// TIA Portal V17 export
// export: Created 2025-03-07T09:17:18.0223508Z, ExportSetting WithDefaults, DisplayName Totally Integrated Automation Portal, DisplayVersion V17 Update 8, DisplayName TIA Portal Openness, DisplayVersion V17 Update 8, DisplayName TIA Portal Version Control Interface, DisplayVersion V17, DisplayName SINAMICS Startdrive Advanced, DisplayVersion V17 SP2, DisplayName SINAMICS Startdrive G110M, G120, G120C, G120D, G120P, G115D, DisplayVersion V17 SP2, DisplayName SINAMICS Startdrive G130, G150, S120, S150, SINAMICS MV, S210, DisplayVersion V17 SP2, DisplayName STEP 7 Professional, DisplayVersion V17 Update 8, DisplayName SINUMERIK ONE STEP 7 Toolbox, DisplayVersion V17 Update 12, DisplayName SINUMERIK 840D sl STEP 7 Toolbox, DisplayVersion V17 Update 12, DisplayName STEP 7 Safety, DisplayVersion V17 Update 6, DisplayName WinCC Advanced, DisplayVersion V17 Update 8
FUNCTION "FC357_NCK_M_CH4_UNIT_2_STA_0" : Void   // FC357, LAD
TITLE = Channel 1 data
{ S7_Optimized_Access := 'FALSE' }
AUTHOR : ETXETAR
VERSION : 1.0
// stored: AutoNumber false, IsIECCheckEnabled false, SetENOAutomatically false, UDAEnableTagReadback false
BEGIN

REGION Network 1: ACKNOWLEDGE M400-UNIT 02 FIXTURE 1 CLAMP SEQUENCE (READ-IN DISABLE) / ACKNOWLEDGE M100-CLAMP SEQUENCE FIXTURE 1
   // NOTE: WHEN THERE IS NOT INDEXING TABLE AVAILABLE IN THE MACHINE DELETE 
   // DB2171.DBX5.0 AND DB2171.DBX2.0
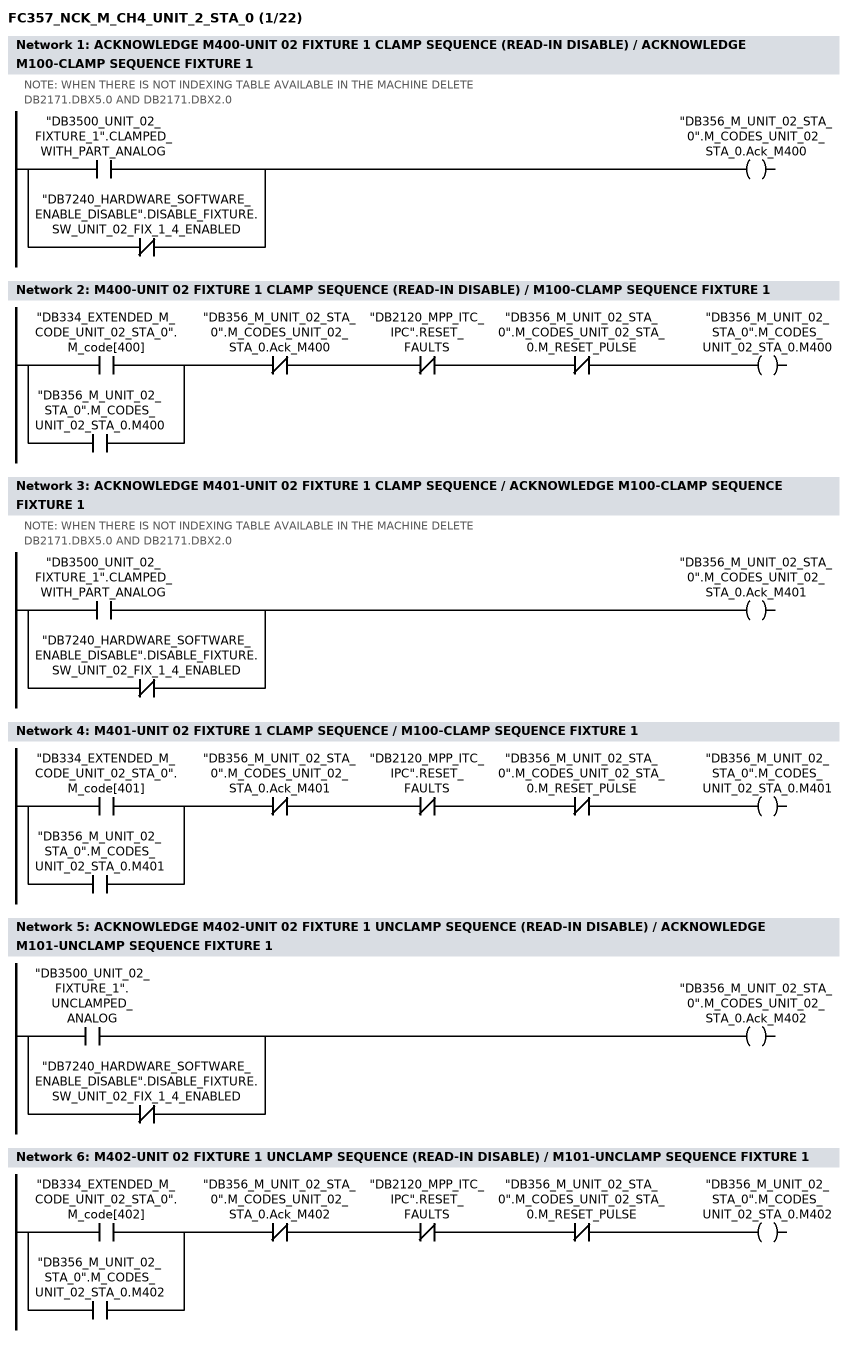
   RUNG wire#powerrail
      Contact( "DB3500_UNIT_02_FIXTURE_1".CLAMPED_WITH_PART_ANALOG )
      wire#w1
      Coil( "DB356_M_UNIT_02_STA_0".M_CODES_UNIT_02_STA_0.Ack_M400 )
   END_RUNG
   RUNG wire#powerrail
      I_Contact( "DB7240_HARDWARE_SOFTWARE_ENABLE_DISABLE".DISABLE_FIXTURE.SW_UNIT_02_FIX_1_4_ENABLED )
   END_RUNG wire#w1
   // the same network as SCL:
   "DB356_M_UNIT_02_STA_0".M_CODES_UNIT_02_STA_0.Ack_M400 := "DB3500_UNIT_02_FIXTURE_1".CLAMPED_WITH_PART_ANALOG OR NOT "DB7240_HARDWARE_SOFTWARE_ENABLE_DISABLE".DISABLE_FIXTURE.SW_UNIT_02_FIX_1_4_ENABLED;
END_REGION

REGION Network 2: M400-UNIT 02 FIXTURE 1 CLAMP SEQUENCE (READ-IN DISABLE) / M100-CLAMP SEQUENCE FIXTURE 1
   RUNG wire#powerrail
      Contact( "DB334_EXTENDED_M_CODE_UNIT_02_STA_0".M_code[400] )
      wire#w1
      I_Contact( "DB356_M_UNIT_02_STA_0".M_CODES_UNIT_02_STA_0.Ack_M400 )
      I_Contact( "DB2120_MPP_ITC_IPC".RESET_FAULTS )
      I_Contact( "DB356_M_UNIT_02_STA_0".M_CODES_UNIT_02_STA_0.M_RESET_PULSE )
      Coil( "DB356_M_UNIT_02_STA_0".M_CODES_UNIT_02_STA_0.M400 )
   END_RUNG
   RUNG wire#powerrail
      Contact( "DB356_M_UNIT_02_STA_0".M_CODES_UNIT_02_STA_0.M400 )
   END_RUNG wire#w1
   // the same network as SCL:
   "DB356_M_UNIT_02_STA_0".M_CODES_UNIT_02_STA_0.M400 := ("DB334_EXTENDED_M_CODE_UNIT_02_STA_0".M_code[400] OR "DB356_M_UNIT_02_STA_0".M_CODES_UNIT_02_STA_0.M400) AND NOT "DB356_M_UNIT_02_STA_0".M_CODES_UNIT_02_STA_0.Ack_M400 AND NOT "DB2120_MPP_ITC_IPC".RESET_FAULTS AND NOT "DB356_M_UNIT_02_STA_0".M_CODES_UNIT_02_STA_0.M_RESET_PULSE;
END_REGION

REGION Network 3: ACKNOWLEDGE M401-UNIT 02 FIXTURE 1 CLAMP SEQUENCE / ACKNOWLEDGE M100-CLAMP SEQUENCE FIXTURE 1
   // NOTE: WHEN THERE IS NOT INDEXING TABLE AVAILABLE IN THE MACHINE DELETE 
   // DB2171.DBX5.0 AND DB2171.DBX2.0
   RUNG wire#powerrail
      Contact( "DB3500_UNIT_02_FIXTURE_1".CLAMPED_WITH_PART_ANALOG )
      wire#w1
      Coil( "DB356_M_UNIT_02_STA_0".M_CODES_UNIT_02_STA_0.Ack_M401 )
   END_RUNG
   RUNG wire#powerrail
      I_Contact( "DB7240_HARDWARE_SOFTWARE_ENABLE_DISABLE".DISABLE_FIXTURE.SW_UNIT_02_FIX_1_4_ENABLED )
   END_RUNG wire#w1
   // the same network as SCL:
   "DB356_M_UNIT_02_STA_0".M_CODES_UNIT_02_STA_0.Ack_M401 := "DB3500_UNIT_02_FIXTURE_1".CLAMPED_WITH_PART_ANALOG OR NOT "DB7240_HARDWARE_SOFTWARE_ENABLE_DISABLE".DISABLE_FIXTURE.SW_UNIT_02_FIX_1_4_ENABLED;
END_REGION

REGION Network 4: M401-UNIT 02 FIXTURE 1 CLAMP SEQUENCE / M100-CLAMP SEQUENCE FIXTURE 1
   RUNG wire#powerrail
      Contact( "DB334_EXTENDED_M_CODE_UNIT_02_STA_0".M_code[401] )
      wire#w1
      I_Contact( "DB356_M_UNIT_02_STA_0".M_CODES_UNIT_02_STA_0.Ack_M401 )
      I_Contact( "DB2120_MPP_ITC_IPC".RESET_FAULTS )
      I_Contact( "DB356_M_UNIT_02_STA_0".M_CODES_UNIT_02_STA_0.M_RESET_PULSE )
      Coil( "DB356_M_UNIT_02_STA_0".M_CODES_UNIT_02_STA_0.M401 )
   END_RUNG
   RUNG wire#powerrail
      Contact( "DB356_M_UNIT_02_STA_0".M_CODES_UNIT_02_STA_0.M401 )
   END_RUNG wire#w1
   // the same network as SCL:
   "DB356_M_UNIT_02_STA_0".M_CODES_UNIT_02_STA_0.M401 := ("DB334_EXTENDED_M_CODE_UNIT_02_STA_0".M_code[401] OR "DB356_M_UNIT_02_STA_0".M_CODES_UNIT_02_STA_0.M401) AND NOT "DB356_M_UNIT_02_STA_0".M_CODES_UNIT_02_STA_0.Ack_M401 AND NOT "DB2120_MPP_ITC_IPC".RESET_FAULTS AND NOT "DB356_M_UNIT_02_STA_0".M_CODES_UNIT_02_STA_0.M_RESET_PULSE;
END_REGION

REGION Network 5: ACKNOWLEDGE M402-UNIT 02 FIXTURE 1 UNCLAMP SEQUENCE (READ-IN DISABLE) / ACKNOWLEDGE M101-UNCLAMP SEQUENCE FIXTURE 1
   RUNG wire#powerrail
      Contact( "DB3500_UNIT_02_FIXTURE_1".UNCLAMPED_ANALOG )
      wire#w1
      Coil( "DB356_M_UNIT_02_STA_0".M_CODES_UNIT_02_STA_0.Ack_M402 )
   END_RUNG
   RUNG wire#powerrail
      I_Contact( "DB7240_HARDWARE_SOFTWARE_ENABLE_DISABLE".DISABLE_FIXTURE.SW_UNIT_02_FIX_1_4_ENABLED )
   END_RUNG wire#w1
   // the same network as SCL:
   "DB356_M_UNIT_02_STA_0".M_CODES_UNIT_02_STA_0.Ack_M402 := "DB3500_UNIT_02_FIXTURE_1".UNCLAMPED_ANALOG OR NOT "DB7240_HARDWARE_SOFTWARE_ENABLE_DISABLE".DISABLE_FIXTURE.SW_UNIT_02_FIX_1_4_ENABLED;
END_REGION

REGION Network 6: M402-UNIT 02 FIXTURE 1 UNCLAMP SEQUENCE (READ-IN DISABLE) / M101-UNCLAMP SEQUENCE FIXTURE 1
   RUNG wire#powerrail
      Contact( "DB334_EXTENDED_M_CODE_UNIT_02_STA_0".M_code[402] )
      wire#w1
      I_Contact( "DB356_M_UNIT_02_STA_0".M_CODES_UNIT_02_STA_0.Ack_M402 )
      I_Contact( "DB2120_MPP_ITC_IPC".RESET_FAULTS )
      I_Contact( "DB356_M_UNIT_02_STA_0".M_CODES_UNIT_02_STA_0.M_RESET_PULSE )
      Coil( "DB356_M_UNIT_02_STA_0".M_CODES_UNIT_02_STA_0.M402 )
   END_RUNG
   RUNG wire#powerrail
      Contact( "DB356_M_UNIT_02_STA_0".M_CODES_UNIT_02_STA_0.M402 )
   END_RUNG wire#w1
   // the same network as SCL:
   "DB356_M_UNIT_02_STA_0".M_CODES_UNIT_02_STA_0.M402 := ("DB334_EXTENDED_M_CODE_UNIT_02_STA_0".M_code[402] OR "DB356_M_UNIT_02_STA_0".M_CODES_UNIT_02_STA_0.M402) AND NOT "DB356_M_UNIT_02_STA_0".M_CODES_UNIT_02_STA_0.Ack_M402 AND NOT "DB2120_MPP_ITC_IPC".RESET_FAULTS AND NOT "DB356_M_UNIT_02_STA_0".M_CODES_UNIT_02_STA_0.M_RESET_PULSE;
END_REGION

REGION Network 7: ACKNOWLEDGE M403-UNIT 02 FIXTURE 1 UNCLAMP SEQUENCE / ACKNOWLEDGE M101-UNCLAMP SEQUENCE FIXTURE 1
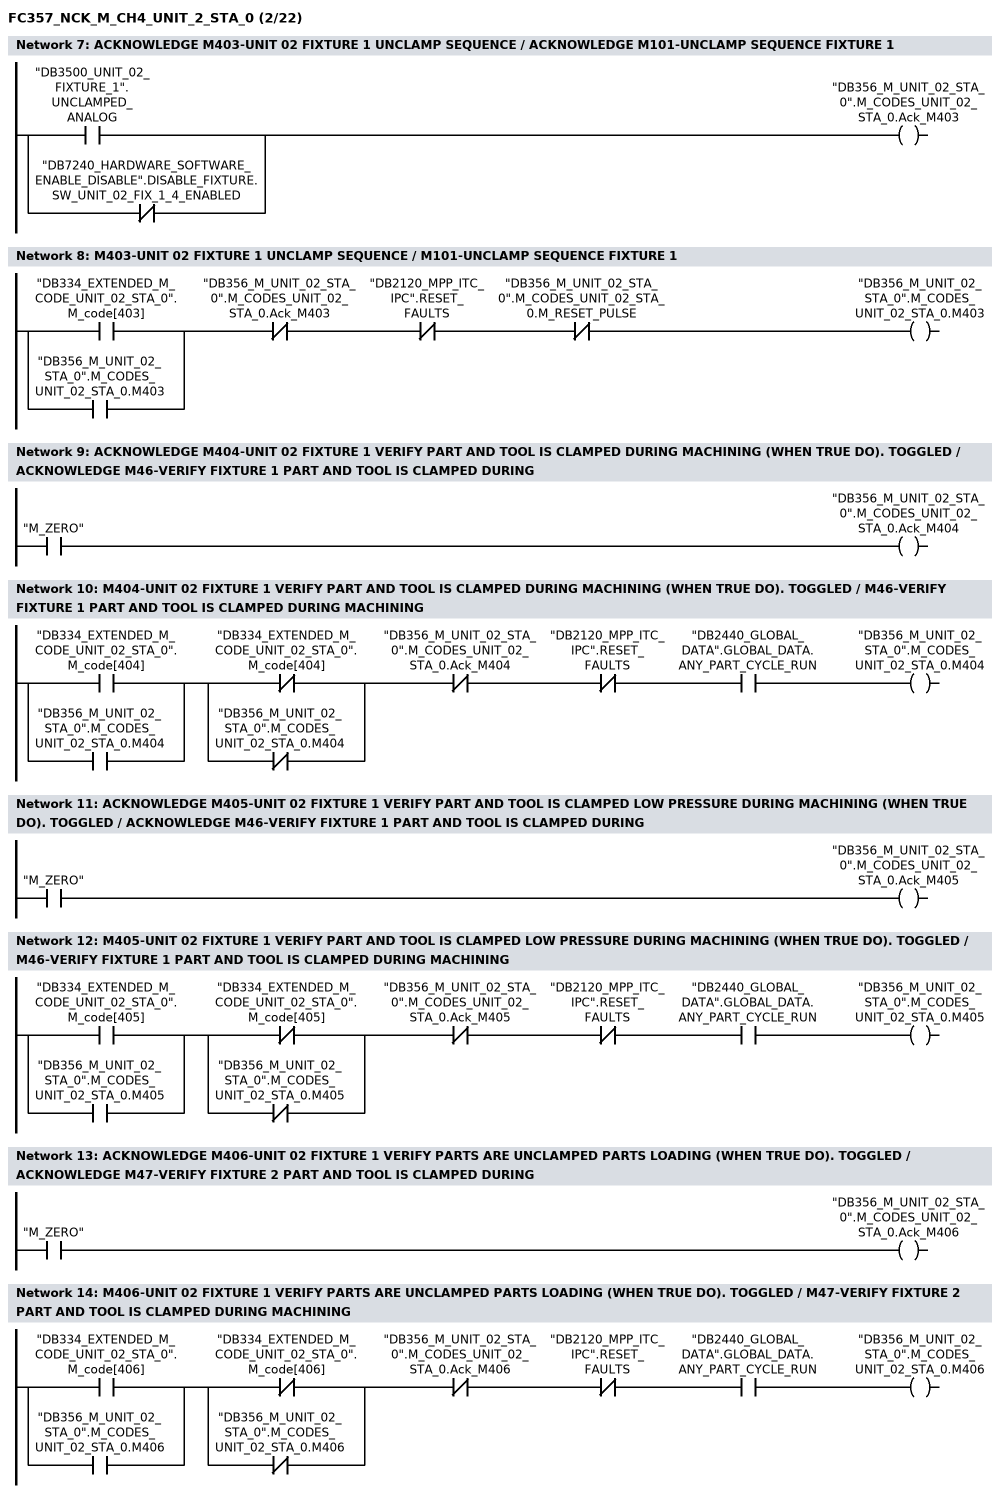
   RUNG wire#powerrail
      Contact( "DB3500_UNIT_02_FIXTURE_1".UNCLAMPED_ANALOG )
      wire#w1
      Coil( "DB356_M_UNIT_02_STA_0".M_CODES_UNIT_02_STA_0.Ack_M403 )
   END_RUNG
   RUNG wire#powerrail
      I_Contact( "DB7240_HARDWARE_SOFTWARE_ENABLE_DISABLE".DISABLE_FIXTURE.SW_UNIT_02_FIX_1_4_ENABLED )
   END_RUNG wire#w1
   // the same network as SCL:
   "DB356_M_UNIT_02_STA_0".M_CODES_UNIT_02_STA_0.Ack_M403 := "DB3500_UNIT_02_FIXTURE_1".UNCLAMPED_ANALOG OR NOT "DB7240_HARDWARE_SOFTWARE_ENABLE_DISABLE".DISABLE_FIXTURE.SW_UNIT_02_FIX_1_4_ENABLED;
END_REGION

REGION Network 8: M403-UNIT 02 FIXTURE 1 UNCLAMP SEQUENCE / M101-UNCLAMP SEQUENCE FIXTURE 1
   RUNG wire#powerrail
      Contact( "DB334_EXTENDED_M_CODE_UNIT_02_STA_0".M_code[403] )
      wire#w1
      I_Contact( "DB356_M_UNIT_02_STA_0".M_CODES_UNIT_02_STA_0.Ack_M403 )
      I_Contact( "DB2120_MPP_ITC_IPC".RESET_FAULTS )
      I_Contact( "DB356_M_UNIT_02_STA_0".M_CODES_UNIT_02_STA_0.M_RESET_PULSE )
      Coil( "DB356_M_UNIT_02_STA_0".M_CODES_UNIT_02_STA_0.M403 )
   END_RUNG
   RUNG wire#powerrail
      Contact( "DB356_M_UNIT_02_STA_0".M_CODES_UNIT_02_STA_0.M403 )
   END_RUNG wire#w1
   // the same network as SCL:
   "DB356_M_UNIT_02_STA_0".M_CODES_UNIT_02_STA_0.M403 := ("DB334_EXTENDED_M_CODE_UNIT_02_STA_0".M_code[403] OR "DB356_M_UNIT_02_STA_0".M_CODES_UNIT_02_STA_0.M403) AND NOT "DB356_M_UNIT_02_STA_0".M_CODES_UNIT_02_STA_0.Ack_M403 AND NOT "DB2120_MPP_ITC_IPC".RESET_FAULTS AND NOT "DB356_M_UNIT_02_STA_0".M_CODES_UNIT_02_STA_0.M_RESET_PULSE;
END_REGION

REGION Network 9: ACKNOWLEDGE M404-UNIT 02 FIXTURE 1 VERIFY PART AND TOOL IS CLAMPED DURING MACHINING (WHEN TRUE DO). TOGGLED / ACKNOWLEDGE M46-VERIFY FIXTURE 1 PART AND TOOL IS CLAMPED DURING
   RUNG wire#powerrail
      Contact( "M_ZERO" )
      Coil( "DB356_M_UNIT_02_STA_0".M_CODES_UNIT_02_STA_0.Ack_M404 )
   END_RUNG
   // the same network as SCL:
   "DB356_M_UNIT_02_STA_0".M_CODES_UNIT_02_STA_0.Ack_M404 := "M_ZERO";
END_REGION

REGION Network 10: M404-UNIT 02 FIXTURE 1 VERIFY PART AND TOOL IS CLAMPED DURING MACHINING (WHEN TRUE DO). TOGGLED / M46-VERIFY FIXTURE 1 PART AND TOOL IS CLAMPED DURING MACHINING
   RUNG wire#powerrail
      Contact( "DB334_EXTENDED_M_CODE_UNIT_02_STA_0".M_code[404] )
      wire#w1
      I_Contact( "DB334_EXTENDED_M_CODE_UNIT_02_STA_0".M_code[404] )
      wire#w2
      I_Contact( "DB356_M_UNIT_02_STA_0".M_CODES_UNIT_02_STA_0.Ack_M404 )
      I_Contact( "DB2120_MPP_ITC_IPC".RESET_FAULTS )
      Contact( "DB2440_GLOBAL_DATA".GLOBAL_DATA.ANY_PART_CYCLE_RUN )
      Coil( "DB356_M_UNIT_02_STA_0".M_CODES_UNIT_02_STA_0.M404 )
   END_RUNG
   RUNG wire#powerrail
      Contact( "DB356_M_UNIT_02_STA_0".M_CODES_UNIT_02_STA_0.M404 )
   END_RUNG wire#w1
   RUNG wire#w1
      I_Contact( "DB356_M_UNIT_02_STA_0".M_CODES_UNIT_02_STA_0.M404 )
   END_RUNG wire#w2
   // the same network as SCL:
   "DB356_M_UNIT_02_STA_0".M_CODES_UNIT_02_STA_0.M404 := ("DB334_EXTENDED_M_CODE_UNIT_02_STA_0".M_code[404] OR "DB356_M_UNIT_02_STA_0".M_CODES_UNIT_02_STA_0.M404) AND (NOT "DB334_EXTENDED_M_CODE_UNIT_02_STA_0".M_code[404] OR NOT "DB356_M_UNIT_02_STA_0".M_CODES_UNIT_02_STA_0.M404) AND NOT "DB356_M_UNIT_02_STA_0".M_CODES_UNIT_02_STA_0.Ack_M404 AND NOT "DB2120_MPP_ITC_IPC".RESET_FAULTS AND "DB2440_GLOBAL_DATA".GLOBAL_DATA.ANY_PART_CYCLE_RUN;
END_REGION

REGION Network 11: ACKNOWLEDGE M405-UNIT 02 FIXTURE 1 VERIFY PART AND TOOL IS CLAMPED LOW PRESSURE DURING MACHINING (WHEN TRUE DO). TOGGLED / ACKNOWLEDGE M46-VERIFY FIXTURE 1 PART AND TOOL IS CLAMPED DURING
   RUNG wire#powerrail
      Contact( "M_ZERO" )
      Coil( "DB356_M_UNIT_02_STA_0".M_CODES_UNIT_02_STA_0.Ack_M405 )
   END_RUNG
   // the same network as SCL:
   "DB356_M_UNIT_02_STA_0".M_CODES_UNIT_02_STA_0.Ack_M405 := "M_ZERO";
END_REGION

REGION Network 12: M405-UNIT 02 FIXTURE 1 VERIFY PART AND TOOL IS CLAMPED LOW PRESSURE DURING MACHINING (WHEN TRUE DO). TOGGLED / M46-VERIFY FIXTURE 1 PART AND TOOL IS CLAMPED DURING MACHINING
   RUNG wire#powerrail
      Contact( "DB334_EXTENDED_M_CODE_UNIT_02_STA_0".M_code[405] )
      wire#w1
      I_Contact( "DB334_EXTENDED_M_CODE_UNIT_02_STA_0".M_code[405] )
      wire#w2
      I_Contact( "DB356_M_UNIT_02_STA_0".M_CODES_UNIT_02_STA_0.Ack_M405 )
      I_Contact( "DB2120_MPP_ITC_IPC".RESET_FAULTS )
      Contact( "DB2440_GLOBAL_DATA".GLOBAL_DATA.ANY_PART_CYCLE_RUN )
      Coil( "DB356_M_UNIT_02_STA_0".M_CODES_UNIT_02_STA_0.M405 )
   END_RUNG
   RUNG wire#powerrail
      Contact( "DB356_M_UNIT_02_STA_0".M_CODES_UNIT_02_STA_0.M405 )
   END_RUNG wire#w1
   RUNG wire#w1
      I_Contact( "DB356_M_UNIT_02_STA_0".M_CODES_UNIT_02_STA_0.M405 )
   END_RUNG wire#w2
   // the same network as SCL:
   "DB356_M_UNIT_02_STA_0".M_CODES_UNIT_02_STA_0.M405 := ("DB334_EXTENDED_M_CODE_UNIT_02_STA_0".M_code[405] OR "DB356_M_UNIT_02_STA_0".M_CODES_UNIT_02_STA_0.M405) AND (NOT "DB334_EXTENDED_M_CODE_UNIT_02_STA_0".M_code[405] OR NOT "DB356_M_UNIT_02_STA_0".M_CODES_UNIT_02_STA_0.M405) AND NOT "DB356_M_UNIT_02_STA_0".M_CODES_UNIT_02_STA_0.Ack_M405 AND NOT "DB2120_MPP_ITC_IPC".RESET_FAULTS AND "DB2440_GLOBAL_DATA".GLOBAL_DATA.ANY_PART_CYCLE_RUN;
END_REGION

REGION Network 13: ACKNOWLEDGE M406-UNIT 02 FIXTURE 1 VERIFY PARTS ARE UNCLAMPED PARTS LOADING (WHEN TRUE DO). TOGGLED / ACKNOWLEDGE M47-VERIFY FIXTURE 2 PART AND TOOL IS CLAMPED DURING
   RUNG wire#powerrail
      Contact( "M_ZERO" )
      Coil( "DB356_M_UNIT_02_STA_0".M_CODES_UNIT_02_STA_0.Ack_M406 )
   END_RUNG
   // the same network as SCL:
   "DB356_M_UNIT_02_STA_0".M_CODES_UNIT_02_STA_0.Ack_M406 := "M_ZERO";
END_REGION

REGION Network 14: M406-UNIT 02 FIXTURE 1 VERIFY PARTS ARE UNCLAMPED PARTS LOADING (WHEN TRUE DO). TOGGLED / M47-VERIFY FIXTURE 2 PART AND TOOL IS CLAMPED DURING MACHINING
   RUNG wire#powerrail
      Contact( "DB334_EXTENDED_M_CODE_UNIT_02_STA_0".M_code[406] )
      wire#w1
      I_Contact( "DB334_EXTENDED_M_CODE_UNIT_02_STA_0".M_code[406] )
      wire#w2
      I_Contact( "DB356_M_UNIT_02_STA_0".M_CODES_UNIT_02_STA_0.Ack_M406 )
      I_Contact( "DB2120_MPP_ITC_IPC".RESET_FAULTS )
      Contact( "DB2440_GLOBAL_DATA".GLOBAL_DATA.ANY_PART_CYCLE_RUN )
      Coil( "DB356_M_UNIT_02_STA_0".M_CODES_UNIT_02_STA_0.M406 )
   END_RUNG
   RUNG wire#powerrail
      Contact( "DB356_M_UNIT_02_STA_0".M_CODES_UNIT_02_STA_0.M406 )
   END_RUNG wire#w1
   RUNG wire#w1
      I_Contact( "DB356_M_UNIT_02_STA_0".M_CODES_UNIT_02_STA_0.M406 )
   END_RUNG wire#w2
   // the same network as SCL:
   "DB356_M_UNIT_02_STA_0".M_CODES_UNIT_02_STA_0.M406 := ("DB334_EXTENDED_M_CODE_UNIT_02_STA_0".M_code[406] OR "DB356_M_UNIT_02_STA_0".M_CODES_UNIT_02_STA_0.M406) AND (NOT "DB334_EXTENDED_M_CODE_UNIT_02_STA_0".M_code[406] OR NOT "DB356_M_UNIT_02_STA_0".M_CODES_UNIT_02_STA_0.M406) AND NOT "DB356_M_UNIT_02_STA_0".M_CODES_UNIT_02_STA_0.Ack_M406 AND NOT "DB2120_MPP_ITC_IPC".RESET_FAULTS AND "DB2440_GLOBAL_DATA".GLOBAL_DATA.ANY_PART_CYCLE_RUN;
END_REGION

REGION Network 15: ACKNOWLEDGE M407-UNIT 02 FIXTURE 1 VERIFY FIXTURE REMAINS CLAMPED
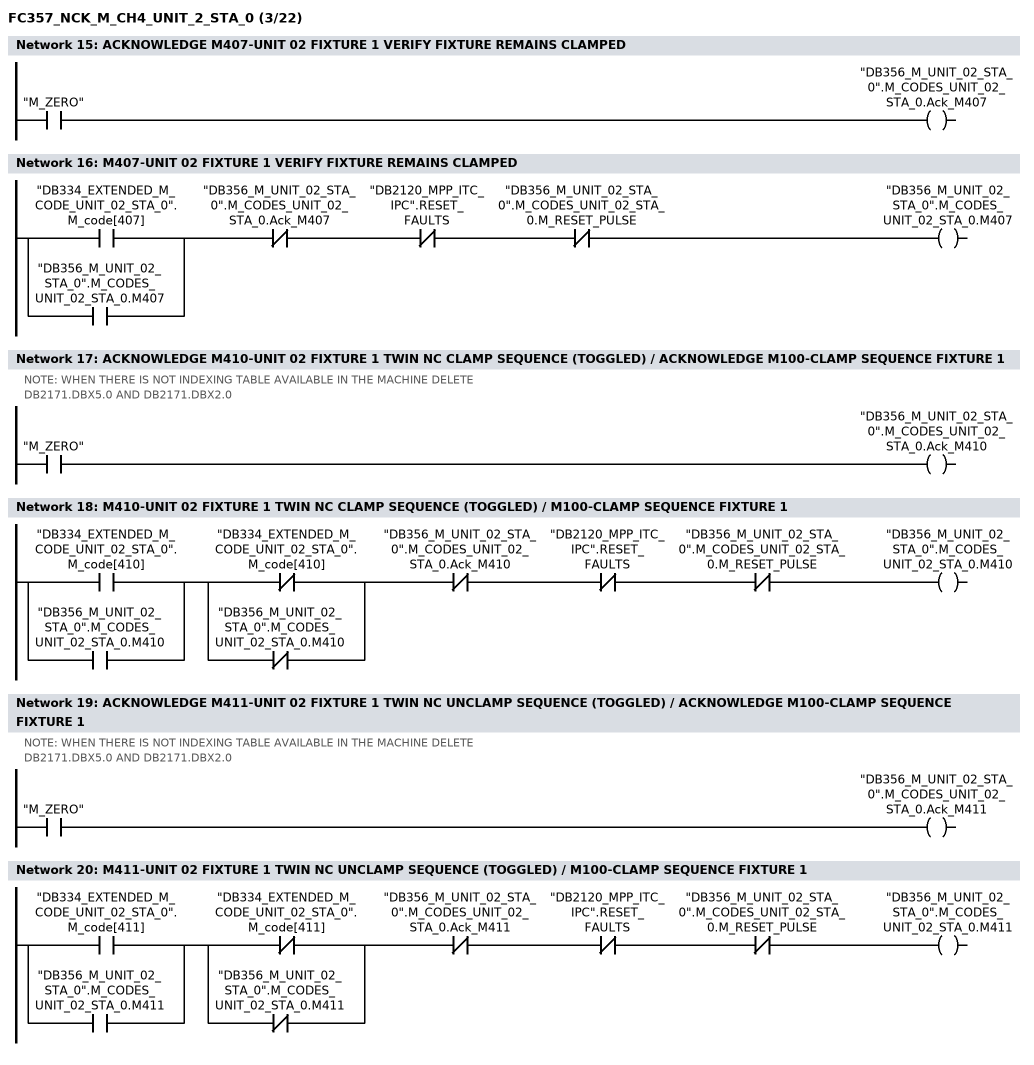
   RUNG wire#powerrail
      Contact( "M_ZERO" )
      Coil( "DB356_M_UNIT_02_STA_0".M_CODES_UNIT_02_STA_0.Ack_M407 )
   END_RUNG
   // the same network as SCL:
   "DB356_M_UNIT_02_STA_0".M_CODES_UNIT_02_STA_0.Ack_M407 := "M_ZERO";
END_REGION

REGION Network 16: M407-UNIT 02 FIXTURE 1 VERIFY FIXTURE REMAINS CLAMPED
   RUNG wire#powerrail
      Contact( "DB334_EXTENDED_M_CODE_UNIT_02_STA_0".M_code[407] )
      wire#w1
      I_Contact( "DB356_M_UNIT_02_STA_0".M_CODES_UNIT_02_STA_0.Ack_M407 )
      I_Contact( "DB2120_MPP_ITC_IPC".RESET_FAULTS )
      I_Contact( "DB356_M_UNIT_02_STA_0".M_CODES_UNIT_02_STA_0.M_RESET_PULSE )
      Coil( "DB356_M_UNIT_02_STA_0".M_CODES_UNIT_02_STA_0.M407 )
   END_RUNG
   RUNG wire#powerrail
      Contact( "DB356_M_UNIT_02_STA_0".M_CODES_UNIT_02_STA_0.M407 )
   END_RUNG wire#w1
   // the same network as SCL:
   "DB356_M_UNIT_02_STA_0".M_CODES_UNIT_02_STA_0.M407 := ("DB334_EXTENDED_M_CODE_UNIT_02_STA_0".M_code[407] OR "DB356_M_UNIT_02_STA_0".M_CODES_UNIT_02_STA_0.M407) AND NOT "DB356_M_UNIT_02_STA_0".M_CODES_UNIT_02_STA_0.Ack_M407 AND NOT "DB2120_MPP_ITC_IPC".RESET_FAULTS AND NOT "DB356_M_UNIT_02_STA_0".M_CODES_UNIT_02_STA_0.M_RESET_PULSE;
END_REGION

REGION Network 17: ACKNOWLEDGE M410-UNIT 02 FIXTURE 1 TWIN NC CLAMP SEQUENCE (TOGGLED) / ACKNOWLEDGE M100-CLAMP SEQUENCE FIXTURE 1
   // NOTE: WHEN THERE IS NOT INDEXING TABLE AVAILABLE IN THE MACHINE DELETE 
   // DB2171.DBX5.0 AND DB2171.DBX2.0
   RUNG wire#powerrail
      Contact( "M_ZERO" )
      Coil( "DB356_M_UNIT_02_STA_0".M_CODES_UNIT_02_STA_0.Ack_M410 )
   END_RUNG
   // the same network as SCL:
   "DB356_M_UNIT_02_STA_0".M_CODES_UNIT_02_STA_0.Ack_M410 := "M_ZERO";
END_REGION

REGION Network 18: M410-UNIT 02 FIXTURE 1 TWIN NC CLAMP SEQUENCE (TOGGLED) / M100-CLAMP SEQUENCE FIXTURE 1
   RUNG wire#powerrail
      Contact( "DB334_EXTENDED_M_CODE_UNIT_02_STA_0".M_code[410] )
      wire#w1
      I_Contact( "DB334_EXTENDED_M_CODE_UNIT_02_STA_0".M_code[410] )
      wire#w2
      I_Contact( "DB356_M_UNIT_02_STA_0".M_CODES_UNIT_02_STA_0.Ack_M410 )
      I_Contact( "DB2120_MPP_ITC_IPC".RESET_FAULTS )
      I_Contact( "DB356_M_UNIT_02_STA_0".M_CODES_UNIT_02_STA_0.M_RESET_PULSE )
      Coil( "DB356_M_UNIT_02_STA_0".M_CODES_UNIT_02_STA_0.M410 )
   END_RUNG
   RUNG wire#powerrail
      Contact( "DB356_M_UNIT_02_STA_0".M_CODES_UNIT_02_STA_0.M410 )
   END_RUNG wire#w1
   RUNG wire#w1
      I_Contact( "DB356_M_UNIT_02_STA_0".M_CODES_UNIT_02_STA_0.M410 )
   END_RUNG wire#w2
   // the same network as SCL:
   "DB356_M_UNIT_02_STA_0".M_CODES_UNIT_02_STA_0.M410 := ("DB334_EXTENDED_M_CODE_UNIT_02_STA_0".M_code[410] OR "DB356_M_UNIT_02_STA_0".M_CODES_UNIT_02_STA_0.M410) AND (NOT "DB334_EXTENDED_M_CODE_UNIT_02_STA_0".M_code[410] OR NOT "DB356_M_UNIT_02_STA_0".M_CODES_UNIT_02_STA_0.M410) AND NOT "DB356_M_UNIT_02_STA_0".M_CODES_UNIT_02_STA_0.Ack_M410 AND NOT "DB2120_MPP_ITC_IPC".RESET_FAULTS AND NOT "DB356_M_UNIT_02_STA_0".M_CODES_UNIT_02_STA_0.M_RESET_PULSE;
END_REGION

REGION Network 19: ACKNOWLEDGE M411-UNIT 02 FIXTURE 1 TWIN NC UNCLAMP SEQUENCE (TOGGLED) / ACKNOWLEDGE M100-CLAMP SEQUENCE FIXTURE 1
   // NOTE: WHEN THERE IS NOT INDEXING TABLE AVAILABLE IN THE MACHINE DELETE 
   // DB2171.DBX5.0 AND DB2171.DBX2.0
   RUNG wire#powerrail
      Contact( "M_ZERO" )
      Coil( "DB356_M_UNIT_02_STA_0".M_CODES_UNIT_02_STA_0.Ack_M411 )
   END_RUNG
   // the same network as SCL:
   "DB356_M_UNIT_02_STA_0".M_CODES_UNIT_02_STA_0.Ack_M411 := "M_ZERO";
END_REGION

REGION Network 20: M411-UNIT 02 FIXTURE 1 TWIN NC UNCLAMP SEQUENCE (TOGGLED) / M100-CLAMP SEQUENCE FIXTURE 1
   RUNG wire#powerrail
      Contact( "DB334_EXTENDED_M_CODE_UNIT_02_STA_0".M_code[411] )
      wire#w1
      I_Contact( "DB334_EXTENDED_M_CODE_UNIT_02_STA_0".M_code[411] )
      wire#w2
      I_Contact( "DB356_M_UNIT_02_STA_0".M_CODES_UNIT_02_STA_0.Ack_M411 )
      I_Contact( "DB2120_MPP_ITC_IPC".RESET_FAULTS )
      I_Contact( "DB356_M_UNIT_02_STA_0".M_CODES_UNIT_02_STA_0.M_RESET_PULSE )
      Coil( "DB356_M_UNIT_02_STA_0".M_CODES_UNIT_02_STA_0.M411 )
   END_RUNG
   RUNG wire#powerrail
      Contact( "DB356_M_UNIT_02_STA_0".M_CODES_UNIT_02_STA_0.M411 )
   END_RUNG wire#w1
   RUNG wire#w1
      I_Contact( "DB356_M_UNIT_02_STA_0".M_CODES_UNIT_02_STA_0.M411 )
   END_RUNG wire#w2
   // the same network as SCL:
   "DB356_M_UNIT_02_STA_0".M_CODES_UNIT_02_STA_0.M411 := ("DB334_EXTENDED_M_CODE_UNIT_02_STA_0".M_code[411] OR "DB356_M_UNIT_02_STA_0".M_CODES_UNIT_02_STA_0.M411) AND (NOT "DB334_EXTENDED_M_CODE_UNIT_02_STA_0".M_code[411] OR NOT "DB356_M_UNIT_02_STA_0".M_CODES_UNIT_02_STA_0.M411) AND NOT "DB356_M_UNIT_02_STA_0".M_CODES_UNIT_02_STA_0.Ack_M411 AND NOT "DB2120_MPP_ITC_IPC".RESET_FAULTS AND NOT "DB356_M_UNIT_02_STA_0".M_CODES_UNIT_02_STA_0.M_RESET_PULSE;
END_REGION

REGION Network 21: ACKNOWLEDGE M420- UNIT 02 FIXTURE 1 GRIPPER CLOSE (READ-IN DISABLE)
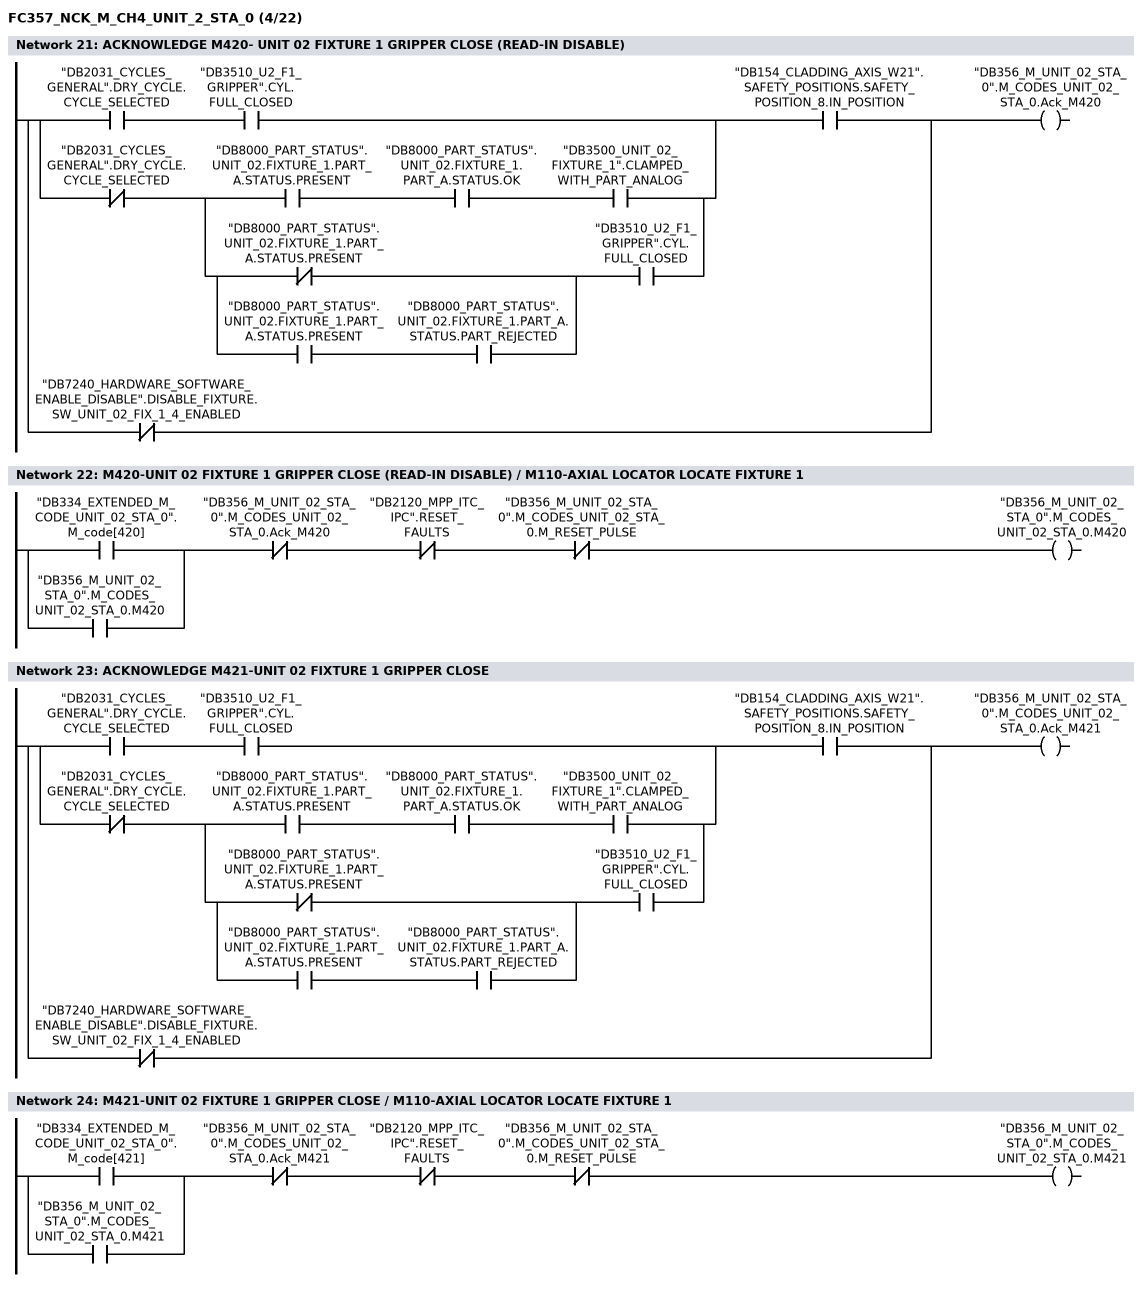
   RUNG wire#powerrail
      Contact( "DB2031_CYCLES_GENERAL".DRY_CYCLE.CYCLE_SELECTED )
      Contact( "DB3510_U2_F1_GRIPPER".CYL.FULL_CLOSED )
      wire#w1
      Contact( "DB154_CLADDING_AXIS_W21".SAFETY_POSITIONS.SAFETY_POSITION_8.IN_POSITION )
      wire#w4
      Coil( "DB356_M_UNIT_02_STA_0".M_CODES_UNIT_02_STA_0.Ack_M420 )
   END_RUNG
   RUNG wire#powerrail
      I_Contact( "DB2031_CYCLES_GENERAL".DRY_CYCLE.CYCLE_SELECTED )
      wire#w2
      Contact( "DB8000_PART_STATUS".UNIT_02.FIXTURE_1.PART_A.STATUS.PRESENT )
      Contact( "DB8000_PART_STATUS".UNIT_02.FIXTURE_1.PART_A.STATUS.OK )
      Contact( "DB3500_UNIT_02_FIXTURE_1".CLAMPED_WITH_PART_ANALOG )
   END_RUNG wire#w1
   RUNG wire#w2
      I_Contact( "DB8000_PART_STATUS".UNIT_02.FIXTURE_1.PART_A.STATUS.PRESENT )
      wire#w3
      Contact( "DB3510_U2_F1_GRIPPER".CYL.FULL_CLOSED )
   END_RUNG wire#w1
   RUNG wire#w2
      Contact( "DB8000_PART_STATUS".UNIT_02.FIXTURE_1.PART_A.STATUS.PRESENT )
      Contact( "DB8000_PART_STATUS".UNIT_02.FIXTURE_1.PART_A.STATUS.PART_REJECTED )
   END_RUNG wire#w3
   RUNG wire#powerrail
      I_Contact( "DB7240_HARDWARE_SOFTWARE_ENABLE_DISABLE".DISABLE_FIXTURE.SW_UNIT_02_FIX_1_4_ENABLED )
   END_RUNG wire#w4
   // the same network as SCL:
   "DB356_M_UNIT_02_STA_0".M_CODES_UNIT_02_STA_0.Ack_M420 := ((("DB2031_CYCLES_GENERAL".DRY_CYCLE.CYCLE_SELECTED AND "DB3510_U2_F1_GRIPPER".CYL.FULL_CLOSED) OR (NOT "DB2031_CYCLES_GENERAL".DRY_CYCLE.CYCLE_SELECTED AND (("DB8000_PART_STATUS".UNIT_02.FIXTURE_1.PART_A.STATUS.PRESENT AND "DB8000_PART_STATUS".UNIT_02.FIXTURE_1.PART_A.STATUS.OK AND "DB3500_UNIT_02_FIXTURE_1".CLAMPED_WITH_PART_ANALOG) OR ((NOT "DB8000_PART_STATUS".UNIT_02.FIXTURE_1.PART_A.STATUS.PRESENT OR ("DB8000_PART_STATUS".UNIT_02.FIXTURE_1.PART_A.STATUS.PRESENT AND "DB8000_PART_STATUS".UNIT_02.FIXTURE_1.PART_A.STATUS.PART_REJECTED)) AND "DB3510_U2_F1_GRIPPER".CYL.FULL_CLOSED)))) AND "DB154_CLADDING_AXIS_W21".SAFETY_POSITIONS.SAFETY_POSITION_8.IN_POSITION) OR NOT "DB7240_HARDWARE_SOFTWARE_ENABLE_DISABLE".DISABLE_FIXTURE.SW_UNIT_02_FIX_1_4_ENABLED;
END_REGION

REGION Network 22: M420-UNIT 02 FIXTURE 1 GRIPPER CLOSE (READ-IN DISABLE) / M110-AXIAL LOCATOR LOCATE FIXTURE 1
   RUNG wire#powerrail
      Contact( "DB334_EXTENDED_M_CODE_UNIT_02_STA_0".M_code[420] )
      wire#w1
      I_Contact( "DB356_M_UNIT_02_STA_0".M_CODES_UNIT_02_STA_0.Ack_M420 )
      I_Contact( "DB2120_MPP_ITC_IPC".RESET_FAULTS )
      I_Contact( "DB356_M_UNIT_02_STA_0".M_CODES_UNIT_02_STA_0.M_RESET_PULSE )
      Coil( "DB356_M_UNIT_02_STA_0".M_CODES_UNIT_02_STA_0.M420 )
   END_RUNG
   RUNG wire#powerrail
      Contact( "DB356_M_UNIT_02_STA_0".M_CODES_UNIT_02_STA_0.M420 )
   END_RUNG wire#w1
   // the same network as SCL:
   "DB356_M_UNIT_02_STA_0".M_CODES_UNIT_02_STA_0.M420 := ("DB334_EXTENDED_M_CODE_UNIT_02_STA_0".M_code[420] OR "DB356_M_UNIT_02_STA_0".M_CODES_UNIT_02_STA_0.M420) AND NOT "DB356_M_UNIT_02_STA_0".M_CODES_UNIT_02_STA_0.Ack_M420 AND NOT "DB2120_MPP_ITC_IPC".RESET_FAULTS AND NOT "DB356_M_UNIT_02_STA_0".M_CODES_UNIT_02_STA_0.M_RESET_PULSE;
END_REGION

REGION Network 23: ACKNOWLEDGE M421-UNIT 02 FIXTURE 1 GRIPPER CLOSE
   RUNG wire#powerrail
      Contact( "DB2031_CYCLES_GENERAL".DRY_CYCLE.CYCLE_SELECTED )
      Contact( "DB3510_U2_F1_GRIPPER".CYL.FULL_CLOSED )
      wire#w1
      Contact( "DB154_CLADDING_AXIS_W21".SAFETY_POSITIONS.SAFETY_POSITION_8.IN_POSITION )
      wire#w4
      Coil( "DB356_M_UNIT_02_STA_0".M_CODES_UNIT_02_STA_0.Ack_M421 )
   END_RUNG
   RUNG wire#powerrail
      I_Contact( "DB2031_CYCLES_GENERAL".DRY_CYCLE.CYCLE_SELECTED )
      wire#w2
      Contact( "DB8000_PART_STATUS".UNIT_02.FIXTURE_1.PART_A.STATUS.PRESENT )
      Contact( "DB8000_PART_STATUS".UNIT_02.FIXTURE_1.PART_A.STATUS.OK )
      Contact( "DB3500_UNIT_02_FIXTURE_1".CLAMPED_WITH_PART_ANALOG )
   END_RUNG wire#w1
   RUNG wire#w2
      I_Contact( "DB8000_PART_STATUS".UNIT_02.FIXTURE_1.PART_A.STATUS.PRESENT )
      wire#w3
      Contact( "DB3510_U2_F1_GRIPPER".CYL.FULL_CLOSED )
   END_RUNG wire#w1
   RUNG wire#w2
      Contact( "DB8000_PART_STATUS".UNIT_02.FIXTURE_1.PART_A.STATUS.PRESENT )
      Contact( "DB8000_PART_STATUS".UNIT_02.FIXTURE_1.PART_A.STATUS.PART_REJECTED )
   END_RUNG wire#w3
   RUNG wire#powerrail
      I_Contact( "DB7240_HARDWARE_SOFTWARE_ENABLE_DISABLE".DISABLE_FIXTURE.SW_UNIT_02_FIX_1_4_ENABLED )
   END_RUNG wire#w4
   // the same network as SCL:
   "DB356_M_UNIT_02_STA_0".M_CODES_UNIT_02_STA_0.Ack_M421 := ((("DB2031_CYCLES_GENERAL".DRY_CYCLE.CYCLE_SELECTED AND "DB3510_U2_F1_GRIPPER".CYL.FULL_CLOSED) OR (NOT "DB2031_CYCLES_GENERAL".DRY_CYCLE.CYCLE_SELECTED AND (("DB8000_PART_STATUS".UNIT_02.FIXTURE_1.PART_A.STATUS.PRESENT AND "DB8000_PART_STATUS".UNIT_02.FIXTURE_1.PART_A.STATUS.OK AND "DB3500_UNIT_02_FIXTURE_1".CLAMPED_WITH_PART_ANALOG) OR ((NOT "DB8000_PART_STATUS".UNIT_02.FIXTURE_1.PART_A.STATUS.PRESENT OR ("DB8000_PART_STATUS".UNIT_02.FIXTURE_1.PART_A.STATUS.PRESENT AND "DB8000_PART_STATUS".UNIT_02.FIXTURE_1.PART_A.STATUS.PART_REJECTED)) AND "DB3510_U2_F1_GRIPPER".CYL.FULL_CLOSED)))) AND "DB154_CLADDING_AXIS_W21".SAFETY_POSITIONS.SAFETY_POSITION_8.IN_POSITION) OR NOT "DB7240_HARDWARE_SOFTWARE_ENABLE_DISABLE".DISABLE_FIXTURE.SW_UNIT_02_FIX_1_4_ENABLED;
END_REGION

REGION Network 24: M421-UNIT 02 FIXTURE 1 GRIPPER CLOSE / M110-AXIAL LOCATOR LOCATE FIXTURE 1
   RUNG wire#powerrail
      Contact( "DB334_EXTENDED_M_CODE_UNIT_02_STA_0".M_code[421] )
      wire#w1
      I_Contact( "DB356_M_UNIT_02_STA_0".M_CODES_UNIT_02_STA_0.Ack_M421 )
      I_Contact( "DB2120_MPP_ITC_IPC".RESET_FAULTS )
      I_Contact( "DB356_M_UNIT_02_STA_0".M_CODES_UNIT_02_STA_0.M_RESET_PULSE )
      Coil( "DB356_M_UNIT_02_STA_0".M_CODES_UNIT_02_STA_0.M421 )
   END_RUNG
   RUNG wire#powerrail
      Contact( "DB356_M_UNIT_02_STA_0".M_CODES_UNIT_02_STA_0.M421 )
   END_RUNG wire#w1
   // the same network as SCL:
   "DB356_M_UNIT_02_STA_0".M_CODES_UNIT_02_STA_0.M421 := ("DB334_EXTENDED_M_CODE_UNIT_02_STA_0".M_code[421] OR "DB356_M_UNIT_02_STA_0".M_CODES_UNIT_02_STA_0.M421) AND NOT "DB356_M_UNIT_02_STA_0".M_CODES_UNIT_02_STA_0.Ack_M421 AND NOT "DB2120_MPP_ITC_IPC".RESET_FAULTS AND NOT "DB356_M_UNIT_02_STA_0".M_CODES_UNIT_02_STA_0.M_RESET_PULSE;
END_REGION

REGION Network 25: ACKNOWLEDGE M422-UNIT 02 FIXTURE 1 GRIPPER OPEN (READ-IN DISABLE) / ACKNOWLEDGE M111-AXIAL LOCATOR RETURN FIXTURE 1
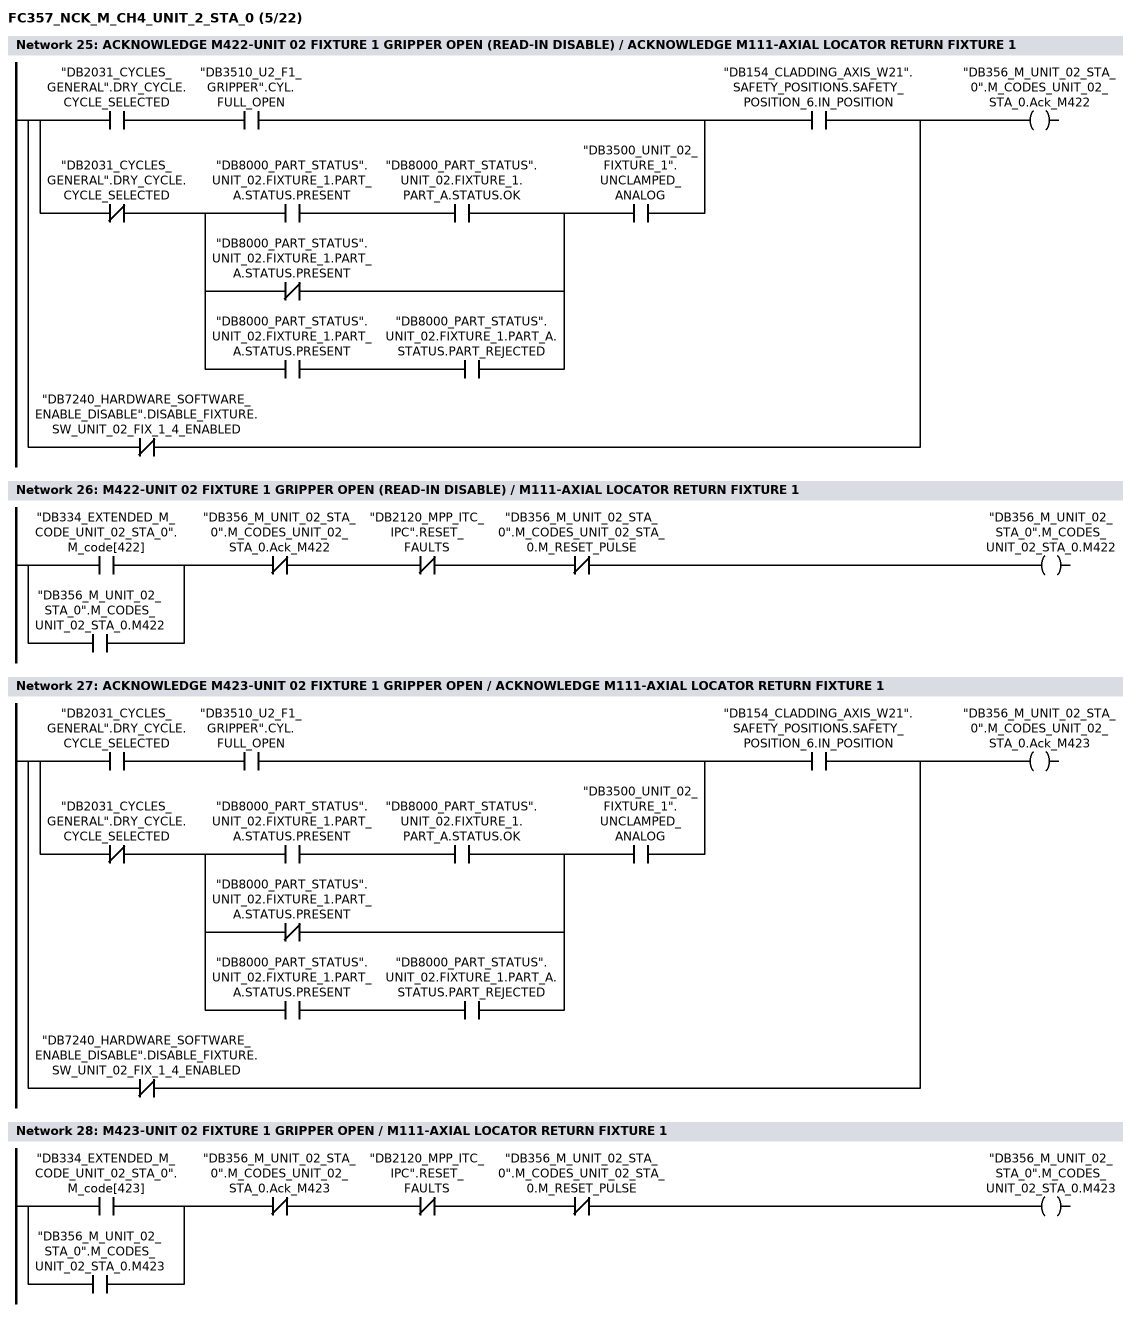
   RUNG wire#powerrail
      Contact( "DB2031_CYCLES_GENERAL".DRY_CYCLE.CYCLE_SELECTED )
      Contact( "DB3510_U2_F1_GRIPPER".CYL.FULL_OPEN )
      wire#w1
      Contact( "DB154_CLADDING_AXIS_W21".SAFETY_POSITIONS.SAFETY_POSITION_6.IN_POSITION )
      wire#w4
      Coil( "DB356_M_UNIT_02_STA_0".M_CODES_UNIT_02_STA_0.Ack_M422 )
   END_RUNG
   RUNG wire#powerrail
      I_Contact( "DB2031_CYCLES_GENERAL".DRY_CYCLE.CYCLE_SELECTED )
      wire#w2
      Contact( "DB8000_PART_STATUS".UNIT_02.FIXTURE_1.PART_A.STATUS.PRESENT )
      Contact( "DB8000_PART_STATUS".UNIT_02.FIXTURE_1.PART_A.STATUS.OK )
      wire#w3
      Contact( "DB3500_UNIT_02_FIXTURE_1".UNCLAMPED_ANALOG )
   END_RUNG wire#w1
   RUNG wire#w2
      I_Contact( "DB8000_PART_STATUS".UNIT_02.FIXTURE_1.PART_A.STATUS.PRESENT )
   END_RUNG wire#w3
   RUNG wire#w2
      Contact( "DB8000_PART_STATUS".UNIT_02.FIXTURE_1.PART_A.STATUS.PRESENT )
      Contact( "DB8000_PART_STATUS".UNIT_02.FIXTURE_1.PART_A.STATUS.PART_REJECTED )
   END_RUNG wire#w3
   RUNG wire#powerrail
      I_Contact( "DB7240_HARDWARE_SOFTWARE_ENABLE_DISABLE".DISABLE_FIXTURE.SW_UNIT_02_FIX_1_4_ENABLED )
   END_RUNG wire#w4
   // the same network as SCL:
   "DB356_M_UNIT_02_STA_0".M_CODES_UNIT_02_STA_0.Ack_M422 := ((("DB2031_CYCLES_GENERAL".DRY_CYCLE.CYCLE_SELECTED AND "DB3510_U2_F1_GRIPPER".CYL.FULL_OPEN) OR (NOT "DB2031_CYCLES_GENERAL".DRY_CYCLE.CYCLE_SELECTED AND (("DB8000_PART_STATUS".UNIT_02.FIXTURE_1.PART_A.STATUS.PRESENT AND "DB8000_PART_STATUS".UNIT_02.FIXTURE_1.PART_A.STATUS.OK) OR NOT "DB8000_PART_STATUS".UNIT_02.FIXTURE_1.PART_A.STATUS.PRESENT OR ("DB8000_PART_STATUS".UNIT_02.FIXTURE_1.PART_A.STATUS.PRESENT AND "DB8000_PART_STATUS".UNIT_02.FIXTURE_1.PART_A.STATUS.PART_REJECTED)) AND "DB3500_UNIT_02_FIXTURE_1".UNCLAMPED_ANALOG)) AND "DB154_CLADDING_AXIS_W21".SAFETY_POSITIONS.SAFETY_POSITION_6.IN_POSITION) OR NOT "DB7240_HARDWARE_SOFTWARE_ENABLE_DISABLE".DISABLE_FIXTURE.SW_UNIT_02_FIX_1_4_ENABLED;
END_REGION

REGION Network 26: M422-UNIT 02 FIXTURE 1 GRIPPER OPEN (READ-IN DISABLE) / M111-AXIAL LOCATOR RETURN FIXTURE 1
   RUNG wire#powerrail
      Contact( "DB334_EXTENDED_M_CODE_UNIT_02_STA_0".M_code[422] )
      wire#w1
      I_Contact( "DB356_M_UNIT_02_STA_0".M_CODES_UNIT_02_STA_0.Ack_M422 )
      I_Contact( "DB2120_MPP_ITC_IPC".RESET_FAULTS )
      I_Contact( "DB356_M_UNIT_02_STA_0".M_CODES_UNIT_02_STA_0.M_RESET_PULSE )
      Coil( "DB356_M_UNIT_02_STA_0".M_CODES_UNIT_02_STA_0.M422 )
   END_RUNG
   RUNG wire#powerrail
      Contact( "DB356_M_UNIT_02_STA_0".M_CODES_UNIT_02_STA_0.M422 )
   END_RUNG wire#w1
   // the same network as SCL:
   "DB356_M_UNIT_02_STA_0".M_CODES_UNIT_02_STA_0.M422 := ("DB334_EXTENDED_M_CODE_UNIT_02_STA_0".M_code[422] OR "DB356_M_UNIT_02_STA_0".M_CODES_UNIT_02_STA_0.M422) AND NOT "DB356_M_UNIT_02_STA_0".M_CODES_UNIT_02_STA_0.Ack_M422 AND NOT "DB2120_MPP_ITC_IPC".RESET_FAULTS AND NOT "DB356_M_UNIT_02_STA_0".M_CODES_UNIT_02_STA_0.M_RESET_PULSE;
END_REGION

REGION Network 27: ACKNOWLEDGE M423-UNIT 02 FIXTURE 1 GRIPPER OPEN / ACKNOWLEDGE M111-AXIAL LOCATOR RETURN FIXTURE 1
   RUNG wire#powerrail
      Contact( "DB2031_CYCLES_GENERAL".DRY_CYCLE.CYCLE_SELECTED )
      Contact( "DB3510_U2_F1_GRIPPER".CYL.FULL_OPEN )
      wire#w1
      Contact( "DB154_CLADDING_AXIS_W21".SAFETY_POSITIONS.SAFETY_POSITION_6.IN_POSITION )
      wire#w4
      Coil( "DB356_M_UNIT_02_STA_0".M_CODES_UNIT_02_STA_0.Ack_M423 )
   END_RUNG
   RUNG wire#powerrail
      I_Contact( "DB2031_CYCLES_GENERAL".DRY_CYCLE.CYCLE_SELECTED )
      wire#w2
      Contact( "DB8000_PART_STATUS".UNIT_02.FIXTURE_1.PART_A.STATUS.PRESENT )
      Contact( "DB8000_PART_STATUS".UNIT_02.FIXTURE_1.PART_A.STATUS.OK )
      wire#w3
      Contact( "DB3500_UNIT_02_FIXTURE_1".UNCLAMPED_ANALOG )
   END_RUNG wire#w1
   RUNG wire#w2
      I_Contact( "DB8000_PART_STATUS".UNIT_02.FIXTURE_1.PART_A.STATUS.PRESENT )
   END_RUNG wire#w3
   RUNG wire#w2
      Contact( "DB8000_PART_STATUS".UNIT_02.FIXTURE_1.PART_A.STATUS.PRESENT )
      Contact( "DB8000_PART_STATUS".UNIT_02.FIXTURE_1.PART_A.STATUS.PART_REJECTED )
   END_RUNG wire#w3
   RUNG wire#powerrail
      I_Contact( "DB7240_HARDWARE_SOFTWARE_ENABLE_DISABLE".DISABLE_FIXTURE.SW_UNIT_02_FIX_1_4_ENABLED )
   END_RUNG wire#w4
   // the same network as SCL:
   "DB356_M_UNIT_02_STA_0".M_CODES_UNIT_02_STA_0.Ack_M423 := ((("DB2031_CYCLES_GENERAL".DRY_CYCLE.CYCLE_SELECTED AND "DB3510_U2_F1_GRIPPER".CYL.FULL_OPEN) OR (NOT "DB2031_CYCLES_GENERAL".DRY_CYCLE.CYCLE_SELECTED AND (("DB8000_PART_STATUS".UNIT_02.FIXTURE_1.PART_A.STATUS.PRESENT AND "DB8000_PART_STATUS".UNIT_02.FIXTURE_1.PART_A.STATUS.OK) OR NOT "DB8000_PART_STATUS".UNIT_02.FIXTURE_1.PART_A.STATUS.PRESENT OR ("DB8000_PART_STATUS".UNIT_02.FIXTURE_1.PART_A.STATUS.PRESENT AND "DB8000_PART_STATUS".UNIT_02.FIXTURE_1.PART_A.STATUS.PART_REJECTED)) AND "DB3500_UNIT_02_FIXTURE_1".UNCLAMPED_ANALOG)) AND "DB154_CLADDING_AXIS_W21".SAFETY_POSITIONS.SAFETY_POSITION_6.IN_POSITION) OR NOT "DB7240_HARDWARE_SOFTWARE_ENABLE_DISABLE".DISABLE_FIXTURE.SW_UNIT_02_FIX_1_4_ENABLED;
END_REGION

REGION Network 28: M423-UNIT 02 FIXTURE 1 GRIPPER OPEN / M111-AXIAL LOCATOR RETURN FIXTURE 1
   RUNG wire#powerrail
      Contact( "DB334_EXTENDED_M_CODE_UNIT_02_STA_0".M_code[423] )
      wire#w1
      I_Contact( "DB356_M_UNIT_02_STA_0".M_CODES_UNIT_02_STA_0.Ack_M423 )
      I_Contact( "DB2120_MPP_ITC_IPC".RESET_FAULTS )
      I_Contact( "DB356_M_UNIT_02_STA_0".M_CODES_UNIT_02_STA_0.M_RESET_PULSE )
      Coil( "DB356_M_UNIT_02_STA_0".M_CODES_UNIT_02_STA_0.M423 )
   END_RUNG
   RUNG wire#powerrail
      Contact( "DB356_M_UNIT_02_STA_0".M_CODES_UNIT_02_STA_0.M423 )
   END_RUNG wire#w1
   // the same network as SCL:
   "DB356_M_UNIT_02_STA_0".M_CODES_UNIT_02_STA_0.M423 := ("DB334_EXTENDED_M_CODE_UNIT_02_STA_0".M_code[423] OR "DB356_M_UNIT_02_STA_0".M_CODES_UNIT_02_STA_0.M423) AND NOT "DB356_M_UNIT_02_STA_0".M_CODES_UNIT_02_STA_0.Ack_M423 AND NOT "DB2120_MPP_ITC_IPC".RESET_FAULTS AND NOT "DB356_M_UNIT_02_STA_0".M_CODES_UNIT_02_STA_0.M_RESET_PULSE;
END_REGION

REGION Network 29: ACKNOWLEDGE M424-UNIT 02 FIXTURE 1 GRIPPER RELEASE PRESSURE (READ-IN DISABLE) / ACKNOWLEDGE M112-AXIAL LOCATOR RELAX FIXTURE 1
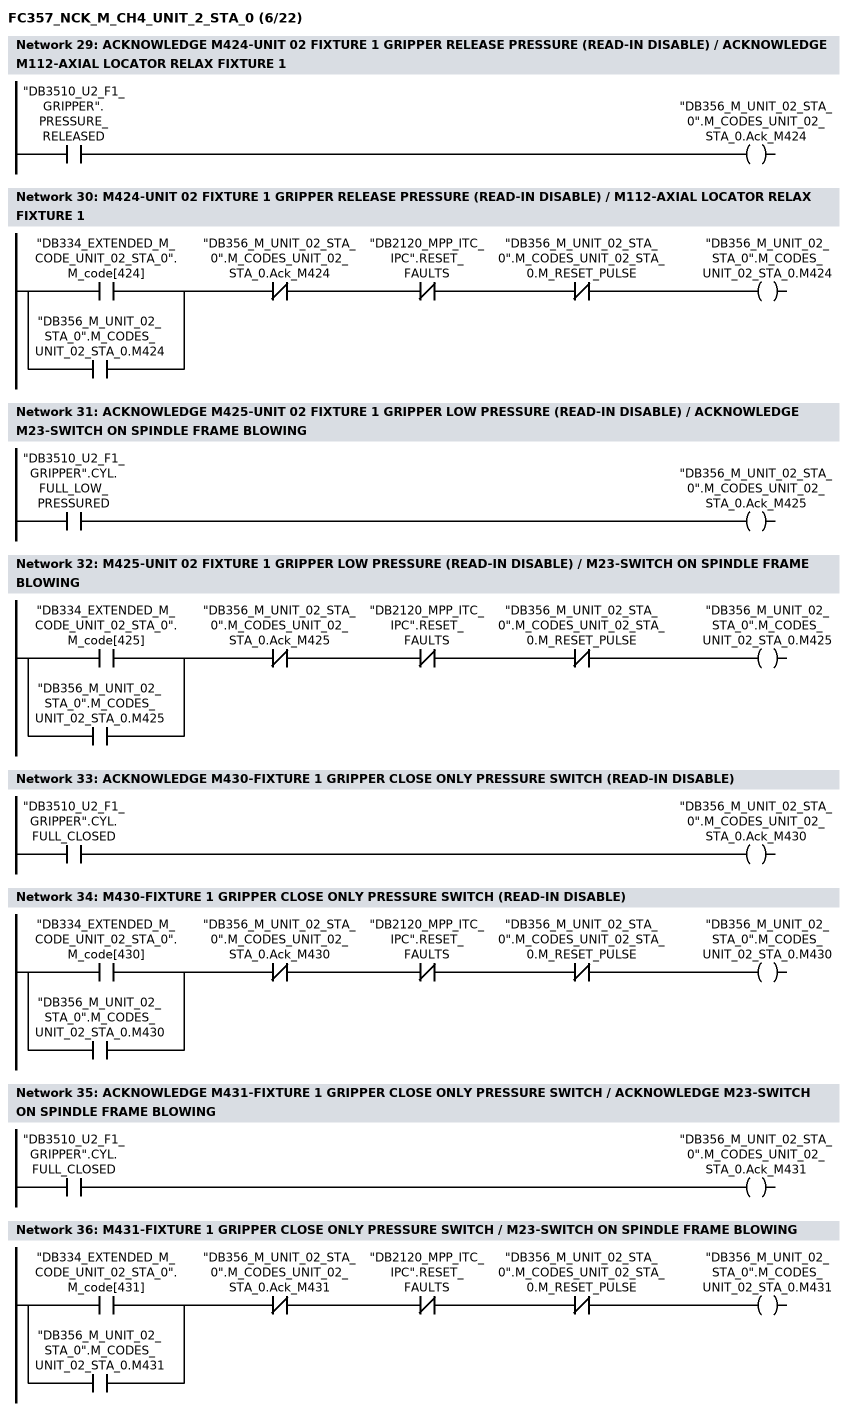
   RUNG wire#powerrail
      Contact( "DB3510_U2_F1_GRIPPER".PRESSURE_RELEASED )
      Coil( "DB356_M_UNIT_02_STA_0".M_CODES_UNIT_02_STA_0.Ack_M424 )
   END_RUNG
   // the same network as SCL:
   "DB356_M_UNIT_02_STA_0".M_CODES_UNIT_02_STA_0.Ack_M424 := "DB3510_U2_F1_GRIPPER".PRESSURE_RELEASED;
END_REGION

REGION Network 30: M424-UNIT 02 FIXTURE 1 GRIPPER RELEASE PRESSURE (READ-IN DISABLE) / M112-AXIAL LOCATOR RELAX FIXTURE 1
   RUNG wire#powerrail
      Contact( "DB334_EXTENDED_M_CODE_UNIT_02_STA_0".M_code[424] )
      wire#w1
      I_Contact( "DB356_M_UNIT_02_STA_0".M_CODES_UNIT_02_STA_0.Ack_M424 )
      I_Contact( "DB2120_MPP_ITC_IPC".RESET_FAULTS )
      I_Contact( "DB356_M_UNIT_02_STA_0".M_CODES_UNIT_02_STA_0.M_RESET_PULSE )
      Coil( "DB356_M_UNIT_02_STA_0".M_CODES_UNIT_02_STA_0.M424 )
   END_RUNG
   RUNG wire#powerrail
      Contact( "DB356_M_UNIT_02_STA_0".M_CODES_UNIT_02_STA_0.M424 )
   END_RUNG wire#w1
   // the same network as SCL:
   "DB356_M_UNIT_02_STA_0".M_CODES_UNIT_02_STA_0.M424 := ("DB334_EXTENDED_M_CODE_UNIT_02_STA_0".M_code[424] OR "DB356_M_UNIT_02_STA_0".M_CODES_UNIT_02_STA_0.M424) AND NOT "DB356_M_UNIT_02_STA_0".M_CODES_UNIT_02_STA_0.Ack_M424 AND NOT "DB2120_MPP_ITC_IPC".RESET_FAULTS AND NOT "DB356_M_UNIT_02_STA_0".M_CODES_UNIT_02_STA_0.M_RESET_PULSE;
END_REGION

REGION Network 31: ACKNOWLEDGE M425-UNIT 02 FIXTURE 1 GRIPPER LOW PRESSURE (READ-IN DISABLE) / ACKNOWLEDGE M23-SWITCH ON SPINDLE FRAME BLOWING
   RUNG wire#powerrail
      Contact( "DB3510_U2_F1_GRIPPER".CYL.FULL_LOW_PRESSURED )
      Coil( "DB356_M_UNIT_02_STA_0".M_CODES_UNIT_02_STA_0.Ack_M425 )
   END_RUNG
   // the same network as SCL:
   "DB356_M_UNIT_02_STA_0".M_CODES_UNIT_02_STA_0.Ack_M425 := "DB3510_U2_F1_GRIPPER".CYL.FULL_LOW_PRESSURED;
END_REGION

REGION Network 32: M425-UNIT 02 FIXTURE 1 GRIPPER LOW PRESSURE (READ-IN DISABLE) / M23-SWITCH ON SPINDLE FRAME BLOWING
   RUNG wire#powerrail
      Contact( "DB334_EXTENDED_M_CODE_UNIT_02_STA_0".M_code[425] )
      wire#w1
      I_Contact( "DB356_M_UNIT_02_STA_0".M_CODES_UNIT_02_STA_0.Ack_M425 )
      I_Contact( "DB2120_MPP_ITC_IPC".RESET_FAULTS )
      I_Contact( "DB356_M_UNIT_02_STA_0".M_CODES_UNIT_02_STA_0.M_RESET_PULSE )
      Coil( "DB356_M_UNIT_02_STA_0".M_CODES_UNIT_02_STA_0.M425 )
   END_RUNG
   RUNG wire#powerrail
      Contact( "DB356_M_UNIT_02_STA_0".M_CODES_UNIT_02_STA_0.M425 )
   END_RUNG wire#w1
   // the same network as SCL:
   "DB356_M_UNIT_02_STA_0".M_CODES_UNIT_02_STA_0.M425 := ("DB334_EXTENDED_M_CODE_UNIT_02_STA_0".M_code[425] OR "DB356_M_UNIT_02_STA_0".M_CODES_UNIT_02_STA_0.M425) AND NOT "DB356_M_UNIT_02_STA_0".M_CODES_UNIT_02_STA_0.Ack_M425 AND NOT "DB2120_MPP_ITC_IPC".RESET_FAULTS AND NOT "DB356_M_UNIT_02_STA_0".M_CODES_UNIT_02_STA_0.M_RESET_PULSE;
END_REGION

REGION Network 33: ACKNOWLEDGE M430-FIXTURE 1 GRIPPER CLOSE ONLY PRESSURE SWITCH (READ-IN DISABLE)
   RUNG wire#powerrail
      Contact( "DB3510_U2_F1_GRIPPER".CYL.FULL_CLOSED )
      Coil( "DB356_M_UNIT_02_STA_0".M_CODES_UNIT_02_STA_0.Ack_M430 )
   END_RUNG
   // the same network as SCL:
   "DB356_M_UNIT_02_STA_0".M_CODES_UNIT_02_STA_0.Ack_M430 := "DB3510_U2_F1_GRIPPER".CYL.FULL_CLOSED;
END_REGION

REGION Network 34: M430-FIXTURE 1 GRIPPER CLOSE ONLY PRESSURE SWITCH (READ-IN DISABLE)
   RUNG wire#powerrail
      Contact( "DB334_EXTENDED_M_CODE_UNIT_02_STA_0".M_code[430] )
      wire#w1
      I_Contact( "DB356_M_UNIT_02_STA_0".M_CODES_UNIT_02_STA_0.Ack_M430 )
      I_Contact( "DB2120_MPP_ITC_IPC".RESET_FAULTS )
      I_Contact( "DB356_M_UNIT_02_STA_0".M_CODES_UNIT_02_STA_0.M_RESET_PULSE )
      Coil( "DB356_M_UNIT_02_STA_0".M_CODES_UNIT_02_STA_0.M430 )
   END_RUNG
   RUNG wire#powerrail
      Contact( "DB356_M_UNIT_02_STA_0".M_CODES_UNIT_02_STA_0.M430 )
   END_RUNG wire#w1
   // the same network as SCL:
   "DB356_M_UNIT_02_STA_0".M_CODES_UNIT_02_STA_0.M430 := ("DB334_EXTENDED_M_CODE_UNIT_02_STA_0".M_code[430] OR "DB356_M_UNIT_02_STA_0".M_CODES_UNIT_02_STA_0.M430) AND NOT "DB356_M_UNIT_02_STA_0".M_CODES_UNIT_02_STA_0.Ack_M430 AND NOT "DB2120_MPP_ITC_IPC".RESET_FAULTS AND NOT "DB356_M_UNIT_02_STA_0".M_CODES_UNIT_02_STA_0.M_RESET_PULSE;
END_REGION

REGION Network 35: ACKNOWLEDGE M431-FIXTURE 1 GRIPPER CLOSE ONLY PRESSURE SWITCH / ACKNOWLEDGE M23-SWITCH ON SPINDLE FRAME BLOWING
   RUNG wire#powerrail
      Contact( "DB3510_U2_F1_GRIPPER".CYL.FULL_CLOSED )
      Coil( "DB356_M_UNIT_02_STA_0".M_CODES_UNIT_02_STA_0.Ack_M431 )
   END_RUNG
   // the same network as SCL:
   "DB356_M_UNIT_02_STA_0".M_CODES_UNIT_02_STA_0.Ack_M431 := "DB3510_U2_F1_GRIPPER".CYL.FULL_CLOSED;
END_REGION

REGION Network 36: M431-FIXTURE 1 GRIPPER CLOSE ONLY PRESSURE SWITCH / M23-SWITCH ON SPINDLE FRAME BLOWING
   RUNG wire#powerrail
      Contact( "DB334_EXTENDED_M_CODE_UNIT_02_STA_0".M_code[431] )
      wire#w1
      I_Contact( "DB356_M_UNIT_02_STA_0".M_CODES_UNIT_02_STA_0.Ack_M431 )
      I_Contact( "DB2120_MPP_ITC_IPC".RESET_FAULTS )
      I_Contact( "DB356_M_UNIT_02_STA_0".M_CODES_UNIT_02_STA_0.M_RESET_PULSE )
      Coil( "DB356_M_UNIT_02_STA_0".M_CODES_UNIT_02_STA_0.M431 )
   END_RUNG
   RUNG wire#powerrail
      Contact( "DB356_M_UNIT_02_STA_0".M_CODES_UNIT_02_STA_0.M431 )
   END_RUNG wire#w1
   // the same network as SCL:
   "DB356_M_UNIT_02_STA_0".M_CODES_UNIT_02_STA_0.M431 := ("DB334_EXTENDED_M_CODE_UNIT_02_STA_0".M_code[431] OR "DB356_M_UNIT_02_STA_0".M_CODES_UNIT_02_STA_0.M431) AND NOT "DB356_M_UNIT_02_STA_0".M_CODES_UNIT_02_STA_0.Ack_M431 AND NOT "DB2120_MPP_ITC_IPC".RESET_FAULTS AND NOT "DB356_M_UNIT_02_STA_0".M_CODES_UNIT_02_STA_0.M_RESET_PULSE;
END_REGION

REGION Network 37: ACKNOWLEDGE M432-FIXTURE 1 GRIPPER OPEN ONLY PRESSURE SWITCH (READ-IN DISABLE) / ACKNOWLEDGE M111-AXIAL LOCATOR RETURN FIXTURE 1
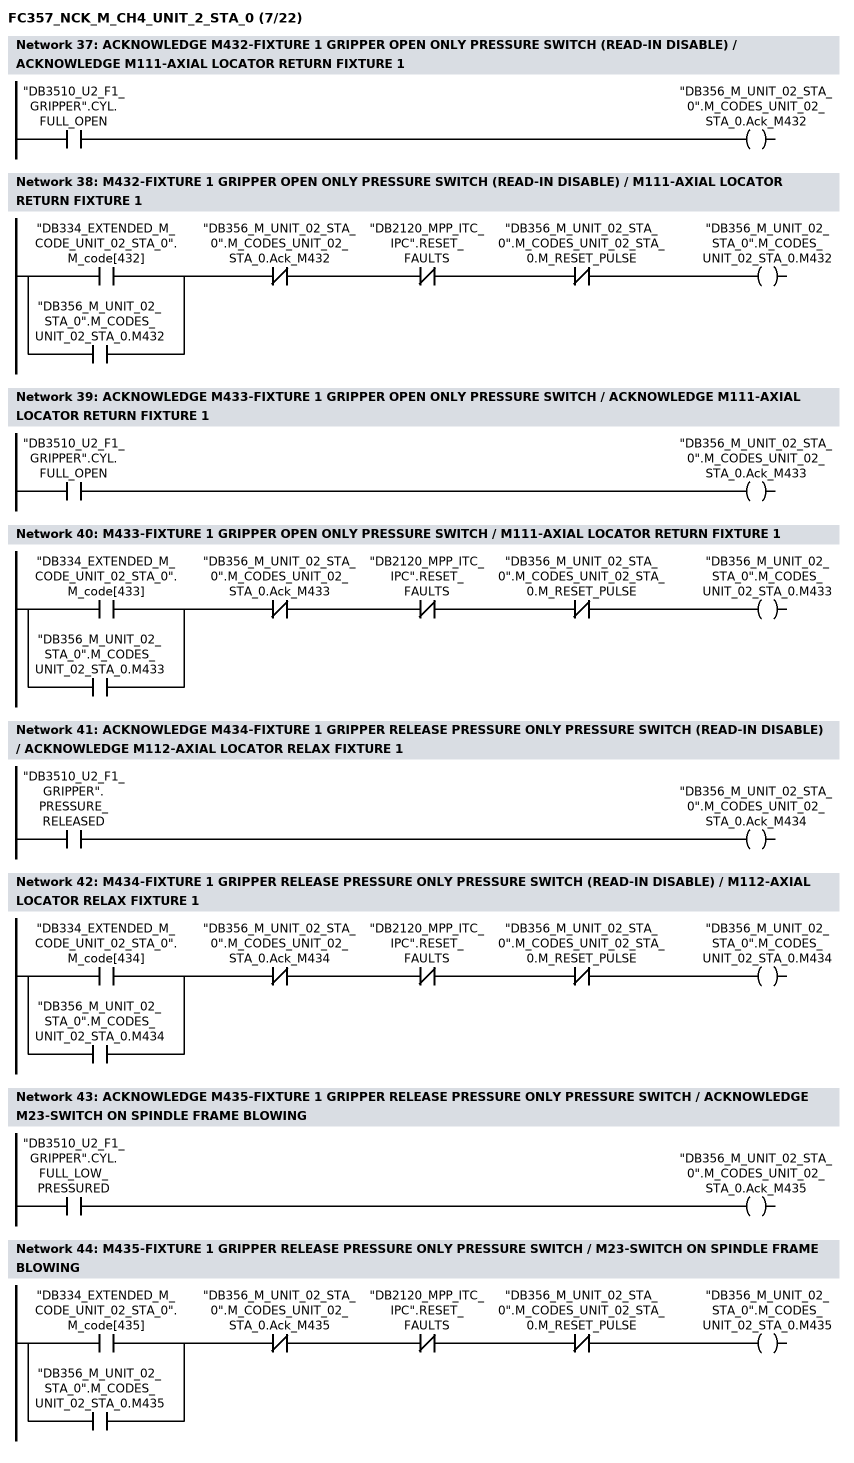
   RUNG wire#powerrail
      Contact( "DB3510_U2_F1_GRIPPER".CYL.FULL_OPEN )
      Coil( "DB356_M_UNIT_02_STA_0".M_CODES_UNIT_02_STA_0.Ack_M432 )
   END_RUNG
   // the same network as SCL:
   "DB356_M_UNIT_02_STA_0".M_CODES_UNIT_02_STA_0.Ack_M432 := "DB3510_U2_F1_GRIPPER".CYL.FULL_OPEN;
END_REGION

REGION Network 38: M432-FIXTURE 1 GRIPPER OPEN ONLY PRESSURE SWITCH (READ-IN DISABLE) / M111-AXIAL LOCATOR RETURN FIXTURE 1
   RUNG wire#powerrail
      Contact( "DB334_EXTENDED_M_CODE_UNIT_02_STA_0".M_code[432] )
      wire#w1
      I_Contact( "DB356_M_UNIT_02_STA_0".M_CODES_UNIT_02_STA_0.Ack_M432 )
      I_Contact( "DB2120_MPP_ITC_IPC".RESET_FAULTS )
      I_Contact( "DB356_M_UNIT_02_STA_0".M_CODES_UNIT_02_STA_0.M_RESET_PULSE )
      Coil( "DB356_M_UNIT_02_STA_0".M_CODES_UNIT_02_STA_0.M432 )
   END_RUNG
   RUNG wire#powerrail
      Contact( "DB356_M_UNIT_02_STA_0".M_CODES_UNIT_02_STA_0.M432 )
   END_RUNG wire#w1
   // the same network as SCL:
   "DB356_M_UNIT_02_STA_0".M_CODES_UNIT_02_STA_0.M432 := ("DB334_EXTENDED_M_CODE_UNIT_02_STA_0".M_code[432] OR "DB356_M_UNIT_02_STA_0".M_CODES_UNIT_02_STA_0.M432) AND NOT "DB356_M_UNIT_02_STA_0".M_CODES_UNIT_02_STA_0.Ack_M432 AND NOT "DB2120_MPP_ITC_IPC".RESET_FAULTS AND NOT "DB356_M_UNIT_02_STA_0".M_CODES_UNIT_02_STA_0.M_RESET_PULSE;
END_REGION

REGION Network 39: ACKNOWLEDGE M433-FIXTURE 1 GRIPPER OPEN ONLY PRESSURE SWITCH / ACKNOWLEDGE M111-AXIAL LOCATOR RETURN FIXTURE 1
   RUNG wire#powerrail
      Contact( "DB3510_U2_F1_GRIPPER".CYL.FULL_OPEN )
      Coil( "DB356_M_UNIT_02_STA_0".M_CODES_UNIT_02_STA_0.Ack_M433 )
   END_RUNG
   // the same network as SCL:
   "DB356_M_UNIT_02_STA_0".M_CODES_UNIT_02_STA_0.Ack_M433 := "DB3510_U2_F1_GRIPPER".CYL.FULL_OPEN;
END_REGION

REGION Network 40: M433-FIXTURE 1 GRIPPER OPEN ONLY PRESSURE SWITCH / M111-AXIAL LOCATOR RETURN FIXTURE 1
   RUNG wire#powerrail
      Contact( "DB334_EXTENDED_M_CODE_UNIT_02_STA_0".M_code[433] )
      wire#w1
      I_Contact( "DB356_M_UNIT_02_STA_0".M_CODES_UNIT_02_STA_0.Ack_M433 )
      I_Contact( "DB2120_MPP_ITC_IPC".RESET_FAULTS )
      I_Contact( "DB356_M_UNIT_02_STA_0".M_CODES_UNIT_02_STA_0.M_RESET_PULSE )
      Coil( "DB356_M_UNIT_02_STA_0".M_CODES_UNIT_02_STA_0.M433 )
   END_RUNG
   RUNG wire#powerrail
      Contact( "DB356_M_UNIT_02_STA_0".M_CODES_UNIT_02_STA_0.M433 )
   END_RUNG wire#w1
   // the same network as SCL:
   "DB356_M_UNIT_02_STA_0".M_CODES_UNIT_02_STA_0.M433 := ("DB334_EXTENDED_M_CODE_UNIT_02_STA_0".M_code[433] OR "DB356_M_UNIT_02_STA_0".M_CODES_UNIT_02_STA_0.M433) AND NOT "DB356_M_UNIT_02_STA_0".M_CODES_UNIT_02_STA_0.Ack_M433 AND NOT "DB2120_MPP_ITC_IPC".RESET_FAULTS AND NOT "DB356_M_UNIT_02_STA_0".M_CODES_UNIT_02_STA_0.M_RESET_PULSE;
END_REGION

REGION Network 41: ACKNOWLEDGE M434-FIXTURE 1 GRIPPER RELEASE PRESSURE ONLY PRESSURE SWITCH (READ-IN DISABLE) / ACKNOWLEDGE M112-AXIAL LOCATOR RELAX FIXTURE 1
   RUNG wire#powerrail
      Contact( "DB3510_U2_F1_GRIPPER".PRESSURE_RELEASED )
      Coil( "DB356_M_UNIT_02_STA_0".M_CODES_UNIT_02_STA_0.Ack_M434 )
   END_RUNG
   // the same network as SCL:
   "DB356_M_UNIT_02_STA_0".M_CODES_UNIT_02_STA_0.Ack_M434 := "DB3510_U2_F1_GRIPPER".PRESSURE_RELEASED;
END_REGION

REGION Network 42: M434-FIXTURE 1 GRIPPER RELEASE PRESSURE ONLY PRESSURE SWITCH (READ-IN DISABLE) / M112-AXIAL LOCATOR RELAX FIXTURE 1
   RUNG wire#powerrail
      Contact( "DB334_EXTENDED_M_CODE_UNIT_02_STA_0".M_code[434] )
      wire#w1
      I_Contact( "DB356_M_UNIT_02_STA_0".M_CODES_UNIT_02_STA_0.Ack_M434 )
      I_Contact( "DB2120_MPP_ITC_IPC".RESET_FAULTS )
      I_Contact( "DB356_M_UNIT_02_STA_0".M_CODES_UNIT_02_STA_0.M_RESET_PULSE )
      Coil( "DB356_M_UNIT_02_STA_0".M_CODES_UNIT_02_STA_0.M434 )
   END_RUNG
   RUNG wire#powerrail
      Contact( "DB356_M_UNIT_02_STA_0".M_CODES_UNIT_02_STA_0.M434 )
   END_RUNG wire#w1
   // the same network as SCL:
   "DB356_M_UNIT_02_STA_0".M_CODES_UNIT_02_STA_0.M434 := ("DB334_EXTENDED_M_CODE_UNIT_02_STA_0".M_code[434] OR "DB356_M_UNIT_02_STA_0".M_CODES_UNIT_02_STA_0.M434) AND NOT "DB356_M_UNIT_02_STA_0".M_CODES_UNIT_02_STA_0.Ack_M434 AND NOT "DB2120_MPP_ITC_IPC".RESET_FAULTS AND NOT "DB356_M_UNIT_02_STA_0".M_CODES_UNIT_02_STA_0.M_RESET_PULSE;
END_REGION

REGION Network 43: ACKNOWLEDGE M435-FIXTURE 1 GRIPPER RELEASE PRESSURE ONLY PRESSURE SWITCH / ACKNOWLEDGE M23-SWITCH ON SPINDLE FRAME BLOWING
   RUNG wire#powerrail
      Contact( "DB3510_U2_F1_GRIPPER".CYL.FULL_LOW_PRESSURED )
      Coil( "DB356_M_UNIT_02_STA_0".M_CODES_UNIT_02_STA_0.Ack_M435 )
   END_RUNG
   // the same network as SCL:
   "DB356_M_UNIT_02_STA_0".M_CODES_UNIT_02_STA_0.Ack_M435 := "DB3510_U2_F1_GRIPPER".CYL.FULL_LOW_PRESSURED;
END_REGION

REGION Network 44: M435-FIXTURE 1 GRIPPER RELEASE PRESSURE ONLY PRESSURE SWITCH / M23-SWITCH ON SPINDLE FRAME BLOWING
   RUNG wire#powerrail
      Contact( "DB334_EXTENDED_M_CODE_UNIT_02_STA_0".M_code[435] )
      wire#w1
      I_Contact( "DB356_M_UNIT_02_STA_0".M_CODES_UNIT_02_STA_0.Ack_M435 )
      I_Contact( "DB2120_MPP_ITC_IPC".RESET_FAULTS )
      I_Contact( "DB356_M_UNIT_02_STA_0".M_CODES_UNIT_02_STA_0.M_RESET_PULSE )
      Coil( "DB356_M_UNIT_02_STA_0".M_CODES_UNIT_02_STA_0.M435 )
   END_RUNG
   RUNG wire#powerrail
      Contact( "DB356_M_UNIT_02_STA_0".M_CODES_UNIT_02_STA_0.M435 )
   END_RUNG wire#w1
   // the same network as SCL:
   "DB356_M_UNIT_02_STA_0".M_CODES_UNIT_02_STA_0.M435 := ("DB334_EXTENDED_M_CODE_UNIT_02_STA_0".M_code[435] OR "DB356_M_UNIT_02_STA_0".M_CODES_UNIT_02_STA_0.M435) AND NOT "DB356_M_UNIT_02_STA_0".M_CODES_UNIT_02_STA_0.Ack_M435 AND NOT "DB2120_MPP_ITC_IPC".RESET_FAULTS AND NOT "DB356_M_UNIT_02_STA_0".M_CODES_UNIT_02_STA_0.M_RESET_PULSE;
END_REGION

REGION Network 45: ACKNOWLEDGE M500-UNIT 02 FIXTURE 2 CLAMP SEQUENCE (READ-IN DISABLE) / ACKNOWLEDGE M100-CLAMP SEQUENCE FIXTURE 1
   // NOTE: WHEN THERE IS NOT INDEXING TABLE AVAILABLE IN THE MACHINE DELETE 
   // DB2171.DBX5.0 AND DB2171.DBX2.0
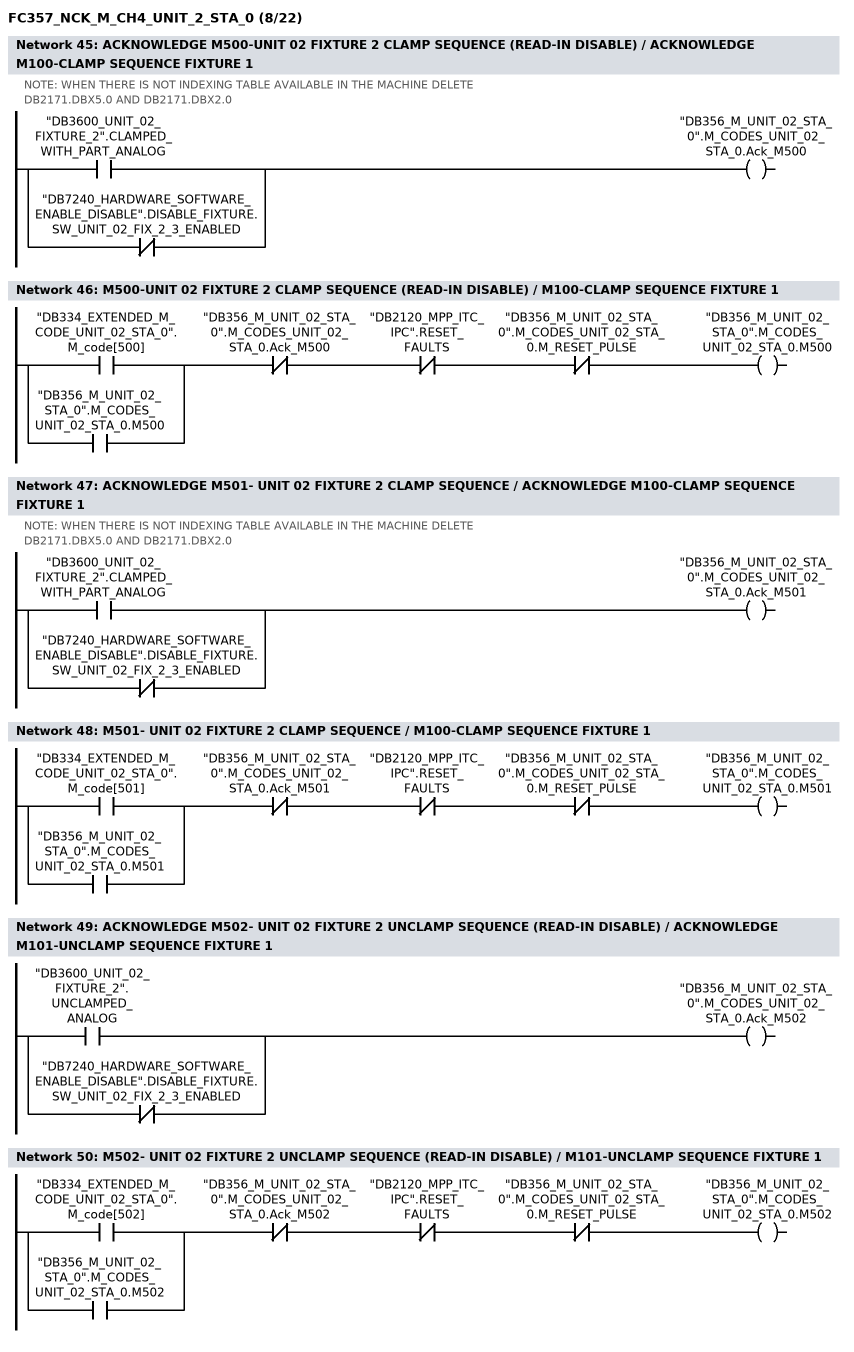
   RUNG wire#powerrail
      Contact( "DB3600_UNIT_02_FIXTURE_2".CLAMPED_WITH_PART_ANALOG )
      wire#w1
      Coil( "DB356_M_UNIT_02_STA_0".M_CODES_UNIT_02_STA_0.Ack_M500 )
   END_RUNG
   RUNG wire#powerrail
      I_Contact( "DB7240_HARDWARE_SOFTWARE_ENABLE_DISABLE".DISABLE_FIXTURE.SW_UNIT_02_FIX_2_3_ENABLED )
   END_RUNG wire#w1
   // the same network as SCL:
   "DB356_M_UNIT_02_STA_0".M_CODES_UNIT_02_STA_0.Ack_M500 := "DB3600_UNIT_02_FIXTURE_2".CLAMPED_WITH_PART_ANALOG OR NOT "DB7240_HARDWARE_SOFTWARE_ENABLE_DISABLE".DISABLE_FIXTURE.SW_UNIT_02_FIX_2_3_ENABLED;
END_REGION

REGION Network 46: M500-UNIT 02 FIXTURE 2 CLAMP SEQUENCE (READ-IN DISABLE) / M100-CLAMP SEQUENCE FIXTURE 1
   RUNG wire#powerrail
      Contact( "DB334_EXTENDED_M_CODE_UNIT_02_STA_0".M_code[500] )
      wire#w1
      I_Contact( "DB356_M_UNIT_02_STA_0".M_CODES_UNIT_02_STA_0.Ack_M500 )
      I_Contact( "DB2120_MPP_ITC_IPC".RESET_FAULTS )
      I_Contact( "DB356_M_UNIT_02_STA_0".M_CODES_UNIT_02_STA_0.M_RESET_PULSE )
      Coil( "DB356_M_UNIT_02_STA_0".M_CODES_UNIT_02_STA_0.M500 )
   END_RUNG
   RUNG wire#powerrail
      Contact( "DB356_M_UNIT_02_STA_0".M_CODES_UNIT_02_STA_0.M500 )
   END_RUNG wire#w1
   // the same network as SCL:
   "DB356_M_UNIT_02_STA_0".M_CODES_UNIT_02_STA_0.M500 := ("DB334_EXTENDED_M_CODE_UNIT_02_STA_0".M_code[500] OR "DB356_M_UNIT_02_STA_0".M_CODES_UNIT_02_STA_0.M500) AND NOT "DB356_M_UNIT_02_STA_0".M_CODES_UNIT_02_STA_0.Ack_M500 AND NOT "DB2120_MPP_ITC_IPC".RESET_FAULTS AND NOT "DB356_M_UNIT_02_STA_0".M_CODES_UNIT_02_STA_0.M_RESET_PULSE;
END_REGION

REGION Network 47: ACKNOWLEDGE M501- UNIT 02 FIXTURE 2 CLAMP SEQUENCE / ACKNOWLEDGE M100-CLAMP SEQUENCE FIXTURE 1
   // NOTE: WHEN THERE IS NOT INDEXING TABLE AVAILABLE IN THE MACHINE DELETE 
   // DB2171.DBX5.0 AND DB2171.DBX2.0
   RUNG wire#powerrail
      Contact( "DB3600_UNIT_02_FIXTURE_2".CLAMPED_WITH_PART_ANALOG )
      wire#w1
      Coil( "DB356_M_UNIT_02_STA_0".M_CODES_UNIT_02_STA_0.Ack_M501 )
   END_RUNG
   RUNG wire#powerrail
      I_Contact( "DB7240_HARDWARE_SOFTWARE_ENABLE_DISABLE".DISABLE_FIXTURE.SW_UNIT_02_FIX_2_3_ENABLED )
   END_RUNG wire#w1
   // the same network as SCL:
   "DB356_M_UNIT_02_STA_0".M_CODES_UNIT_02_STA_0.Ack_M501 := "DB3600_UNIT_02_FIXTURE_2".CLAMPED_WITH_PART_ANALOG OR NOT "DB7240_HARDWARE_SOFTWARE_ENABLE_DISABLE".DISABLE_FIXTURE.SW_UNIT_02_FIX_2_3_ENABLED;
END_REGION

REGION Network 48: M501- UNIT 02 FIXTURE 2 CLAMP SEQUENCE / M100-CLAMP SEQUENCE FIXTURE 1
   RUNG wire#powerrail
      Contact( "DB334_EXTENDED_M_CODE_UNIT_02_STA_0".M_code[501] )
      wire#w1
      I_Contact( "DB356_M_UNIT_02_STA_0".M_CODES_UNIT_02_STA_0.Ack_M501 )
      I_Contact( "DB2120_MPP_ITC_IPC".RESET_FAULTS )
      I_Contact( "DB356_M_UNIT_02_STA_0".M_CODES_UNIT_02_STA_0.M_RESET_PULSE )
      Coil( "DB356_M_UNIT_02_STA_0".M_CODES_UNIT_02_STA_0.M501 )
   END_RUNG
   RUNG wire#powerrail
      Contact( "DB356_M_UNIT_02_STA_0".M_CODES_UNIT_02_STA_0.M501 )
   END_RUNG wire#w1
   // the same network as SCL:
   "DB356_M_UNIT_02_STA_0".M_CODES_UNIT_02_STA_0.M501 := ("DB334_EXTENDED_M_CODE_UNIT_02_STA_0".M_code[501] OR "DB356_M_UNIT_02_STA_0".M_CODES_UNIT_02_STA_0.M501) AND NOT "DB356_M_UNIT_02_STA_0".M_CODES_UNIT_02_STA_0.Ack_M501 AND NOT "DB2120_MPP_ITC_IPC".RESET_FAULTS AND NOT "DB356_M_UNIT_02_STA_0".M_CODES_UNIT_02_STA_0.M_RESET_PULSE;
END_REGION

REGION Network 49: ACKNOWLEDGE M502- UNIT 02 FIXTURE 2 UNCLAMP SEQUENCE (READ-IN DISABLE) / ACKNOWLEDGE M101-UNCLAMP SEQUENCE FIXTURE 1
   RUNG wire#powerrail
      Contact( "DB3600_UNIT_02_FIXTURE_2".UNCLAMPED_ANALOG )
      wire#w1
      Coil( "DB356_M_UNIT_02_STA_0".M_CODES_UNIT_02_STA_0.Ack_M502 )
   END_RUNG
   RUNG wire#powerrail
      I_Contact( "DB7240_HARDWARE_SOFTWARE_ENABLE_DISABLE".DISABLE_FIXTURE.SW_UNIT_02_FIX_2_3_ENABLED )
   END_RUNG wire#w1
   // the same network as SCL:
   "DB356_M_UNIT_02_STA_0".M_CODES_UNIT_02_STA_0.Ack_M502 := "DB3600_UNIT_02_FIXTURE_2".UNCLAMPED_ANALOG OR NOT "DB7240_HARDWARE_SOFTWARE_ENABLE_DISABLE".DISABLE_FIXTURE.SW_UNIT_02_FIX_2_3_ENABLED;
END_REGION

REGION Network 50: M502- UNIT 02 FIXTURE 2 UNCLAMP SEQUENCE (READ-IN DISABLE) / M101-UNCLAMP SEQUENCE FIXTURE 1
   RUNG wire#powerrail
      Contact( "DB334_EXTENDED_M_CODE_UNIT_02_STA_0".M_code[502] )
      wire#w1
      I_Contact( "DB356_M_UNIT_02_STA_0".M_CODES_UNIT_02_STA_0.Ack_M502 )
      I_Contact( "DB2120_MPP_ITC_IPC".RESET_FAULTS )
      I_Contact( "DB356_M_UNIT_02_STA_0".M_CODES_UNIT_02_STA_0.M_RESET_PULSE )
      Coil( "DB356_M_UNIT_02_STA_0".M_CODES_UNIT_02_STA_0.M502 )
   END_RUNG
   RUNG wire#powerrail
      Contact( "DB356_M_UNIT_02_STA_0".M_CODES_UNIT_02_STA_0.M502 )
   END_RUNG wire#w1
   // the same network as SCL:
   "DB356_M_UNIT_02_STA_0".M_CODES_UNIT_02_STA_0.M502 := ("DB334_EXTENDED_M_CODE_UNIT_02_STA_0".M_code[502] OR "DB356_M_UNIT_02_STA_0".M_CODES_UNIT_02_STA_0.M502) AND NOT "DB356_M_UNIT_02_STA_0".M_CODES_UNIT_02_STA_0.Ack_M502 AND NOT "DB2120_MPP_ITC_IPC".RESET_FAULTS AND NOT "DB356_M_UNIT_02_STA_0".M_CODES_UNIT_02_STA_0.M_RESET_PULSE;
END_REGION

REGION Network 51: ACKNOWLEDGE M503- UNIT 02 FIXTURE 2 UNCLAMP SEQUENCE / ACKNOWLEDGE M101-UNCLAMP SEQUENCE FIXTURE 1
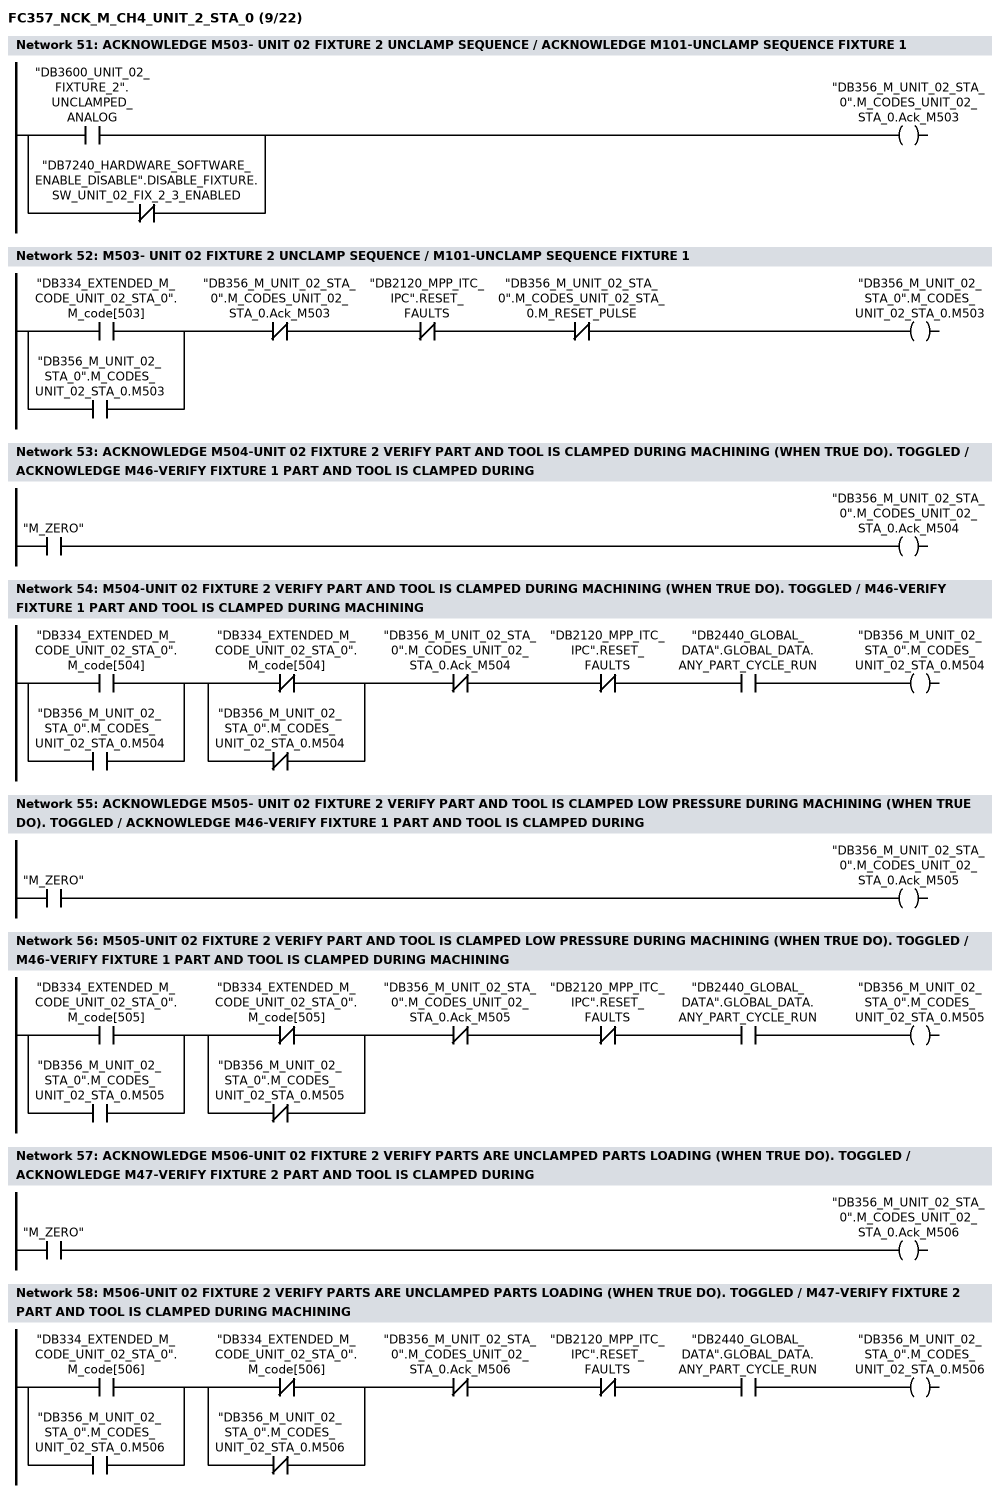
   RUNG wire#powerrail
      Contact( "DB3600_UNIT_02_FIXTURE_2".UNCLAMPED_ANALOG )
      wire#w1
      Coil( "DB356_M_UNIT_02_STA_0".M_CODES_UNIT_02_STA_0.Ack_M503 )
   END_RUNG
   RUNG wire#powerrail
      I_Contact( "DB7240_HARDWARE_SOFTWARE_ENABLE_DISABLE".DISABLE_FIXTURE.SW_UNIT_02_FIX_2_3_ENABLED )
   END_RUNG wire#w1
   // the same network as SCL:
   "DB356_M_UNIT_02_STA_0".M_CODES_UNIT_02_STA_0.Ack_M503 := "DB3600_UNIT_02_FIXTURE_2".UNCLAMPED_ANALOG OR NOT "DB7240_HARDWARE_SOFTWARE_ENABLE_DISABLE".DISABLE_FIXTURE.SW_UNIT_02_FIX_2_3_ENABLED;
END_REGION

REGION Network 52: M503- UNIT 02 FIXTURE 2 UNCLAMP SEQUENCE / M101-UNCLAMP SEQUENCE FIXTURE 1
   RUNG wire#powerrail
      Contact( "DB334_EXTENDED_M_CODE_UNIT_02_STA_0".M_code[503] )
      wire#w1
      I_Contact( "DB356_M_UNIT_02_STA_0".M_CODES_UNIT_02_STA_0.Ack_M503 )
      I_Contact( "DB2120_MPP_ITC_IPC".RESET_FAULTS )
      I_Contact( "DB356_M_UNIT_02_STA_0".M_CODES_UNIT_02_STA_0.M_RESET_PULSE )
      Coil( "DB356_M_UNIT_02_STA_0".M_CODES_UNIT_02_STA_0.M503 )
   END_RUNG
   RUNG wire#powerrail
      Contact( "DB356_M_UNIT_02_STA_0".M_CODES_UNIT_02_STA_0.M503 )
   END_RUNG wire#w1
   // the same network as SCL:
   "DB356_M_UNIT_02_STA_0".M_CODES_UNIT_02_STA_0.M503 := ("DB334_EXTENDED_M_CODE_UNIT_02_STA_0".M_code[503] OR "DB356_M_UNIT_02_STA_0".M_CODES_UNIT_02_STA_0.M503) AND NOT "DB356_M_UNIT_02_STA_0".M_CODES_UNIT_02_STA_0.Ack_M503 AND NOT "DB2120_MPP_ITC_IPC".RESET_FAULTS AND NOT "DB356_M_UNIT_02_STA_0".M_CODES_UNIT_02_STA_0.M_RESET_PULSE;
END_REGION

REGION Network 53: ACKNOWLEDGE M504-UNIT 02 FIXTURE 2 VERIFY PART AND TOOL IS CLAMPED DURING MACHINING (WHEN TRUE DO). TOGGLED / ACKNOWLEDGE M46-VERIFY FIXTURE 1 PART AND TOOL IS CLAMPED DURING
   RUNG wire#powerrail
      Contact( "M_ZERO" )
      Coil( "DB356_M_UNIT_02_STA_0".M_CODES_UNIT_02_STA_0.Ack_M504 )
   END_RUNG
   // the same network as SCL:
   "DB356_M_UNIT_02_STA_0".M_CODES_UNIT_02_STA_0.Ack_M504 := "M_ZERO";
END_REGION

REGION Network 54: M504-UNIT 02 FIXTURE 2 VERIFY PART AND TOOL IS CLAMPED DURING MACHINING (WHEN TRUE DO). TOGGLED / M46-VERIFY FIXTURE 1 PART AND TOOL IS CLAMPED DURING MACHINING
   RUNG wire#powerrail
      Contact( "DB334_EXTENDED_M_CODE_UNIT_02_STA_0".M_code[504] )
      wire#w1
      I_Contact( "DB334_EXTENDED_M_CODE_UNIT_02_STA_0".M_code[504] )
      wire#w2
      I_Contact( "DB356_M_UNIT_02_STA_0".M_CODES_UNIT_02_STA_0.Ack_M504 )
      I_Contact( "DB2120_MPP_ITC_IPC".RESET_FAULTS )
      Contact( "DB2440_GLOBAL_DATA".GLOBAL_DATA.ANY_PART_CYCLE_RUN )
      Coil( "DB356_M_UNIT_02_STA_0".M_CODES_UNIT_02_STA_0.M504 )
   END_RUNG
   RUNG wire#powerrail
      Contact( "DB356_M_UNIT_02_STA_0".M_CODES_UNIT_02_STA_0.M504 )
   END_RUNG wire#w1
   RUNG wire#w1
      I_Contact( "DB356_M_UNIT_02_STA_0".M_CODES_UNIT_02_STA_0.M504 )
   END_RUNG wire#w2
   // the same network as SCL:
   "DB356_M_UNIT_02_STA_0".M_CODES_UNIT_02_STA_0.M504 := ("DB334_EXTENDED_M_CODE_UNIT_02_STA_0".M_code[504] OR "DB356_M_UNIT_02_STA_0".M_CODES_UNIT_02_STA_0.M504) AND (NOT "DB334_EXTENDED_M_CODE_UNIT_02_STA_0".M_code[504] OR NOT "DB356_M_UNIT_02_STA_0".M_CODES_UNIT_02_STA_0.M504) AND NOT "DB356_M_UNIT_02_STA_0".M_CODES_UNIT_02_STA_0.Ack_M504 AND NOT "DB2120_MPP_ITC_IPC".RESET_FAULTS AND "DB2440_GLOBAL_DATA".GLOBAL_DATA.ANY_PART_CYCLE_RUN;
END_REGION

REGION Network 55: ACKNOWLEDGE M505- UNIT 02 FIXTURE 2 VERIFY PART AND TOOL IS CLAMPED LOW PRESSURE DURING MACHINING (WHEN TRUE DO). TOGGLED / ACKNOWLEDGE M46-VERIFY FIXTURE 1 PART AND TOOL IS CLAMPED DURING
   RUNG wire#powerrail
      Contact( "M_ZERO" )
      Coil( "DB356_M_UNIT_02_STA_0".M_CODES_UNIT_02_STA_0.Ack_M505 )
   END_RUNG
   // the same network as SCL:
   "DB356_M_UNIT_02_STA_0".M_CODES_UNIT_02_STA_0.Ack_M505 := "M_ZERO";
END_REGION

REGION Network 56: M505-UNIT 02 FIXTURE 2 VERIFY PART AND TOOL IS CLAMPED LOW PRESSURE DURING MACHINING (WHEN TRUE DO). TOGGLED / M46-VERIFY FIXTURE 1 PART AND TOOL IS CLAMPED DURING MACHINING
   RUNG wire#powerrail
      Contact( "DB334_EXTENDED_M_CODE_UNIT_02_STA_0".M_code[505] )
      wire#w1
      I_Contact( "DB334_EXTENDED_M_CODE_UNIT_02_STA_0".M_code[505] )
      wire#w2
      I_Contact( "DB356_M_UNIT_02_STA_0".M_CODES_UNIT_02_STA_0.Ack_M505 )
      I_Contact( "DB2120_MPP_ITC_IPC".RESET_FAULTS )
      Contact( "DB2440_GLOBAL_DATA".GLOBAL_DATA.ANY_PART_CYCLE_RUN )
      Coil( "DB356_M_UNIT_02_STA_0".M_CODES_UNIT_02_STA_0.M505 )
   END_RUNG
   RUNG wire#powerrail
      Contact( "DB356_M_UNIT_02_STA_0".M_CODES_UNIT_02_STA_0.M505 )
   END_RUNG wire#w1
   RUNG wire#w1
      I_Contact( "DB356_M_UNIT_02_STA_0".M_CODES_UNIT_02_STA_0.M505 )
   END_RUNG wire#w2
   // the same network as SCL:
   "DB356_M_UNIT_02_STA_0".M_CODES_UNIT_02_STA_0.M505 := ("DB334_EXTENDED_M_CODE_UNIT_02_STA_0".M_code[505] OR "DB356_M_UNIT_02_STA_0".M_CODES_UNIT_02_STA_0.M505) AND (NOT "DB334_EXTENDED_M_CODE_UNIT_02_STA_0".M_code[505] OR NOT "DB356_M_UNIT_02_STA_0".M_CODES_UNIT_02_STA_0.M505) AND NOT "DB356_M_UNIT_02_STA_0".M_CODES_UNIT_02_STA_0.Ack_M505 AND NOT "DB2120_MPP_ITC_IPC".RESET_FAULTS AND "DB2440_GLOBAL_DATA".GLOBAL_DATA.ANY_PART_CYCLE_RUN;
END_REGION

REGION Network 57: ACKNOWLEDGE M506-UNIT 02 FIXTURE 2 VERIFY PARTS ARE UNCLAMPED PARTS LOADING (WHEN TRUE DO). TOGGLED / ACKNOWLEDGE M47-VERIFY FIXTURE 2 PART AND TOOL IS CLAMPED DURING
   RUNG wire#powerrail
      Contact( "M_ZERO" )
      Coil( "DB356_M_UNIT_02_STA_0".M_CODES_UNIT_02_STA_0.Ack_M506 )
   END_RUNG
   // the same network as SCL:
   "DB356_M_UNIT_02_STA_0".M_CODES_UNIT_02_STA_0.Ack_M506 := "M_ZERO";
END_REGION

REGION Network 58: M506-UNIT 02 FIXTURE 2 VERIFY PARTS ARE UNCLAMPED PARTS LOADING (WHEN TRUE DO). TOGGLED / M47-VERIFY FIXTURE 2 PART AND TOOL IS CLAMPED DURING MACHINING
   RUNG wire#powerrail
      Contact( "DB334_EXTENDED_M_CODE_UNIT_02_STA_0".M_code[506] )
      wire#w1
      I_Contact( "DB334_EXTENDED_M_CODE_UNIT_02_STA_0".M_code[506] )
      wire#w2
      I_Contact( "DB356_M_UNIT_02_STA_0".M_CODES_UNIT_02_STA_0.Ack_M506 )
      I_Contact( "DB2120_MPP_ITC_IPC".RESET_FAULTS )
      Contact( "DB2440_GLOBAL_DATA".GLOBAL_DATA.ANY_PART_CYCLE_RUN )
      Coil( "DB356_M_UNIT_02_STA_0".M_CODES_UNIT_02_STA_0.M506 )
   END_RUNG
   RUNG wire#powerrail
      Contact( "DB356_M_UNIT_02_STA_0".M_CODES_UNIT_02_STA_0.M506 )
   END_RUNG wire#w1
   RUNG wire#w1
      I_Contact( "DB356_M_UNIT_02_STA_0".M_CODES_UNIT_02_STA_0.M506 )
   END_RUNG wire#w2
   // the same network as SCL:
   "DB356_M_UNIT_02_STA_0".M_CODES_UNIT_02_STA_0.M506 := ("DB334_EXTENDED_M_CODE_UNIT_02_STA_0".M_code[506] OR "DB356_M_UNIT_02_STA_0".M_CODES_UNIT_02_STA_0.M506) AND (NOT "DB334_EXTENDED_M_CODE_UNIT_02_STA_0".M_code[506] OR NOT "DB356_M_UNIT_02_STA_0".M_CODES_UNIT_02_STA_0.M506) AND NOT "DB356_M_UNIT_02_STA_0".M_CODES_UNIT_02_STA_0.Ack_M506 AND NOT "DB2120_MPP_ITC_IPC".RESET_FAULTS AND "DB2440_GLOBAL_DATA".GLOBAL_DATA.ANY_PART_CYCLE_RUN;
END_REGION

REGION Network 59: ACKNOWLEDGE M507-UNIT 02 FIXTURE 2 VERIFY FIXTURE REMAINS CLAMPED
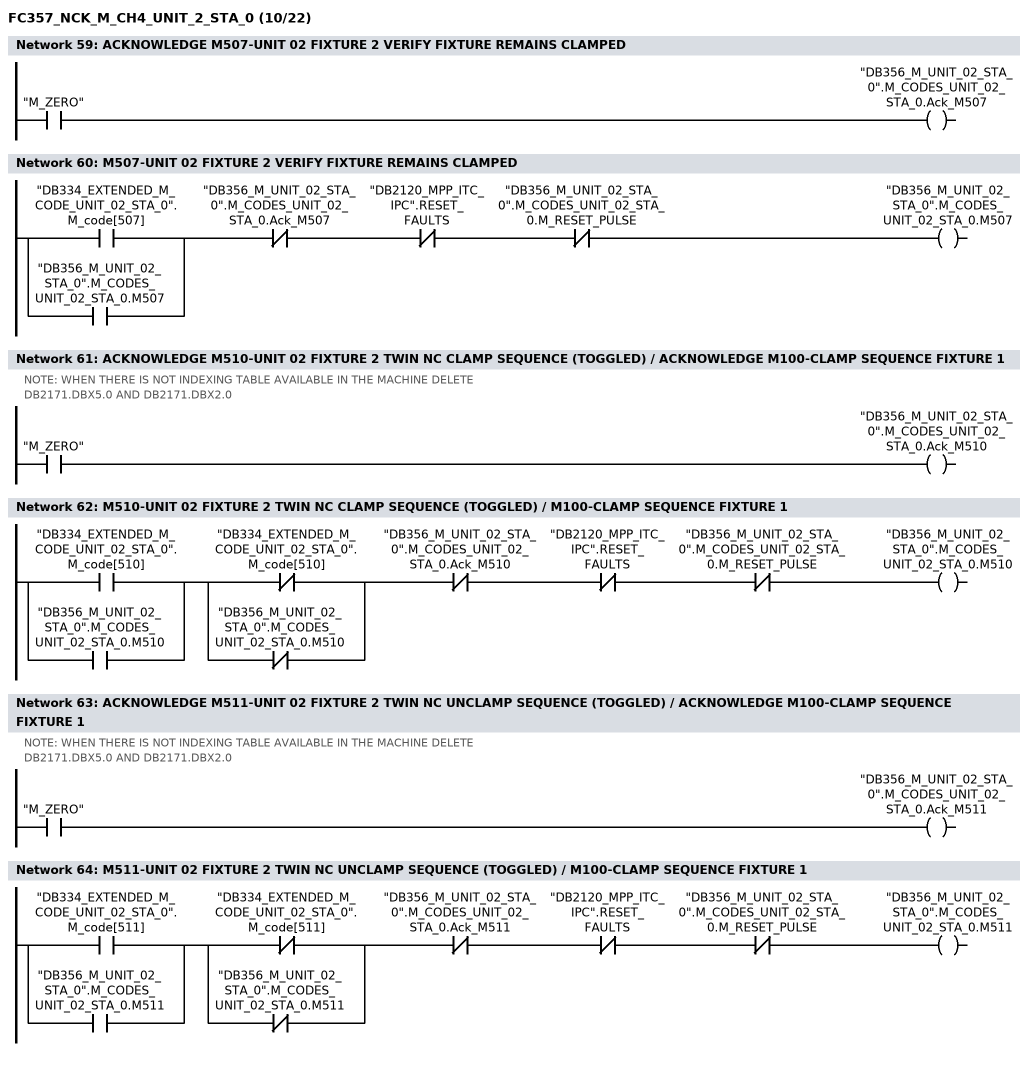
   RUNG wire#powerrail
      Contact( "M_ZERO" )
      Coil( "DB356_M_UNIT_02_STA_0".M_CODES_UNIT_02_STA_0.Ack_M507 )
   END_RUNG
   // the same network as SCL:
   "DB356_M_UNIT_02_STA_0".M_CODES_UNIT_02_STA_0.Ack_M507 := "M_ZERO";
END_REGION

REGION Network 60: M507-UNIT 02 FIXTURE 2 VERIFY FIXTURE REMAINS CLAMPED
   RUNG wire#powerrail
      Contact( "DB334_EXTENDED_M_CODE_UNIT_02_STA_0".M_code[507] )
      wire#w1
      I_Contact( "DB356_M_UNIT_02_STA_0".M_CODES_UNIT_02_STA_0.Ack_M507 )
      I_Contact( "DB2120_MPP_ITC_IPC".RESET_FAULTS )
      I_Contact( "DB356_M_UNIT_02_STA_0".M_CODES_UNIT_02_STA_0.M_RESET_PULSE )
      Coil( "DB356_M_UNIT_02_STA_0".M_CODES_UNIT_02_STA_0.M507 )
   END_RUNG
   RUNG wire#powerrail
      Contact( "DB356_M_UNIT_02_STA_0".M_CODES_UNIT_02_STA_0.M507 )
   END_RUNG wire#w1
   // the same network as SCL:
   "DB356_M_UNIT_02_STA_0".M_CODES_UNIT_02_STA_0.M507 := ("DB334_EXTENDED_M_CODE_UNIT_02_STA_0".M_code[507] OR "DB356_M_UNIT_02_STA_0".M_CODES_UNIT_02_STA_0.M507) AND NOT "DB356_M_UNIT_02_STA_0".M_CODES_UNIT_02_STA_0.Ack_M507 AND NOT "DB2120_MPP_ITC_IPC".RESET_FAULTS AND NOT "DB356_M_UNIT_02_STA_0".M_CODES_UNIT_02_STA_0.M_RESET_PULSE;
END_REGION

REGION Network 61: ACKNOWLEDGE M510-UNIT 02 FIXTURE 2 TWIN NC CLAMP SEQUENCE (TOGGLED) / ACKNOWLEDGE M100-CLAMP SEQUENCE FIXTURE 1
   // NOTE: WHEN THERE IS NOT INDEXING TABLE AVAILABLE IN THE MACHINE DELETE 
   // DB2171.DBX5.0 AND DB2171.DBX2.0
   RUNG wire#powerrail
      Contact( "M_ZERO" )
      Coil( "DB356_M_UNIT_02_STA_0".M_CODES_UNIT_02_STA_0.Ack_M510 )
   END_RUNG
   // the same network as SCL:
   "DB356_M_UNIT_02_STA_0".M_CODES_UNIT_02_STA_0.Ack_M510 := "M_ZERO";
END_REGION

REGION Network 62: M510-UNIT 02 FIXTURE 2 TWIN NC CLAMP SEQUENCE (TOGGLED) / M100-CLAMP SEQUENCE FIXTURE 1
   RUNG wire#powerrail
      Contact( "DB334_EXTENDED_M_CODE_UNIT_02_STA_0".M_code[510] )
      wire#w1
      I_Contact( "DB334_EXTENDED_M_CODE_UNIT_02_STA_0".M_code[510] )
      wire#w2
      I_Contact( "DB356_M_UNIT_02_STA_0".M_CODES_UNIT_02_STA_0.Ack_M510 )
      I_Contact( "DB2120_MPP_ITC_IPC".RESET_FAULTS )
      I_Contact( "DB356_M_UNIT_02_STA_0".M_CODES_UNIT_02_STA_0.M_RESET_PULSE )
      Coil( "DB356_M_UNIT_02_STA_0".M_CODES_UNIT_02_STA_0.M510 )
   END_RUNG
   RUNG wire#powerrail
      Contact( "DB356_M_UNIT_02_STA_0".M_CODES_UNIT_02_STA_0.M510 )
   END_RUNG wire#w1
   RUNG wire#w1
      I_Contact( "DB356_M_UNIT_02_STA_0".M_CODES_UNIT_02_STA_0.M510 )
   END_RUNG wire#w2
   // the same network as SCL:
   "DB356_M_UNIT_02_STA_0".M_CODES_UNIT_02_STA_0.M510 := ("DB334_EXTENDED_M_CODE_UNIT_02_STA_0".M_code[510] OR "DB356_M_UNIT_02_STA_0".M_CODES_UNIT_02_STA_0.M510) AND (NOT "DB334_EXTENDED_M_CODE_UNIT_02_STA_0".M_code[510] OR NOT "DB356_M_UNIT_02_STA_0".M_CODES_UNIT_02_STA_0.M510) AND NOT "DB356_M_UNIT_02_STA_0".M_CODES_UNIT_02_STA_0.Ack_M510 AND NOT "DB2120_MPP_ITC_IPC".RESET_FAULTS AND NOT "DB356_M_UNIT_02_STA_0".M_CODES_UNIT_02_STA_0.M_RESET_PULSE;
END_REGION

REGION Network 63: ACKNOWLEDGE M511-UNIT 02 FIXTURE 2 TWIN NC UNCLAMP SEQUENCE (TOGGLED) / ACKNOWLEDGE M100-CLAMP SEQUENCE FIXTURE 1
   // NOTE: WHEN THERE IS NOT INDEXING TABLE AVAILABLE IN THE MACHINE DELETE 
   // DB2171.DBX5.0 AND DB2171.DBX2.0
   RUNG wire#powerrail
      Contact( "M_ZERO" )
      Coil( "DB356_M_UNIT_02_STA_0".M_CODES_UNIT_02_STA_0.Ack_M511 )
   END_RUNG
   // the same network as SCL:
   "DB356_M_UNIT_02_STA_0".M_CODES_UNIT_02_STA_0.Ack_M511 := "M_ZERO";
END_REGION

REGION Network 64: M511-UNIT 02 FIXTURE 2 TWIN NC UNCLAMP SEQUENCE (TOGGLED) / M100-CLAMP SEQUENCE FIXTURE 1
   RUNG wire#powerrail
      Contact( "DB334_EXTENDED_M_CODE_UNIT_02_STA_0".M_code[511] )
      wire#w1
      I_Contact( "DB334_EXTENDED_M_CODE_UNIT_02_STA_0".M_code[511] )
      wire#w2
      I_Contact( "DB356_M_UNIT_02_STA_0".M_CODES_UNIT_02_STA_0.Ack_M511 )
      I_Contact( "DB2120_MPP_ITC_IPC".RESET_FAULTS )
      I_Contact( "DB356_M_UNIT_02_STA_0".M_CODES_UNIT_02_STA_0.M_RESET_PULSE )
      Coil( "DB356_M_UNIT_02_STA_0".M_CODES_UNIT_02_STA_0.M511 )
   END_RUNG
   RUNG wire#powerrail
      Contact( "DB356_M_UNIT_02_STA_0".M_CODES_UNIT_02_STA_0.M511 )
   END_RUNG wire#w1
   RUNG wire#w1
      I_Contact( "DB356_M_UNIT_02_STA_0".M_CODES_UNIT_02_STA_0.M511 )
   END_RUNG wire#w2
   // the same network as SCL:
   "DB356_M_UNIT_02_STA_0".M_CODES_UNIT_02_STA_0.M511 := ("DB334_EXTENDED_M_CODE_UNIT_02_STA_0".M_code[511] OR "DB356_M_UNIT_02_STA_0".M_CODES_UNIT_02_STA_0.M511) AND (NOT "DB334_EXTENDED_M_CODE_UNIT_02_STA_0".M_code[511] OR NOT "DB356_M_UNIT_02_STA_0".M_CODES_UNIT_02_STA_0.M511) AND NOT "DB356_M_UNIT_02_STA_0".M_CODES_UNIT_02_STA_0.Ack_M511 AND NOT "DB2120_MPP_ITC_IPC".RESET_FAULTS AND NOT "DB356_M_UNIT_02_STA_0".M_CODES_UNIT_02_STA_0.M_RESET_PULSE;
END_REGION

REGION Network 65: ACKNOWLEDGE M520- UNIT 02 FIXTURE 2 GRIPPER CLOSE (READ-IN DISABLE)
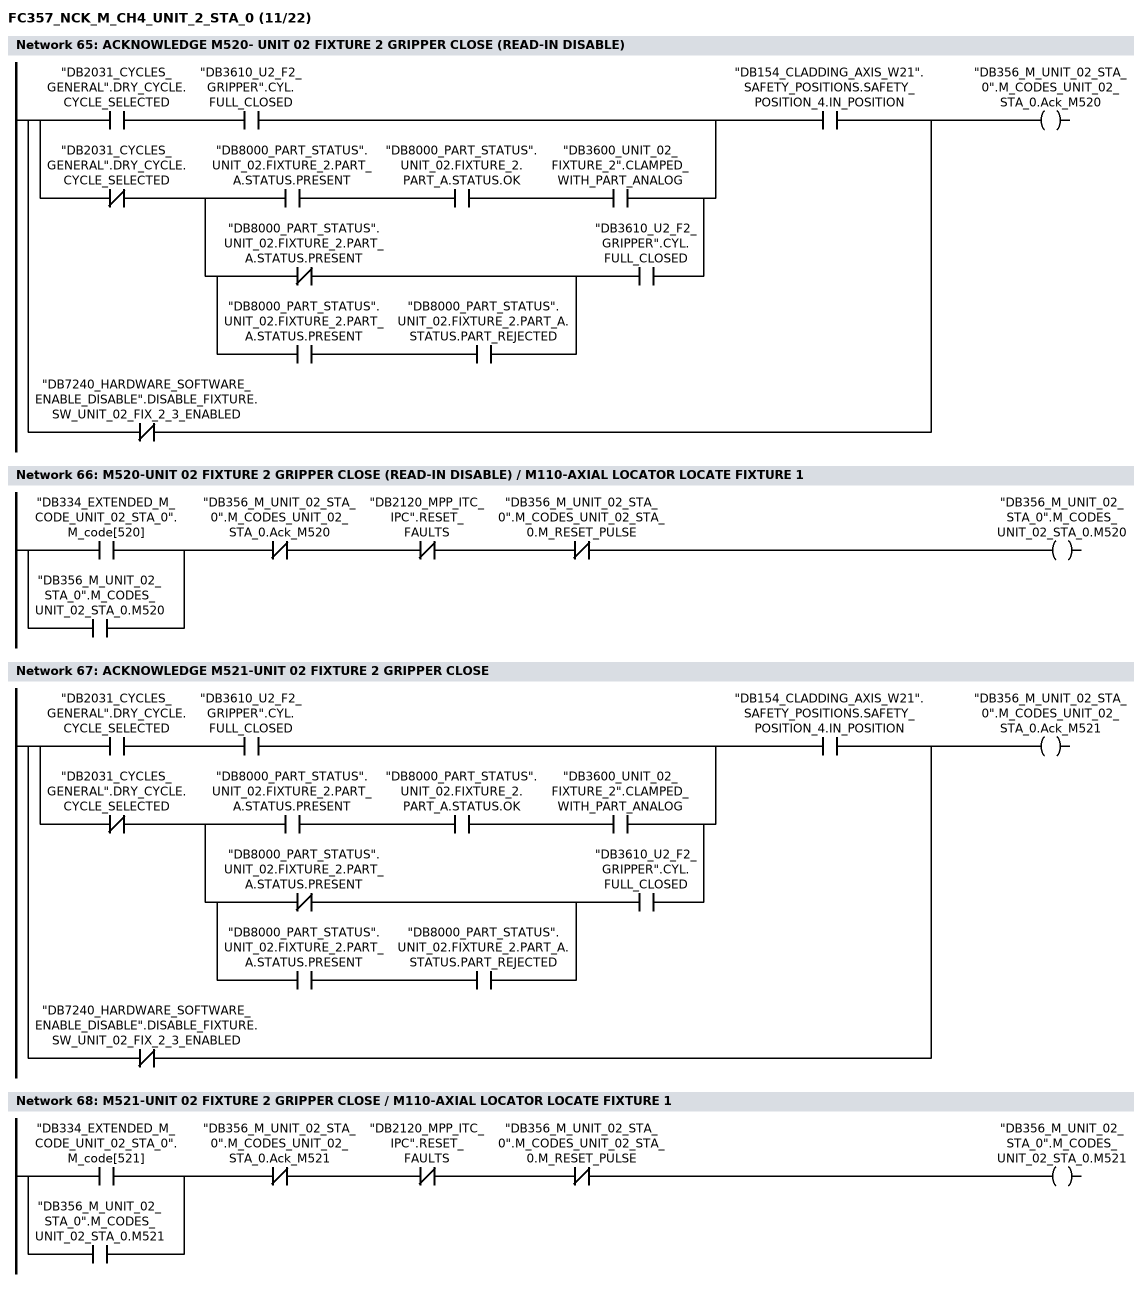
   RUNG wire#powerrail
      Contact( "DB2031_CYCLES_GENERAL".DRY_CYCLE.CYCLE_SELECTED )
      Contact( "DB3610_U2_F2_GRIPPER".CYL.FULL_CLOSED )
      wire#w1
      Contact( "DB154_CLADDING_AXIS_W21".SAFETY_POSITIONS.SAFETY_POSITION_4.IN_POSITION )
      wire#w4
      Coil( "DB356_M_UNIT_02_STA_0".M_CODES_UNIT_02_STA_0.Ack_M520 )
   END_RUNG
   RUNG wire#powerrail
      I_Contact( "DB2031_CYCLES_GENERAL".DRY_CYCLE.CYCLE_SELECTED )
      wire#w2
      Contact( "DB8000_PART_STATUS".UNIT_02.FIXTURE_2.PART_A.STATUS.PRESENT )
      Contact( "DB8000_PART_STATUS".UNIT_02.FIXTURE_2.PART_A.STATUS.OK )
      Contact( "DB3600_UNIT_02_FIXTURE_2".CLAMPED_WITH_PART_ANALOG )
   END_RUNG wire#w1
   RUNG wire#w2
      I_Contact( "DB8000_PART_STATUS".UNIT_02.FIXTURE_2.PART_A.STATUS.PRESENT )
      wire#w3
      Contact( "DB3610_U2_F2_GRIPPER".CYL.FULL_CLOSED )
   END_RUNG wire#w1
   RUNG wire#w2
      Contact( "DB8000_PART_STATUS".UNIT_02.FIXTURE_2.PART_A.STATUS.PRESENT )
      Contact( "DB8000_PART_STATUS".UNIT_02.FIXTURE_2.PART_A.STATUS.PART_REJECTED )
   END_RUNG wire#w3
   RUNG wire#powerrail
      I_Contact( "DB7240_HARDWARE_SOFTWARE_ENABLE_DISABLE".DISABLE_FIXTURE.SW_UNIT_02_FIX_2_3_ENABLED )
   END_RUNG wire#w4
   // the same network as SCL:
   "DB356_M_UNIT_02_STA_0".M_CODES_UNIT_02_STA_0.Ack_M520 := ((("DB2031_CYCLES_GENERAL".DRY_CYCLE.CYCLE_SELECTED AND "DB3610_U2_F2_GRIPPER".CYL.FULL_CLOSED) OR (NOT "DB2031_CYCLES_GENERAL".DRY_CYCLE.CYCLE_SELECTED AND (("DB8000_PART_STATUS".UNIT_02.FIXTURE_2.PART_A.STATUS.PRESENT AND "DB8000_PART_STATUS".UNIT_02.FIXTURE_2.PART_A.STATUS.OK AND "DB3600_UNIT_02_FIXTURE_2".CLAMPED_WITH_PART_ANALOG) OR ((NOT "DB8000_PART_STATUS".UNIT_02.FIXTURE_2.PART_A.STATUS.PRESENT OR ("DB8000_PART_STATUS".UNIT_02.FIXTURE_2.PART_A.STATUS.PRESENT AND "DB8000_PART_STATUS".UNIT_02.FIXTURE_2.PART_A.STATUS.PART_REJECTED)) AND "DB3610_U2_F2_GRIPPER".CYL.FULL_CLOSED)))) AND "DB154_CLADDING_AXIS_W21".SAFETY_POSITIONS.SAFETY_POSITION_4.IN_POSITION) OR NOT "DB7240_HARDWARE_SOFTWARE_ENABLE_DISABLE".DISABLE_FIXTURE.SW_UNIT_02_FIX_2_3_ENABLED;
END_REGION

REGION Network 66: M520-UNIT 02 FIXTURE 2 GRIPPER CLOSE (READ-IN DISABLE) / M110-AXIAL LOCATOR LOCATE FIXTURE 1
   RUNG wire#powerrail
      Contact( "DB334_EXTENDED_M_CODE_UNIT_02_STA_0".M_code[520] )
      wire#w1
      I_Contact( "DB356_M_UNIT_02_STA_0".M_CODES_UNIT_02_STA_0.Ack_M520 )
      I_Contact( "DB2120_MPP_ITC_IPC".RESET_FAULTS )
      I_Contact( "DB356_M_UNIT_02_STA_0".M_CODES_UNIT_02_STA_0.M_RESET_PULSE )
      Coil( "DB356_M_UNIT_02_STA_0".M_CODES_UNIT_02_STA_0.M520 )
   END_RUNG
   RUNG wire#powerrail
      Contact( "DB356_M_UNIT_02_STA_0".M_CODES_UNIT_02_STA_0.M520 )
   END_RUNG wire#w1
   // the same network as SCL:
   "DB356_M_UNIT_02_STA_0".M_CODES_UNIT_02_STA_0.M520 := ("DB334_EXTENDED_M_CODE_UNIT_02_STA_0".M_code[520] OR "DB356_M_UNIT_02_STA_0".M_CODES_UNIT_02_STA_0.M520) AND NOT "DB356_M_UNIT_02_STA_0".M_CODES_UNIT_02_STA_0.Ack_M520 AND NOT "DB2120_MPP_ITC_IPC".RESET_FAULTS AND NOT "DB356_M_UNIT_02_STA_0".M_CODES_UNIT_02_STA_0.M_RESET_PULSE;
END_REGION

REGION Network 67: ACKNOWLEDGE M521-UNIT 02 FIXTURE 2 GRIPPER CLOSE
   RUNG wire#powerrail
      Contact( "DB2031_CYCLES_GENERAL".DRY_CYCLE.CYCLE_SELECTED )
      Contact( "DB3610_U2_F2_GRIPPER".CYL.FULL_CLOSED )
      wire#w1
      Contact( "DB154_CLADDING_AXIS_W21".SAFETY_POSITIONS.SAFETY_POSITION_4.IN_POSITION )
      wire#w4
      Coil( "DB356_M_UNIT_02_STA_0".M_CODES_UNIT_02_STA_0.Ack_M521 )
   END_RUNG
   RUNG wire#powerrail
      I_Contact( "DB2031_CYCLES_GENERAL".DRY_CYCLE.CYCLE_SELECTED )
      wire#w2
      Contact( "DB8000_PART_STATUS".UNIT_02.FIXTURE_2.PART_A.STATUS.PRESENT )
      Contact( "DB8000_PART_STATUS".UNIT_02.FIXTURE_2.PART_A.STATUS.OK )
      Contact( "DB3600_UNIT_02_FIXTURE_2".CLAMPED_WITH_PART_ANALOG )
   END_RUNG wire#w1
   RUNG wire#w2
      I_Contact( "DB8000_PART_STATUS".UNIT_02.FIXTURE_2.PART_A.STATUS.PRESENT )
      wire#w3
      Contact( "DB3610_U2_F2_GRIPPER".CYL.FULL_CLOSED )
   END_RUNG wire#w1
   RUNG wire#w2
      Contact( "DB8000_PART_STATUS".UNIT_02.FIXTURE_2.PART_A.STATUS.PRESENT )
      Contact( "DB8000_PART_STATUS".UNIT_02.FIXTURE_2.PART_A.STATUS.PART_REJECTED )
   END_RUNG wire#w3
   RUNG wire#powerrail
      I_Contact( "DB7240_HARDWARE_SOFTWARE_ENABLE_DISABLE".DISABLE_FIXTURE.SW_UNIT_02_FIX_2_3_ENABLED )
   END_RUNG wire#w4
   // the same network as SCL:
   "DB356_M_UNIT_02_STA_0".M_CODES_UNIT_02_STA_0.Ack_M521 := ((("DB2031_CYCLES_GENERAL".DRY_CYCLE.CYCLE_SELECTED AND "DB3610_U2_F2_GRIPPER".CYL.FULL_CLOSED) OR (NOT "DB2031_CYCLES_GENERAL".DRY_CYCLE.CYCLE_SELECTED AND (("DB8000_PART_STATUS".UNIT_02.FIXTURE_2.PART_A.STATUS.PRESENT AND "DB8000_PART_STATUS".UNIT_02.FIXTURE_2.PART_A.STATUS.OK AND "DB3600_UNIT_02_FIXTURE_2".CLAMPED_WITH_PART_ANALOG) OR ((NOT "DB8000_PART_STATUS".UNIT_02.FIXTURE_2.PART_A.STATUS.PRESENT OR ("DB8000_PART_STATUS".UNIT_02.FIXTURE_2.PART_A.STATUS.PRESENT AND "DB8000_PART_STATUS".UNIT_02.FIXTURE_2.PART_A.STATUS.PART_REJECTED)) AND "DB3610_U2_F2_GRIPPER".CYL.FULL_CLOSED)))) AND "DB154_CLADDING_AXIS_W21".SAFETY_POSITIONS.SAFETY_POSITION_4.IN_POSITION) OR NOT "DB7240_HARDWARE_SOFTWARE_ENABLE_DISABLE".DISABLE_FIXTURE.SW_UNIT_02_FIX_2_3_ENABLED;
END_REGION

REGION Network 68: M521-UNIT 02 FIXTURE 2 GRIPPER CLOSE / M110-AXIAL LOCATOR LOCATE FIXTURE 1
   RUNG wire#powerrail
      Contact( "DB334_EXTENDED_M_CODE_UNIT_02_STA_0".M_code[521] )
      wire#w1
      I_Contact( "DB356_M_UNIT_02_STA_0".M_CODES_UNIT_02_STA_0.Ack_M521 )
      I_Contact( "DB2120_MPP_ITC_IPC".RESET_FAULTS )
      I_Contact( "DB356_M_UNIT_02_STA_0".M_CODES_UNIT_02_STA_0.M_RESET_PULSE )
      Coil( "DB356_M_UNIT_02_STA_0".M_CODES_UNIT_02_STA_0.M521 )
   END_RUNG
   RUNG wire#powerrail
      Contact( "DB356_M_UNIT_02_STA_0".M_CODES_UNIT_02_STA_0.M521 )
   END_RUNG wire#w1
   // the same network as SCL:
   "DB356_M_UNIT_02_STA_0".M_CODES_UNIT_02_STA_0.M521 := ("DB334_EXTENDED_M_CODE_UNIT_02_STA_0".M_code[521] OR "DB356_M_UNIT_02_STA_0".M_CODES_UNIT_02_STA_0.M521) AND NOT "DB356_M_UNIT_02_STA_0".M_CODES_UNIT_02_STA_0.Ack_M521 AND NOT "DB2120_MPP_ITC_IPC".RESET_FAULTS AND NOT "DB356_M_UNIT_02_STA_0".M_CODES_UNIT_02_STA_0.M_RESET_PULSE;
END_REGION

REGION Network 69: ACKNOWLEDGE M522-UNIT 02 FIXTURE 2 GRIPPER OPEN (READ-IN DISABLE) / ACKNOWLEDGE M111-AXIAL LOCATOR RETURN FIXTURE 1
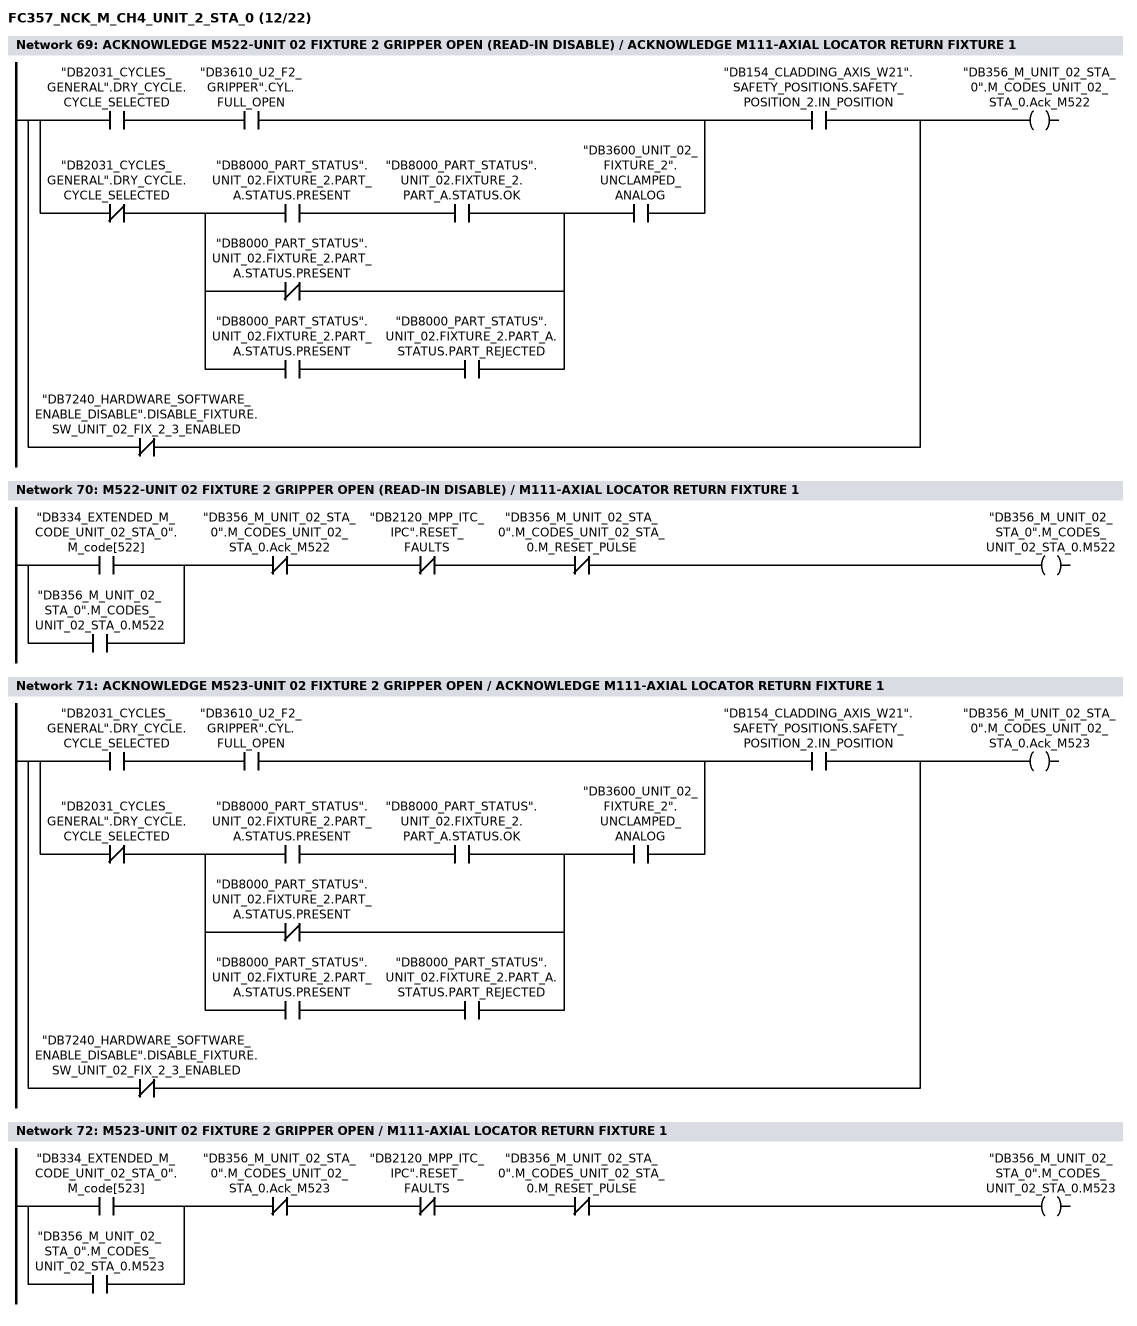
   RUNG wire#powerrail
      Contact( "DB2031_CYCLES_GENERAL".DRY_CYCLE.CYCLE_SELECTED )
      Contact( "DB3610_U2_F2_GRIPPER".CYL.FULL_OPEN )
      wire#w1
      Contact( "DB154_CLADDING_AXIS_W21".SAFETY_POSITIONS.SAFETY_POSITION_2.IN_POSITION )
      wire#w4
      Coil( "DB356_M_UNIT_02_STA_0".M_CODES_UNIT_02_STA_0.Ack_M522 )
   END_RUNG
   RUNG wire#powerrail
      I_Contact( "DB2031_CYCLES_GENERAL".DRY_CYCLE.CYCLE_SELECTED )
      wire#w2
      Contact( "DB8000_PART_STATUS".UNIT_02.FIXTURE_2.PART_A.STATUS.PRESENT )
      Contact( "DB8000_PART_STATUS".UNIT_02.FIXTURE_2.PART_A.STATUS.OK )
      wire#w3
      Contact( "DB3600_UNIT_02_FIXTURE_2".UNCLAMPED_ANALOG )
   END_RUNG wire#w1
   RUNG wire#w2
      I_Contact( "DB8000_PART_STATUS".UNIT_02.FIXTURE_2.PART_A.STATUS.PRESENT )
   END_RUNG wire#w3
   RUNG wire#w2
      Contact( "DB8000_PART_STATUS".UNIT_02.FIXTURE_2.PART_A.STATUS.PRESENT )
      Contact( "DB8000_PART_STATUS".UNIT_02.FIXTURE_2.PART_A.STATUS.PART_REJECTED )
   END_RUNG wire#w3
   RUNG wire#powerrail
      I_Contact( "DB7240_HARDWARE_SOFTWARE_ENABLE_DISABLE".DISABLE_FIXTURE.SW_UNIT_02_FIX_2_3_ENABLED )
   END_RUNG wire#w4
   // the same network as SCL:
   "DB356_M_UNIT_02_STA_0".M_CODES_UNIT_02_STA_0.Ack_M522 := ((("DB2031_CYCLES_GENERAL".DRY_CYCLE.CYCLE_SELECTED AND "DB3610_U2_F2_GRIPPER".CYL.FULL_OPEN) OR (NOT "DB2031_CYCLES_GENERAL".DRY_CYCLE.CYCLE_SELECTED AND (("DB8000_PART_STATUS".UNIT_02.FIXTURE_2.PART_A.STATUS.PRESENT AND "DB8000_PART_STATUS".UNIT_02.FIXTURE_2.PART_A.STATUS.OK) OR NOT "DB8000_PART_STATUS".UNIT_02.FIXTURE_2.PART_A.STATUS.PRESENT OR ("DB8000_PART_STATUS".UNIT_02.FIXTURE_2.PART_A.STATUS.PRESENT AND "DB8000_PART_STATUS".UNIT_02.FIXTURE_2.PART_A.STATUS.PART_REJECTED)) AND "DB3600_UNIT_02_FIXTURE_2".UNCLAMPED_ANALOG)) AND "DB154_CLADDING_AXIS_W21".SAFETY_POSITIONS.SAFETY_POSITION_2.IN_POSITION) OR NOT "DB7240_HARDWARE_SOFTWARE_ENABLE_DISABLE".DISABLE_FIXTURE.SW_UNIT_02_FIX_2_3_ENABLED;
END_REGION

REGION Network 70: M522-UNIT 02 FIXTURE 2 GRIPPER OPEN (READ-IN DISABLE) / M111-AXIAL LOCATOR RETURN FIXTURE 1
   RUNG wire#powerrail
      Contact( "DB334_EXTENDED_M_CODE_UNIT_02_STA_0".M_code[522] )
      wire#w1
      I_Contact( "DB356_M_UNIT_02_STA_0".M_CODES_UNIT_02_STA_0.Ack_M522 )
      I_Contact( "DB2120_MPP_ITC_IPC".RESET_FAULTS )
      I_Contact( "DB356_M_UNIT_02_STA_0".M_CODES_UNIT_02_STA_0.M_RESET_PULSE )
      Coil( "DB356_M_UNIT_02_STA_0".M_CODES_UNIT_02_STA_0.M522 )
   END_RUNG
   RUNG wire#powerrail
      Contact( "DB356_M_UNIT_02_STA_0".M_CODES_UNIT_02_STA_0.M522 )
   END_RUNG wire#w1
   // the same network as SCL:
   "DB356_M_UNIT_02_STA_0".M_CODES_UNIT_02_STA_0.M522 := ("DB334_EXTENDED_M_CODE_UNIT_02_STA_0".M_code[522] OR "DB356_M_UNIT_02_STA_0".M_CODES_UNIT_02_STA_0.M522) AND NOT "DB356_M_UNIT_02_STA_0".M_CODES_UNIT_02_STA_0.Ack_M522 AND NOT "DB2120_MPP_ITC_IPC".RESET_FAULTS AND NOT "DB356_M_UNIT_02_STA_0".M_CODES_UNIT_02_STA_0.M_RESET_PULSE;
END_REGION

REGION Network 71: ACKNOWLEDGE M523-UNIT 02 FIXTURE 2 GRIPPER OPEN / ACKNOWLEDGE M111-AXIAL LOCATOR RETURN FIXTURE 1
   RUNG wire#powerrail
      Contact( "DB2031_CYCLES_GENERAL".DRY_CYCLE.CYCLE_SELECTED )
      Contact( "DB3610_U2_F2_GRIPPER".CYL.FULL_OPEN )
      wire#w1
      Contact( "DB154_CLADDING_AXIS_W21".SAFETY_POSITIONS.SAFETY_POSITION_2.IN_POSITION )
      wire#w4
      Coil( "DB356_M_UNIT_02_STA_0".M_CODES_UNIT_02_STA_0.Ack_M523 )
   END_RUNG
   RUNG wire#powerrail
      I_Contact( "DB2031_CYCLES_GENERAL".DRY_CYCLE.CYCLE_SELECTED )
      wire#w2
      Contact( "DB8000_PART_STATUS".UNIT_02.FIXTURE_2.PART_A.STATUS.PRESENT )
      Contact( "DB8000_PART_STATUS".UNIT_02.FIXTURE_2.PART_A.STATUS.OK )
      wire#w3
      Contact( "DB3600_UNIT_02_FIXTURE_2".UNCLAMPED_ANALOG )
   END_RUNG wire#w1
   RUNG wire#w2
      I_Contact( "DB8000_PART_STATUS".UNIT_02.FIXTURE_2.PART_A.STATUS.PRESENT )
   END_RUNG wire#w3
   RUNG wire#w2
      Contact( "DB8000_PART_STATUS".UNIT_02.FIXTURE_2.PART_A.STATUS.PRESENT )
      Contact( "DB8000_PART_STATUS".UNIT_02.FIXTURE_2.PART_A.STATUS.PART_REJECTED )
   END_RUNG wire#w3
   RUNG wire#powerrail
      I_Contact( "DB7240_HARDWARE_SOFTWARE_ENABLE_DISABLE".DISABLE_FIXTURE.SW_UNIT_02_FIX_2_3_ENABLED )
   END_RUNG wire#w4
   // the same network as SCL:
   "DB356_M_UNIT_02_STA_0".M_CODES_UNIT_02_STA_0.Ack_M523 := ((("DB2031_CYCLES_GENERAL".DRY_CYCLE.CYCLE_SELECTED AND "DB3610_U2_F2_GRIPPER".CYL.FULL_OPEN) OR (NOT "DB2031_CYCLES_GENERAL".DRY_CYCLE.CYCLE_SELECTED AND (("DB8000_PART_STATUS".UNIT_02.FIXTURE_2.PART_A.STATUS.PRESENT AND "DB8000_PART_STATUS".UNIT_02.FIXTURE_2.PART_A.STATUS.OK) OR NOT "DB8000_PART_STATUS".UNIT_02.FIXTURE_2.PART_A.STATUS.PRESENT OR ("DB8000_PART_STATUS".UNIT_02.FIXTURE_2.PART_A.STATUS.PRESENT AND "DB8000_PART_STATUS".UNIT_02.FIXTURE_2.PART_A.STATUS.PART_REJECTED)) AND "DB3600_UNIT_02_FIXTURE_2".UNCLAMPED_ANALOG)) AND "DB154_CLADDING_AXIS_W21".SAFETY_POSITIONS.SAFETY_POSITION_2.IN_POSITION) OR NOT "DB7240_HARDWARE_SOFTWARE_ENABLE_DISABLE".DISABLE_FIXTURE.SW_UNIT_02_FIX_2_3_ENABLED;
END_REGION

REGION Network 72: M523-UNIT 02 FIXTURE 2 GRIPPER OPEN / M111-AXIAL LOCATOR RETURN FIXTURE 1
   RUNG wire#powerrail
      Contact( "DB334_EXTENDED_M_CODE_UNIT_02_STA_0".M_code[523] )
      wire#w1
      I_Contact( "DB356_M_UNIT_02_STA_0".M_CODES_UNIT_02_STA_0.Ack_M523 )
      I_Contact( "DB2120_MPP_ITC_IPC".RESET_FAULTS )
      I_Contact( "DB356_M_UNIT_02_STA_0".M_CODES_UNIT_02_STA_0.M_RESET_PULSE )
      Coil( "DB356_M_UNIT_02_STA_0".M_CODES_UNIT_02_STA_0.M523 )
   END_RUNG
   RUNG wire#powerrail
      Contact( "DB356_M_UNIT_02_STA_0".M_CODES_UNIT_02_STA_0.M523 )
   END_RUNG wire#w1
   // the same network as SCL:
   "DB356_M_UNIT_02_STA_0".M_CODES_UNIT_02_STA_0.M523 := ("DB334_EXTENDED_M_CODE_UNIT_02_STA_0".M_code[523] OR "DB356_M_UNIT_02_STA_0".M_CODES_UNIT_02_STA_0.M523) AND NOT "DB356_M_UNIT_02_STA_0".M_CODES_UNIT_02_STA_0.Ack_M523 AND NOT "DB2120_MPP_ITC_IPC".RESET_FAULTS AND NOT "DB356_M_UNIT_02_STA_0".M_CODES_UNIT_02_STA_0.M_RESET_PULSE;
END_REGION

REGION Network 73: ACKNOWLEDGE M524-UNIT 02 FIXTURE 2 GRIPPER RELEASE PRESSURE (READ-IN DISABLE) / ACKNOWLEDGE M112-AXIAL LOCATOR RELAX FIXTURE 1
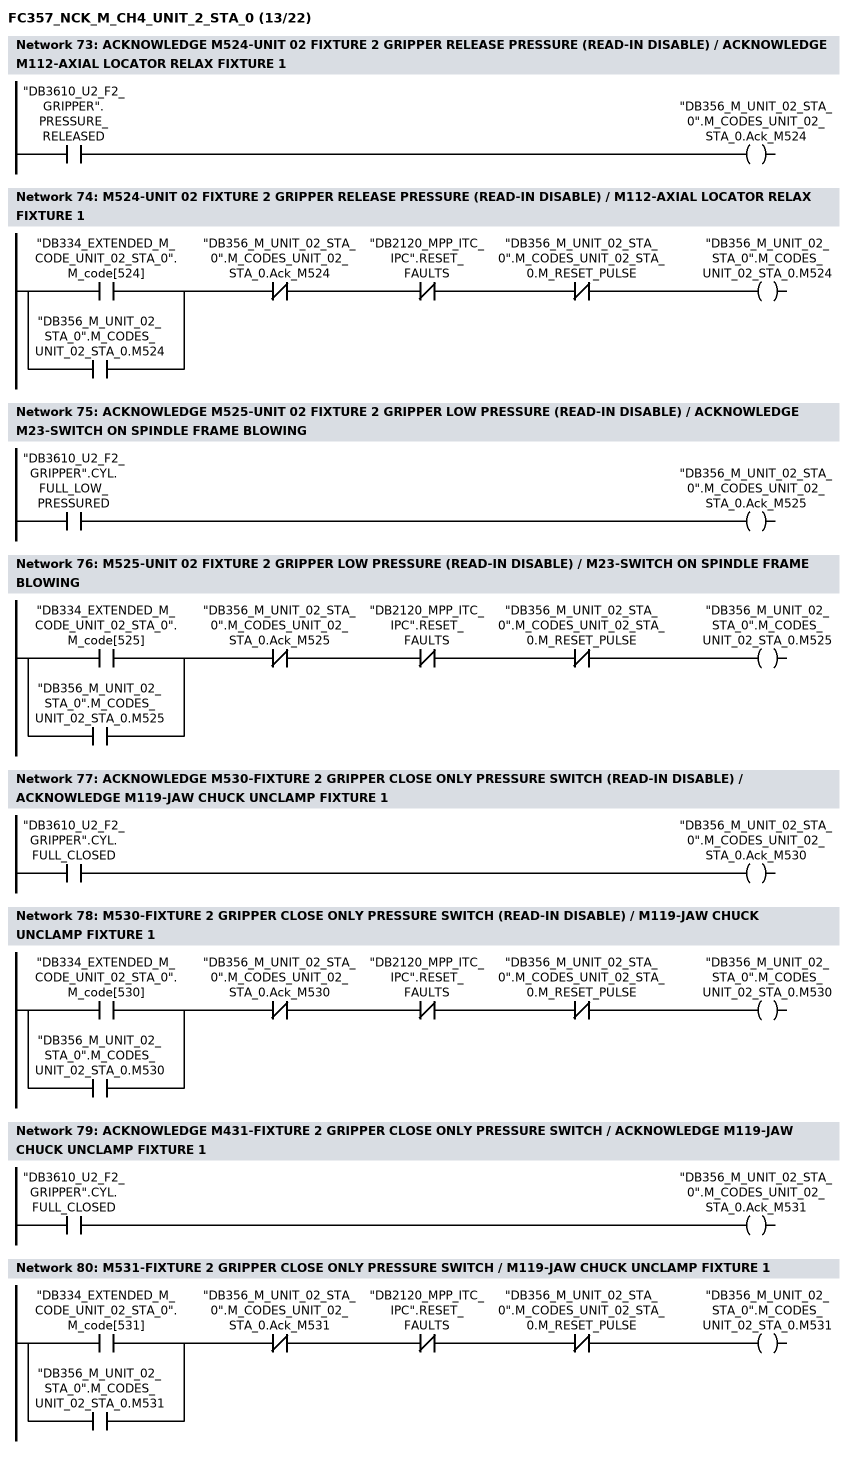
   RUNG wire#powerrail
      Contact( "DB3610_U2_F2_GRIPPER".PRESSURE_RELEASED )
      Coil( "DB356_M_UNIT_02_STA_0".M_CODES_UNIT_02_STA_0.Ack_M524 )
   END_RUNG
   // the same network as SCL:
   "DB356_M_UNIT_02_STA_0".M_CODES_UNIT_02_STA_0.Ack_M524 := "DB3610_U2_F2_GRIPPER".PRESSURE_RELEASED;
END_REGION

REGION Network 74: M524-UNIT 02 FIXTURE 2 GRIPPER RELEASE PRESSURE (READ-IN DISABLE) / M112-AXIAL LOCATOR RELAX FIXTURE 1
   RUNG wire#powerrail
      Contact( "DB334_EXTENDED_M_CODE_UNIT_02_STA_0".M_code[524] )
      wire#w1
      I_Contact( "DB356_M_UNIT_02_STA_0".M_CODES_UNIT_02_STA_0.Ack_M524 )
      I_Contact( "DB2120_MPP_ITC_IPC".RESET_FAULTS )
      I_Contact( "DB356_M_UNIT_02_STA_0".M_CODES_UNIT_02_STA_0.M_RESET_PULSE )
      Coil( "DB356_M_UNIT_02_STA_0".M_CODES_UNIT_02_STA_0.M524 )
   END_RUNG
   RUNG wire#powerrail
      Contact( "DB356_M_UNIT_02_STA_0".M_CODES_UNIT_02_STA_0.M524 )
   END_RUNG wire#w1
   // the same network as SCL:
   "DB356_M_UNIT_02_STA_0".M_CODES_UNIT_02_STA_0.M524 := ("DB334_EXTENDED_M_CODE_UNIT_02_STA_0".M_code[524] OR "DB356_M_UNIT_02_STA_0".M_CODES_UNIT_02_STA_0.M524) AND NOT "DB356_M_UNIT_02_STA_0".M_CODES_UNIT_02_STA_0.Ack_M524 AND NOT "DB2120_MPP_ITC_IPC".RESET_FAULTS AND NOT "DB356_M_UNIT_02_STA_0".M_CODES_UNIT_02_STA_0.M_RESET_PULSE;
END_REGION

REGION Network 75: ACKNOWLEDGE M525-UNIT 02 FIXTURE 2 GRIPPER LOW PRESSURE (READ-IN DISABLE) / ACKNOWLEDGE M23-SWITCH ON SPINDLE FRAME BLOWING
   RUNG wire#powerrail
      Contact( "DB3610_U2_F2_GRIPPER".CYL.FULL_LOW_PRESSURED )
      Coil( "DB356_M_UNIT_02_STA_0".M_CODES_UNIT_02_STA_0.Ack_M525 )
   END_RUNG
   // the same network as SCL:
   "DB356_M_UNIT_02_STA_0".M_CODES_UNIT_02_STA_0.Ack_M525 := "DB3610_U2_F2_GRIPPER".CYL.FULL_LOW_PRESSURED;
END_REGION

REGION Network 76: M525-UNIT 02 FIXTURE 2 GRIPPER LOW PRESSURE (READ-IN DISABLE) / M23-SWITCH ON SPINDLE FRAME BLOWING
   RUNG wire#powerrail
      Contact( "DB334_EXTENDED_M_CODE_UNIT_02_STA_0".M_code[525] )
      wire#w1
      I_Contact( "DB356_M_UNIT_02_STA_0".M_CODES_UNIT_02_STA_0.Ack_M525 )
      I_Contact( "DB2120_MPP_ITC_IPC".RESET_FAULTS )
      I_Contact( "DB356_M_UNIT_02_STA_0".M_CODES_UNIT_02_STA_0.M_RESET_PULSE )
      Coil( "DB356_M_UNIT_02_STA_0".M_CODES_UNIT_02_STA_0.M525 )
   END_RUNG
   RUNG wire#powerrail
      Contact( "DB356_M_UNIT_02_STA_0".M_CODES_UNIT_02_STA_0.M525 )
   END_RUNG wire#w1
   // the same network as SCL:
   "DB356_M_UNIT_02_STA_0".M_CODES_UNIT_02_STA_0.M525 := ("DB334_EXTENDED_M_CODE_UNIT_02_STA_0".M_code[525] OR "DB356_M_UNIT_02_STA_0".M_CODES_UNIT_02_STA_0.M525) AND NOT "DB356_M_UNIT_02_STA_0".M_CODES_UNIT_02_STA_0.Ack_M525 AND NOT "DB2120_MPP_ITC_IPC".RESET_FAULTS AND NOT "DB356_M_UNIT_02_STA_0".M_CODES_UNIT_02_STA_0.M_RESET_PULSE;
END_REGION

REGION Network 77: ACKNOWLEDGE M530-FIXTURE 2 GRIPPER CLOSE ONLY PRESSURE SWITCH (READ-IN DISABLE) / ACKNOWLEDGE M119-JAW CHUCK UNCLAMP FIXTURE 1
   RUNG wire#powerrail
      Contact( "DB3610_U2_F2_GRIPPER".CYL.FULL_CLOSED )
      Coil( "DB356_M_UNIT_02_STA_0".M_CODES_UNIT_02_STA_0.Ack_M530 )
   END_RUNG
   // the same network as SCL:
   "DB356_M_UNIT_02_STA_0".M_CODES_UNIT_02_STA_0.Ack_M530 := "DB3610_U2_F2_GRIPPER".CYL.FULL_CLOSED;
END_REGION

REGION Network 78: M530-FIXTURE 2 GRIPPER CLOSE ONLY PRESSURE SWITCH (READ-IN DISABLE) / M119-JAW CHUCK UNCLAMP FIXTURE 1
   RUNG wire#powerrail
      Contact( "DB334_EXTENDED_M_CODE_UNIT_02_STA_0".M_code[530] )
      wire#w1
      I_Contact( "DB356_M_UNIT_02_STA_0".M_CODES_UNIT_02_STA_0.Ack_M530 )
      I_Contact( "DB2120_MPP_ITC_IPC".RESET_FAULTS )
      I_Contact( "DB356_M_UNIT_02_STA_0".M_CODES_UNIT_02_STA_0.M_RESET_PULSE )
      Coil( "DB356_M_UNIT_02_STA_0".M_CODES_UNIT_02_STA_0.M530 )
   END_RUNG
   RUNG wire#powerrail
      Contact( "DB356_M_UNIT_02_STA_0".M_CODES_UNIT_02_STA_0.M530 )
   END_RUNG wire#w1
   // the same network as SCL:
   "DB356_M_UNIT_02_STA_0".M_CODES_UNIT_02_STA_0.M530 := ("DB334_EXTENDED_M_CODE_UNIT_02_STA_0".M_code[530] OR "DB356_M_UNIT_02_STA_0".M_CODES_UNIT_02_STA_0.M530) AND NOT "DB356_M_UNIT_02_STA_0".M_CODES_UNIT_02_STA_0.Ack_M530 AND NOT "DB2120_MPP_ITC_IPC".RESET_FAULTS AND NOT "DB356_M_UNIT_02_STA_0".M_CODES_UNIT_02_STA_0.M_RESET_PULSE;
END_REGION

REGION Network 79: ACKNOWLEDGE M431-FIXTURE 2 GRIPPER CLOSE ONLY PRESSURE SWITCH / ACKNOWLEDGE M119-JAW CHUCK UNCLAMP FIXTURE 1
   RUNG wire#powerrail
      Contact( "DB3610_U2_F2_GRIPPER".CYL.FULL_CLOSED )
      Coil( "DB356_M_UNIT_02_STA_0".M_CODES_UNIT_02_STA_0.Ack_M531 )
   END_RUNG
   // the same network as SCL:
   "DB356_M_UNIT_02_STA_0".M_CODES_UNIT_02_STA_0.Ack_M531 := "DB3610_U2_F2_GRIPPER".CYL.FULL_CLOSED;
END_REGION

REGION Network 80: M531-FIXTURE 2 GRIPPER CLOSE ONLY PRESSURE SWITCH / M119-JAW CHUCK UNCLAMP FIXTURE 1
   RUNG wire#powerrail
      Contact( "DB334_EXTENDED_M_CODE_UNIT_02_STA_0".M_code[531] )
      wire#w1
      I_Contact( "DB356_M_UNIT_02_STA_0".M_CODES_UNIT_02_STA_0.Ack_M531 )
      I_Contact( "DB2120_MPP_ITC_IPC".RESET_FAULTS )
      I_Contact( "DB356_M_UNIT_02_STA_0".M_CODES_UNIT_02_STA_0.M_RESET_PULSE )
      Coil( "DB356_M_UNIT_02_STA_0".M_CODES_UNIT_02_STA_0.M531 )
   END_RUNG
   RUNG wire#powerrail
      Contact( "DB356_M_UNIT_02_STA_0".M_CODES_UNIT_02_STA_0.M531 )
   END_RUNG wire#w1
   // the same network as SCL:
   "DB356_M_UNIT_02_STA_0".M_CODES_UNIT_02_STA_0.M531 := ("DB334_EXTENDED_M_CODE_UNIT_02_STA_0".M_code[531] OR "DB356_M_UNIT_02_STA_0".M_CODES_UNIT_02_STA_0.M531) AND NOT "DB356_M_UNIT_02_STA_0".M_CODES_UNIT_02_STA_0.Ack_M531 AND NOT "DB2120_MPP_ITC_IPC".RESET_FAULTS AND NOT "DB356_M_UNIT_02_STA_0".M_CODES_UNIT_02_STA_0.M_RESET_PULSE;
END_REGION

REGION Network 81: ACKNOWLEDGE M532-FIXTURE 2 GRIPPER OPEN ONLY PRESSURE SWITCH (READ-IN DISABLE) / ACKNOWLEDGE M120-JAW CHUCK RELAX FIXTURE 1
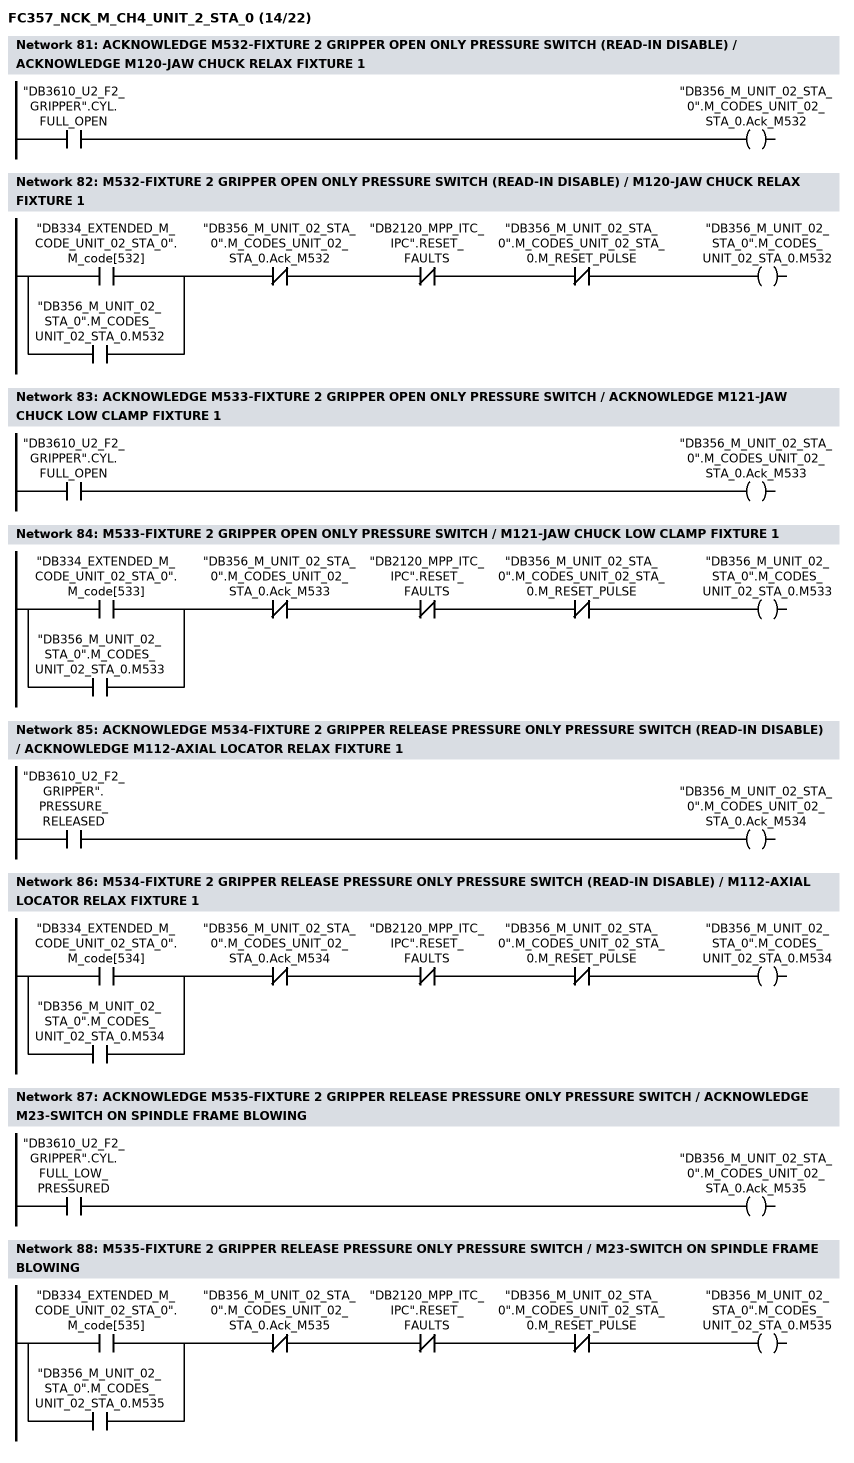
   RUNG wire#powerrail
      Contact( "DB3610_U2_F2_GRIPPER".CYL.FULL_OPEN )
      Coil( "DB356_M_UNIT_02_STA_0".M_CODES_UNIT_02_STA_0.Ack_M532 )
   END_RUNG
   // the same network as SCL:
   "DB356_M_UNIT_02_STA_0".M_CODES_UNIT_02_STA_0.Ack_M532 := "DB3610_U2_F2_GRIPPER".CYL.FULL_OPEN;
END_REGION

REGION Network 82: M532-FIXTURE 2 GRIPPER OPEN ONLY PRESSURE SWITCH (READ-IN DISABLE) / M120-JAW CHUCK RELAX FIXTURE 1
   RUNG wire#powerrail
      Contact( "DB334_EXTENDED_M_CODE_UNIT_02_STA_0".M_code[532] )
      wire#w1
      I_Contact( "DB356_M_UNIT_02_STA_0".M_CODES_UNIT_02_STA_0.Ack_M532 )
      I_Contact( "DB2120_MPP_ITC_IPC".RESET_FAULTS )
      I_Contact( "DB356_M_UNIT_02_STA_0".M_CODES_UNIT_02_STA_0.M_RESET_PULSE )
      Coil( "DB356_M_UNIT_02_STA_0".M_CODES_UNIT_02_STA_0.M532 )
   END_RUNG
   RUNG wire#powerrail
      Contact( "DB356_M_UNIT_02_STA_0".M_CODES_UNIT_02_STA_0.M532 )
   END_RUNG wire#w1
   // the same network as SCL:
   "DB356_M_UNIT_02_STA_0".M_CODES_UNIT_02_STA_0.M532 := ("DB334_EXTENDED_M_CODE_UNIT_02_STA_0".M_code[532] OR "DB356_M_UNIT_02_STA_0".M_CODES_UNIT_02_STA_0.M532) AND NOT "DB356_M_UNIT_02_STA_0".M_CODES_UNIT_02_STA_0.Ack_M532 AND NOT "DB2120_MPP_ITC_IPC".RESET_FAULTS AND NOT "DB356_M_UNIT_02_STA_0".M_CODES_UNIT_02_STA_0.M_RESET_PULSE;
END_REGION

REGION Network 83: ACKNOWLEDGE M533-FIXTURE 2 GRIPPER OPEN ONLY PRESSURE SWITCH / ACKNOWLEDGE M121-JAW CHUCK LOW CLAMP FIXTURE 1
   RUNG wire#powerrail
      Contact( "DB3610_U2_F2_GRIPPER".CYL.FULL_OPEN )
      Coil( "DB356_M_UNIT_02_STA_0".M_CODES_UNIT_02_STA_0.Ack_M533 )
   END_RUNG
   // the same network as SCL:
   "DB356_M_UNIT_02_STA_0".M_CODES_UNIT_02_STA_0.Ack_M533 := "DB3610_U2_F2_GRIPPER".CYL.FULL_OPEN;
END_REGION

REGION Network 84: M533-FIXTURE 2 GRIPPER OPEN ONLY PRESSURE SWITCH / M121-JAW CHUCK LOW CLAMP FIXTURE 1
   RUNG wire#powerrail
      Contact( "DB334_EXTENDED_M_CODE_UNIT_02_STA_0".M_code[533] )
      wire#w1
      I_Contact( "DB356_M_UNIT_02_STA_0".M_CODES_UNIT_02_STA_0.Ack_M533 )
      I_Contact( "DB2120_MPP_ITC_IPC".RESET_FAULTS )
      I_Contact( "DB356_M_UNIT_02_STA_0".M_CODES_UNIT_02_STA_0.M_RESET_PULSE )
      Coil( "DB356_M_UNIT_02_STA_0".M_CODES_UNIT_02_STA_0.M533 )
   END_RUNG
   RUNG wire#powerrail
      Contact( "DB356_M_UNIT_02_STA_0".M_CODES_UNIT_02_STA_0.M533 )
   END_RUNG wire#w1
   // the same network as SCL:
   "DB356_M_UNIT_02_STA_0".M_CODES_UNIT_02_STA_0.M533 := ("DB334_EXTENDED_M_CODE_UNIT_02_STA_0".M_code[533] OR "DB356_M_UNIT_02_STA_0".M_CODES_UNIT_02_STA_0.M533) AND NOT "DB356_M_UNIT_02_STA_0".M_CODES_UNIT_02_STA_0.Ack_M533 AND NOT "DB2120_MPP_ITC_IPC".RESET_FAULTS AND NOT "DB356_M_UNIT_02_STA_0".M_CODES_UNIT_02_STA_0.M_RESET_PULSE;
END_REGION

REGION Network 85: ACKNOWLEDGE M534-FIXTURE 2 GRIPPER RELEASE PRESSURE ONLY PRESSURE SWITCH (READ-IN DISABLE) / ACKNOWLEDGE M112-AXIAL LOCATOR RELAX FIXTURE 1
   RUNG wire#powerrail
      Contact( "DB3610_U2_F2_GRIPPER".PRESSURE_RELEASED )
      Coil( "DB356_M_UNIT_02_STA_0".M_CODES_UNIT_02_STA_0.Ack_M534 )
   END_RUNG
   // the same network as SCL:
   "DB356_M_UNIT_02_STA_0".M_CODES_UNIT_02_STA_0.Ack_M534 := "DB3610_U2_F2_GRIPPER".PRESSURE_RELEASED;
END_REGION

REGION Network 86: M534-FIXTURE 2 GRIPPER RELEASE PRESSURE ONLY PRESSURE SWITCH (READ-IN DISABLE) / M112-AXIAL LOCATOR RELAX FIXTURE 1
   RUNG wire#powerrail
      Contact( "DB334_EXTENDED_M_CODE_UNIT_02_STA_0".M_code[534] )
      wire#w1
      I_Contact( "DB356_M_UNIT_02_STA_0".M_CODES_UNIT_02_STA_0.Ack_M534 )
      I_Contact( "DB2120_MPP_ITC_IPC".RESET_FAULTS )
      I_Contact( "DB356_M_UNIT_02_STA_0".M_CODES_UNIT_02_STA_0.M_RESET_PULSE )
      Coil( "DB356_M_UNIT_02_STA_0".M_CODES_UNIT_02_STA_0.M534 )
   END_RUNG
   RUNG wire#powerrail
      Contact( "DB356_M_UNIT_02_STA_0".M_CODES_UNIT_02_STA_0.M534 )
   END_RUNG wire#w1
   // the same network as SCL:
   "DB356_M_UNIT_02_STA_0".M_CODES_UNIT_02_STA_0.M534 := ("DB334_EXTENDED_M_CODE_UNIT_02_STA_0".M_code[534] OR "DB356_M_UNIT_02_STA_0".M_CODES_UNIT_02_STA_0.M534) AND NOT "DB356_M_UNIT_02_STA_0".M_CODES_UNIT_02_STA_0.Ack_M534 AND NOT "DB2120_MPP_ITC_IPC".RESET_FAULTS AND NOT "DB356_M_UNIT_02_STA_0".M_CODES_UNIT_02_STA_0.M_RESET_PULSE;
END_REGION

REGION Network 87: ACKNOWLEDGE M535-FIXTURE 2 GRIPPER RELEASE PRESSURE ONLY PRESSURE SWITCH / ACKNOWLEDGE M23-SWITCH ON SPINDLE FRAME BLOWING
   RUNG wire#powerrail
      Contact( "DB3610_U2_F2_GRIPPER".CYL.FULL_LOW_PRESSURED )
      Coil( "DB356_M_UNIT_02_STA_0".M_CODES_UNIT_02_STA_0.Ack_M535 )
   END_RUNG
   // the same network as SCL:
   "DB356_M_UNIT_02_STA_0".M_CODES_UNIT_02_STA_0.Ack_M535 := "DB3610_U2_F2_GRIPPER".CYL.FULL_LOW_PRESSURED;
END_REGION

REGION Network 88: M535-FIXTURE 2 GRIPPER RELEASE PRESSURE ONLY PRESSURE SWITCH / M23-SWITCH ON SPINDLE FRAME BLOWING
   RUNG wire#powerrail
      Contact( "DB334_EXTENDED_M_CODE_UNIT_02_STA_0".M_code[535] )
      wire#w1
      I_Contact( "DB356_M_UNIT_02_STA_0".M_CODES_UNIT_02_STA_0.Ack_M535 )
      I_Contact( "DB2120_MPP_ITC_IPC".RESET_FAULTS )
      I_Contact( "DB356_M_UNIT_02_STA_0".M_CODES_UNIT_02_STA_0.M_RESET_PULSE )
      Coil( "DB356_M_UNIT_02_STA_0".M_CODES_UNIT_02_STA_0.M535 )
   END_RUNG
   RUNG wire#powerrail
      Contact( "DB356_M_UNIT_02_STA_0".M_CODES_UNIT_02_STA_0.M535 )
   END_RUNG wire#w1
   // the same network as SCL:
   "DB356_M_UNIT_02_STA_0".M_CODES_UNIT_02_STA_0.M535 := ("DB334_EXTENDED_M_CODE_UNIT_02_STA_0".M_code[535] OR "DB356_M_UNIT_02_STA_0".M_CODES_UNIT_02_STA_0.M535) AND NOT "DB356_M_UNIT_02_STA_0".M_CODES_UNIT_02_STA_0.Ack_M535 AND NOT "DB2120_MPP_ITC_IPC".RESET_FAULTS AND NOT "DB356_M_UNIT_02_STA_0".M_CODES_UNIT_02_STA_0.M_RESET_PULSE;
END_REGION

REGION Network 89: ACKNOWLEDGE M600-UNIT 02 FIXTURE 3 CLAMP SEQUENCE (READ-IN DISABLE) / ACKNOWLEDGE M100-CLAMP SEQUENCE FIXTURE 1
   // NOTE: WHEN THERE IS NOT INDEXING TABLE AVAILABLE IN THE MACHINE DELETE 
   // DB2171.DBX5.0 AND DB2171.DBX2.0
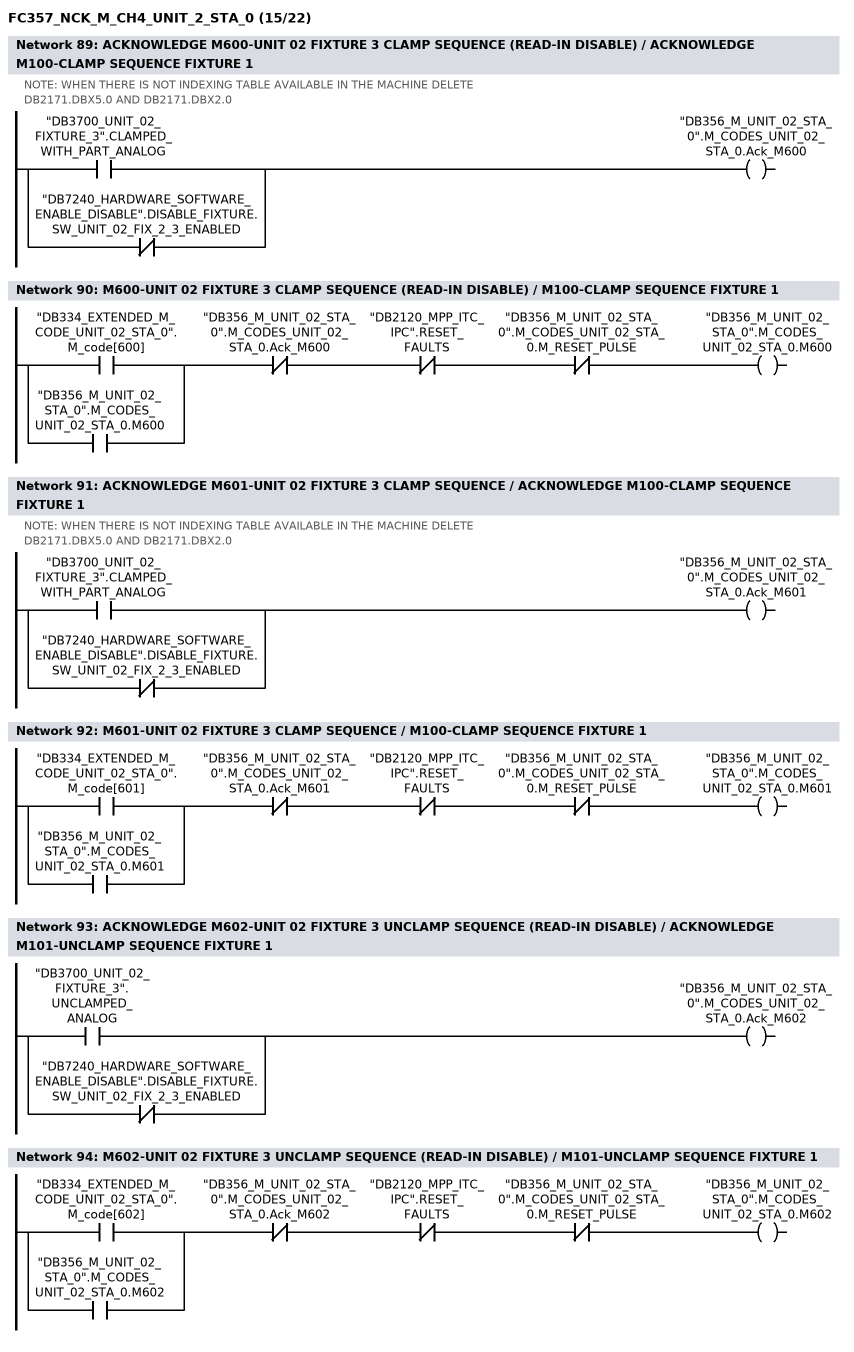
   RUNG wire#powerrail
      Contact( "DB3700_UNIT_02_FIXTURE_3".CLAMPED_WITH_PART_ANALOG )
      wire#w1
      Coil( "DB356_M_UNIT_02_STA_0".M_CODES_UNIT_02_STA_0.Ack_M600 )
   END_RUNG
   RUNG wire#powerrail
      I_Contact( "DB7240_HARDWARE_SOFTWARE_ENABLE_DISABLE".DISABLE_FIXTURE.SW_UNIT_02_FIX_2_3_ENABLED )
   END_RUNG wire#w1
   // the same network as SCL:
   "DB356_M_UNIT_02_STA_0".M_CODES_UNIT_02_STA_0.Ack_M600 := "DB3700_UNIT_02_FIXTURE_3".CLAMPED_WITH_PART_ANALOG OR NOT "DB7240_HARDWARE_SOFTWARE_ENABLE_DISABLE".DISABLE_FIXTURE.SW_UNIT_02_FIX_2_3_ENABLED;
END_REGION

REGION Network 90: M600-UNIT 02 FIXTURE 3 CLAMP SEQUENCE (READ-IN DISABLE) / M100-CLAMP SEQUENCE FIXTURE 1
   RUNG wire#powerrail
      Contact( "DB334_EXTENDED_M_CODE_UNIT_02_STA_0".M_code[600] )
      wire#w1
      I_Contact( "DB356_M_UNIT_02_STA_0".M_CODES_UNIT_02_STA_0.Ack_M600 )
      I_Contact( "DB2120_MPP_ITC_IPC".RESET_FAULTS )
      I_Contact( "DB356_M_UNIT_02_STA_0".M_CODES_UNIT_02_STA_0.M_RESET_PULSE )
      Coil( "DB356_M_UNIT_02_STA_0".M_CODES_UNIT_02_STA_0.M600 )
   END_RUNG
   RUNG wire#powerrail
      Contact( "DB356_M_UNIT_02_STA_0".M_CODES_UNIT_02_STA_0.M600 )
   END_RUNG wire#w1
   // the same network as SCL:
   "DB356_M_UNIT_02_STA_0".M_CODES_UNIT_02_STA_0.M600 := ("DB334_EXTENDED_M_CODE_UNIT_02_STA_0".M_code[600] OR "DB356_M_UNIT_02_STA_0".M_CODES_UNIT_02_STA_0.M600) AND NOT "DB356_M_UNIT_02_STA_0".M_CODES_UNIT_02_STA_0.Ack_M600 AND NOT "DB2120_MPP_ITC_IPC".RESET_FAULTS AND NOT "DB356_M_UNIT_02_STA_0".M_CODES_UNIT_02_STA_0.M_RESET_PULSE;
END_REGION

REGION Network 91: ACKNOWLEDGE M601-UNIT 02 FIXTURE 3 CLAMP SEQUENCE / ACKNOWLEDGE M100-CLAMP SEQUENCE FIXTURE 1
   // NOTE: WHEN THERE IS NOT INDEXING TABLE AVAILABLE IN THE MACHINE DELETE 
   // DB2171.DBX5.0 AND DB2171.DBX2.0
   RUNG wire#powerrail
      Contact( "DB3700_UNIT_02_FIXTURE_3".CLAMPED_WITH_PART_ANALOG )
      wire#w1
      Coil( "DB356_M_UNIT_02_STA_0".M_CODES_UNIT_02_STA_0.Ack_M601 )
   END_RUNG
   RUNG wire#powerrail
      I_Contact( "DB7240_HARDWARE_SOFTWARE_ENABLE_DISABLE".DISABLE_FIXTURE.SW_UNIT_02_FIX_2_3_ENABLED )
   END_RUNG wire#w1
   // the same network as SCL:
   "DB356_M_UNIT_02_STA_0".M_CODES_UNIT_02_STA_0.Ack_M601 := "DB3700_UNIT_02_FIXTURE_3".CLAMPED_WITH_PART_ANALOG OR NOT "DB7240_HARDWARE_SOFTWARE_ENABLE_DISABLE".DISABLE_FIXTURE.SW_UNIT_02_FIX_2_3_ENABLED;
END_REGION

REGION Network 92: M601-UNIT 02 FIXTURE 3 CLAMP SEQUENCE / M100-CLAMP SEQUENCE FIXTURE 1
   RUNG wire#powerrail
      Contact( "DB334_EXTENDED_M_CODE_UNIT_02_STA_0".M_code[601] )
      wire#w1
      I_Contact( "DB356_M_UNIT_02_STA_0".M_CODES_UNIT_02_STA_0.Ack_M601 )
      I_Contact( "DB2120_MPP_ITC_IPC".RESET_FAULTS )
      I_Contact( "DB356_M_UNIT_02_STA_0".M_CODES_UNIT_02_STA_0.M_RESET_PULSE )
      Coil( "DB356_M_UNIT_02_STA_0".M_CODES_UNIT_02_STA_0.M601 )
   END_RUNG
   RUNG wire#powerrail
      Contact( "DB356_M_UNIT_02_STA_0".M_CODES_UNIT_02_STA_0.M601 )
   END_RUNG wire#w1
   // the same network as SCL:
   "DB356_M_UNIT_02_STA_0".M_CODES_UNIT_02_STA_0.M601 := ("DB334_EXTENDED_M_CODE_UNIT_02_STA_0".M_code[601] OR "DB356_M_UNIT_02_STA_0".M_CODES_UNIT_02_STA_0.M601) AND NOT "DB356_M_UNIT_02_STA_0".M_CODES_UNIT_02_STA_0.Ack_M601 AND NOT "DB2120_MPP_ITC_IPC".RESET_FAULTS AND NOT "DB356_M_UNIT_02_STA_0".M_CODES_UNIT_02_STA_0.M_RESET_PULSE;
END_REGION

REGION Network 93: ACKNOWLEDGE M602-UNIT 02 FIXTURE 3 UNCLAMP SEQUENCE (READ-IN DISABLE) / ACKNOWLEDGE M101-UNCLAMP SEQUENCE FIXTURE 1
   RUNG wire#powerrail
      Contact( "DB3700_UNIT_02_FIXTURE_3".UNCLAMPED_ANALOG )
      wire#w1
      Coil( "DB356_M_UNIT_02_STA_0".M_CODES_UNIT_02_STA_0.Ack_M602 )
   END_RUNG
   RUNG wire#powerrail
      I_Contact( "DB7240_HARDWARE_SOFTWARE_ENABLE_DISABLE".DISABLE_FIXTURE.SW_UNIT_02_FIX_2_3_ENABLED )
   END_RUNG wire#w1
   // the same network as SCL:
   "DB356_M_UNIT_02_STA_0".M_CODES_UNIT_02_STA_0.Ack_M602 := "DB3700_UNIT_02_FIXTURE_3".UNCLAMPED_ANALOG OR NOT "DB7240_HARDWARE_SOFTWARE_ENABLE_DISABLE".DISABLE_FIXTURE.SW_UNIT_02_FIX_2_3_ENABLED;
END_REGION

REGION Network 94: M602-UNIT 02 FIXTURE 3 UNCLAMP SEQUENCE (READ-IN DISABLE) / M101-UNCLAMP SEQUENCE FIXTURE 1
   RUNG wire#powerrail
      Contact( "DB334_EXTENDED_M_CODE_UNIT_02_STA_0".M_code[602] )
      wire#w1
      I_Contact( "DB356_M_UNIT_02_STA_0".M_CODES_UNIT_02_STA_0.Ack_M602 )
      I_Contact( "DB2120_MPP_ITC_IPC".RESET_FAULTS )
      I_Contact( "DB356_M_UNIT_02_STA_0".M_CODES_UNIT_02_STA_0.M_RESET_PULSE )
      Coil( "DB356_M_UNIT_02_STA_0".M_CODES_UNIT_02_STA_0.M602 )
   END_RUNG
   RUNG wire#powerrail
      Contact( "DB356_M_UNIT_02_STA_0".M_CODES_UNIT_02_STA_0.M602 )
   END_RUNG wire#w1
   // the same network as SCL:
   "DB356_M_UNIT_02_STA_0".M_CODES_UNIT_02_STA_0.M602 := ("DB334_EXTENDED_M_CODE_UNIT_02_STA_0".M_code[602] OR "DB356_M_UNIT_02_STA_0".M_CODES_UNIT_02_STA_0.M602) AND NOT "DB356_M_UNIT_02_STA_0".M_CODES_UNIT_02_STA_0.Ack_M602 AND NOT "DB2120_MPP_ITC_IPC".RESET_FAULTS AND NOT "DB356_M_UNIT_02_STA_0".M_CODES_UNIT_02_STA_0.M_RESET_PULSE;
END_REGION

REGION Network 95: ACKNOWLEDGE M603-UNIT 02 FIXTURE 3 UNCLAMP SEQUENCE / ACKNOWLEDGE M101-UNCLAMP SEQUENCE FIXTURE 1
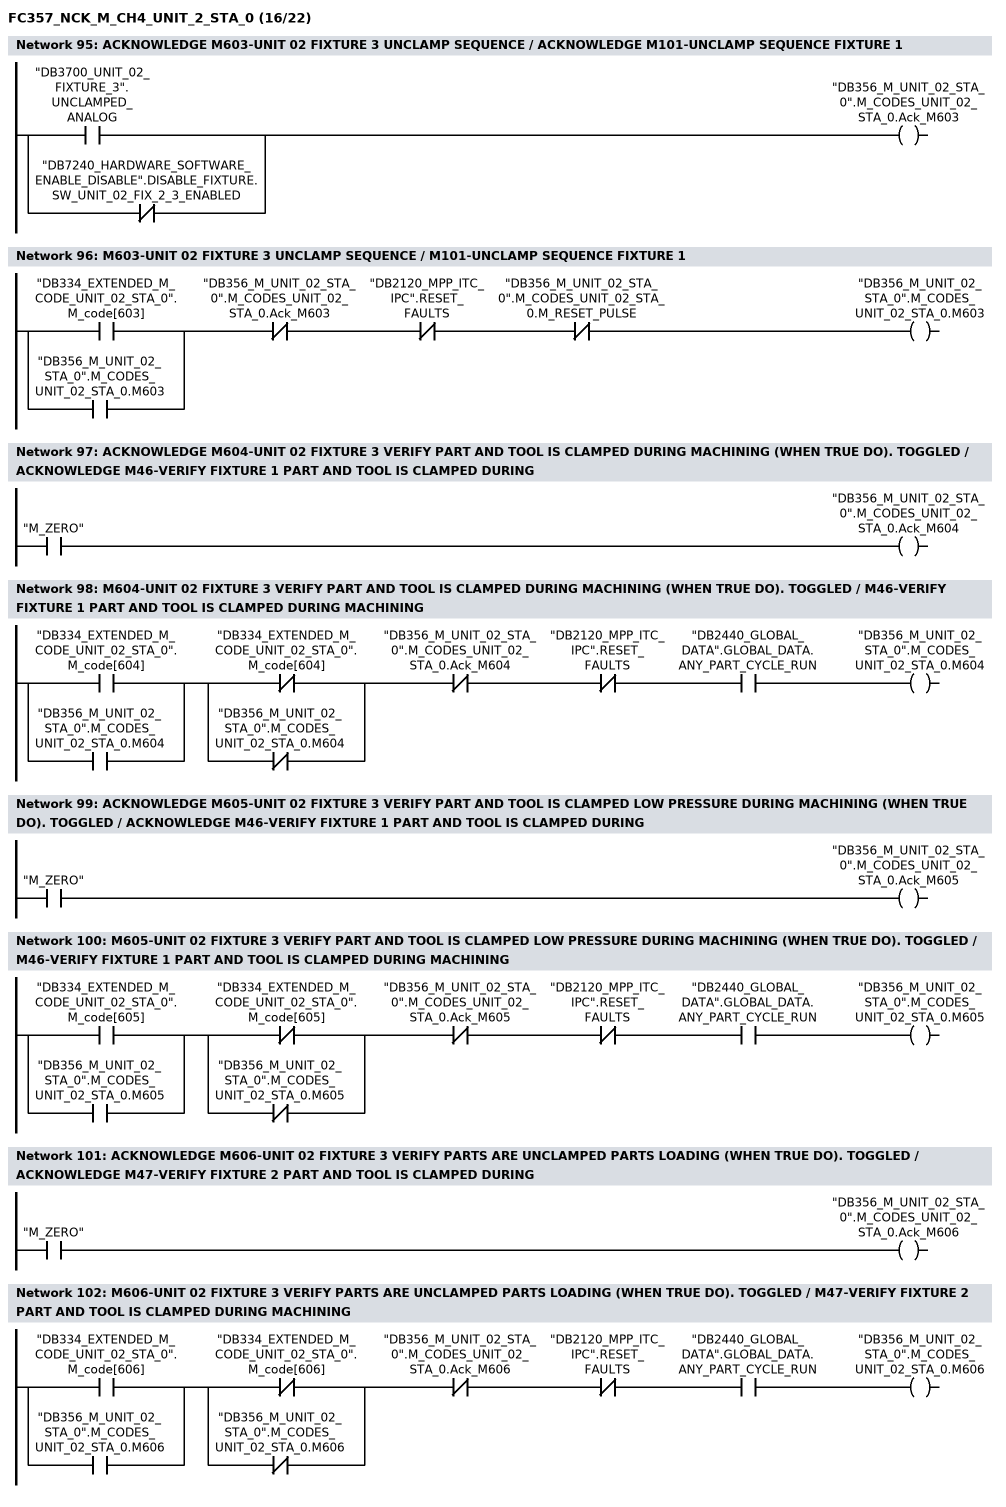
   RUNG wire#powerrail
      Contact( "DB3700_UNIT_02_FIXTURE_3".UNCLAMPED_ANALOG )
      wire#w1
      Coil( "DB356_M_UNIT_02_STA_0".M_CODES_UNIT_02_STA_0.Ack_M603 )
   END_RUNG
   RUNG wire#powerrail
      I_Contact( "DB7240_HARDWARE_SOFTWARE_ENABLE_DISABLE".DISABLE_FIXTURE.SW_UNIT_02_FIX_2_3_ENABLED )
   END_RUNG wire#w1
   // the same network as SCL:
   "DB356_M_UNIT_02_STA_0".M_CODES_UNIT_02_STA_0.Ack_M603 := "DB3700_UNIT_02_FIXTURE_3".UNCLAMPED_ANALOG OR NOT "DB7240_HARDWARE_SOFTWARE_ENABLE_DISABLE".DISABLE_FIXTURE.SW_UNIT_02_FIX_2_3_ENABLED;
END_REGION

REGION Network 96: M603-UNIT 02 FIXTURE 3 UNCLAMP SEQUENCE / M101-UNCLAMP SEQUENCE FIXTURE 1
   RUNG wire#powerrail
      Contact( "DB334_EXTENDED_M_CODE_UNIT_02_STA_0".M_code[603] )
      wire#w1
      I_Contact( "DB356_M_UNIT_02_STA_0".M_CODES_UNIT_02_STA_0.Ack_M603 )
      I_Contact( "DB2120_MPP_ITC_IPC".RESET_FAULTS )
      I_Contact( "DB356_M_UNIT_02_STA_0".M_CODES_UNIT_02_STA_0.M_RESET_PULSE )
      Coil( "DB356_M_UNIT_02_STA_0".M_CODES_UNIT_02_STA_0.M603 )
   END_RUNG
   RUNG wire#powerrail
      Contact( "DB356_M_UNIT_02_STA_0".M_CODES_UNIT_02_STA_0.M603 )
   END_RUNG wire#w1
   // the same network as SCL:
   "DB356_M_UNIT_02_STA_0".M_CODES_UNIT_02_STA_0.M603 := ("DB334_EXTENDED_M_CODE_UNIT_02_STA_0".M_code[603] OR "DB356_M_UNIT_02_STA_0".M_CODES_UNIT_02_STA_0.M603) AND NOT "DB356_M_UNIT_02_STA_0".M_CODES_UNIT_02_STA_0.Ack_M603 AND NOT "DB2120_MPP_ITC_IPC".RESET_FAULTS AND NOT "DB356_M_UNIT_02_STA_0".M_CODES_UNIT_02_STA_0.M_RESET_PULSE;
END_REGION

REGION Network 97: ACKNOWLEDGE M604-UNIT 02 FIXTURE 3 VERIFY PART AND TOOL IS CLAMPED DURING MACHINING (WHEN TRUE DO). TOGGLED / ACKNOWLEDGE M46-VERIFY FIXTURE 1 PART AND TOOL IS CLAMPED DURING
   RUNG wire#powerrail
      Contact( "M_ZERO" )
      Coil( "DB356_M_UNIT_02_STA_0".M_CODES_UNIT_02_STA_0.Ack_M604 )
   END_RUNG
   // the same network as SCL:
   "DB356_M_UNIT_02_STA_0".M_CODES_UNIT_02_STA_0.Ack_M604 := "M_ZERO";
END_REGION

REGION Network 98: M604-UNIT 02 FIXTURE 3 VERIFY PART AND TOOL IS CLAMPED DURING MACHINING (WHEN TRUE DO). TOGGLED / M46-VERIFY FIXTURE 1 PART AND TOOL IS CLAMPED DURING MACHINING
   RUNG wire#powerrail
      Contact( "DB334_EXTENDED_M_CODE_UNIT_02_STA_0".M_code[604] )
      wire#w1
      I_Contact( "DB334_EXTENDED_M_CODE_UNIT_02_STA_0".M_code[604] )
      wire#w2
      I_Contact( "DB356_M_UNIT_02_STA_0".M_CODES_UNIT_02_STA_0.Ack_M604 )
      I_Contact( "DB2120_MPP_ITC_IPC".RESET_FAULTS )
      Contact( "DB2440_GLOBAL_DATA".GLOBAL_DATA.ANY_PART_CYCLE_RUN )
      Coil( "DB356_M_UNIT_02_STA_0".M_CODES_UNIT_02_STA_0.M604 )
   END_RUNG
   RUNG wire#powerrail
      Contact( "DB356_M_UNIT_02_STA_0".M_CODES_UNIT_02_STA_0.M604 )
   END_RUNG wire#w1
   RUNG wire#w1
      I_Contact( "DB356_M_UNIT_02_STA_0".M_CODES_UNIT_02_STA_0.M604 )
   END_RUNG wire#w2
   // the same network as SCL:
   "DB356_M_UNIT_02_STA_0".M_CODES_UNIT_02_STA_0.M604 := ("DB334_EXTENDED_M_CODE_UNIT_02_STA_0".M_code[604] OR "DB356_M_UNIT_02_STA_0".M_CODES_UNIT_02_STA_0.M604) AND (NOT "DB334_EXTENDED_M_CODE_UNIT_02_STA_0".M_code[604] OR NOT "DB356_M_UNIT_02_STA_0".M_CODES_UNIT_02_STA_0.M604) AND NOT "DB356_M_UNIT_02_STA_0".M_CODES_UNIT_02_STA_0.Ack_M604 AND NOT "DB2120_MPP_ITC_IPC".RESET_FAULTS AND "DB2440_GLOBAL_DATA".GLOBAL_DATA.ANY_PART_CYCLE_RUN;
END_REGION

REGION Network 99: ACKNOWLEDGE M605-UNIT 02 FIXTURE 3 VERIFY PART AND TOOL IS CLAMPED LOW PRESSURE DURING MACHINING (WHEN TRUE DO). TOGGLED / ACKNOWLEDGE M46-VERIFY FIXTURE 1 PART AND TOOL IS CLAMPED DURING
   RUNG wire#powerrail
      Contact( "M_ZERO" )
      Coil( "DB356_M_UNIT_02_STA_0".M_CODES_UNIT_02_STA_0.Ack_M605 )
   END_RUNG
   // the same network as SCL:
   "DB356_M_UNIT_02_STA_0".M_CODES_UNIT_02_STA_0.Ack_M605 := "M_ZERO";
END_REGION

REGION Network 100: M605-UNIT 02 FIXTURE 3 VERIFY PART AND TOOL IS CLAMPED LOW PRESSURE DURING MACHINING (WHEN TRUE DO). TOGGLED / M46-VERIFY FIXTURE 1 PART AND TOOL IS CLAMPED DURING MACHINING
   RUNG wire#powerrail
      Contact( "DB334_EXTENDED_M_CODE_UNIT_02_STA_0".M_code[605] )
      wire#w1
      I_Contact( "DB334_EXTENDED_M_CODE_UNIT_02_STA_0".M_code[605] )
      wire#w2
      I_Contact( "DB356_M_UNIT_02_STA_0".M_CODES_UNIT_02_STA_0.Ack_M605 )
      I_Contact( "DB2120_MPP_ITC_IPC".RESET_FAULTS )
      Contact( "DB2440_GLOBAL_DATA".GLOBAL_DATA.ANY_PART_CYCLE_RUN )
      Coil( "DB356_M_UNIT_02_STA_0".M_CODES_UNIT_02_STA_0.M605 )
   END_RUNG
   RUNG wire#powerrail
      Contact( "DB356_M_UNIT_02_STA_0".M_CODES_UNIT_02_STA_0.M605 )
   END_RUNG wire#w1
   RUNG wire#w1
      I_Contact( "DB356_M_UNIT_02_STA_0".M_CODES_UNIT_02_STA_0.M605 )
   END_RUNG wire#w2
   // the same network as SCL:
   "DB356_M_UNIT_02_STA_0".M_CODES_UNIT_02_STA_0.M605 := ("DB334_EXTENDED_M_CODE_UNIT_02_STA_0".M_code[605] OR "DB356_M_UNIT_02_STA_0".M_CODES_UNIT_02_STA_0.M605) AND (NOT "DB334_EXTENDED_M_CODE_UNIT_02_STA_0".M_code[605] OR NOT "DB356_M_UNIT_02_STA_0".M_CODES_UNIT_02_STA_0.M605) AND NOT "DB356_M_UNIT_02_STA_0".M_CODES_UNIT_02_STA_0.Ack_M605 AND NOT "DB2120_MPP_ITC_IPC".RESET_FAULTS AND "DB2440_GLOBAL_DATA".GLOBAL_DATA.ANY_PART_CYCLE_RUN;
END_REGION

REGION Network 101: ACKNOWLEDGE M606-UNIT 02 FIXTURE 3 VERIFY PARTS ARE UNCLAMPED PARTS LOADING (WHEN TRUE DO). TOGGLED / ACKNOWLEDGE M47-VERIFY FIXTURE 2 PART AND TOOL IS CLAMPED DURING
   RUNG wire#powerrail
      Contact( "M_ZERO" )
      Coil( "DB356_M_UNIT_02_STA_0".M_CODES_UNIT_02_STA_0.Ack_M606 )
   END_RUNG
   // the same network as SCL:
   "DB356_M_UNIT_02_STA_0".M_CODES_UNIT_02_STA_0.Ack_M606 := "M_ZERO";
END_REGION

REGION Network 102: M606-UNIT 02 FIXTURE 3 VERIFY PARTS ARE UNCLAMPED PARTS LOADING (WHEN TRUE DO). TOGGLED / M47-VERIFY FIXTURE 2 PART AND TOOL IS CLAMPED DURING MACHINING
   RUNG wire#powerrail
      Contact( "DB334_EXTENDED_M_CODE_UNIT_02_STA_0".M_code[606] )
      wire#w1
      I_Contact( "DB334_EXTENDED_M_CODE_UNIT_02_STA_0".M_code[606] )
      wire#w2
      I_Contact( "DB356_M_UNIT_02_STA_0".M_CODES_UNIT_02_STA_0.Ack_M606 )
      I_Contact( "DB2120_MPP_ITC_IPC".RESET_FAULTS )
      Contact( "DB2440_GLOBAL_DATA".GLOBAL_DATA.ANY_PART_CYCLE_RUN )
      Coil( "DB356_M_UNIT_02_STA_0".M_CODES_UNIT_02_STA_0.M606 )
   END_RUNG
   RUNG wire#powerrail
      Contact( "DB356_M_UNIT_02_STA_0".M_CODES_UNIT_02_STA_0.M606 )
   END_RUNG wire#w1
   RUNG wire#w1
      I_Contact( "DB356_M_UNIT_02_STA_0".M_CODES_UNIT_02_STA_0.M606 )
   END_RUNG wire#w2
   // the same network as SCL:
   "DB356_M_UNIT_02_STA_0".M_CODES_UNIT_02_STA_0.M606 := ("DB334_EXTENDED_M_CODE_UNIT_02_STA_0".M_code[606] OR "DB356_M_UNIT_02_STA_0".M_CODES_UNIT_02_STA_0.M606) AND (NOT "DB334_EXTENDED_M_CODE_UNIT_02_STA_0".M_code[606] OR NOT "DB356_M_UNIT_02_STA_0".M_CODES_UNIT_02_STA_0.M606) AND NOT "DB356_M_UNIT_02_STA_0".M_CODES_UNIT_02_STA_0.Ack_M606 AND NOT "DB2120_MPP_ITC_IPC".RESET_FAULTS AND "DB2440_GLOBAL_DATA".GLOBAL_DATA.ANY_PART_CYCLE_RUN;
END_REGION

REGION Network 103: ACKNOWLEDGE M607-UNIT 02 FIXTURE 3 VERIFY FIXTURE REMAINS CLAMPED
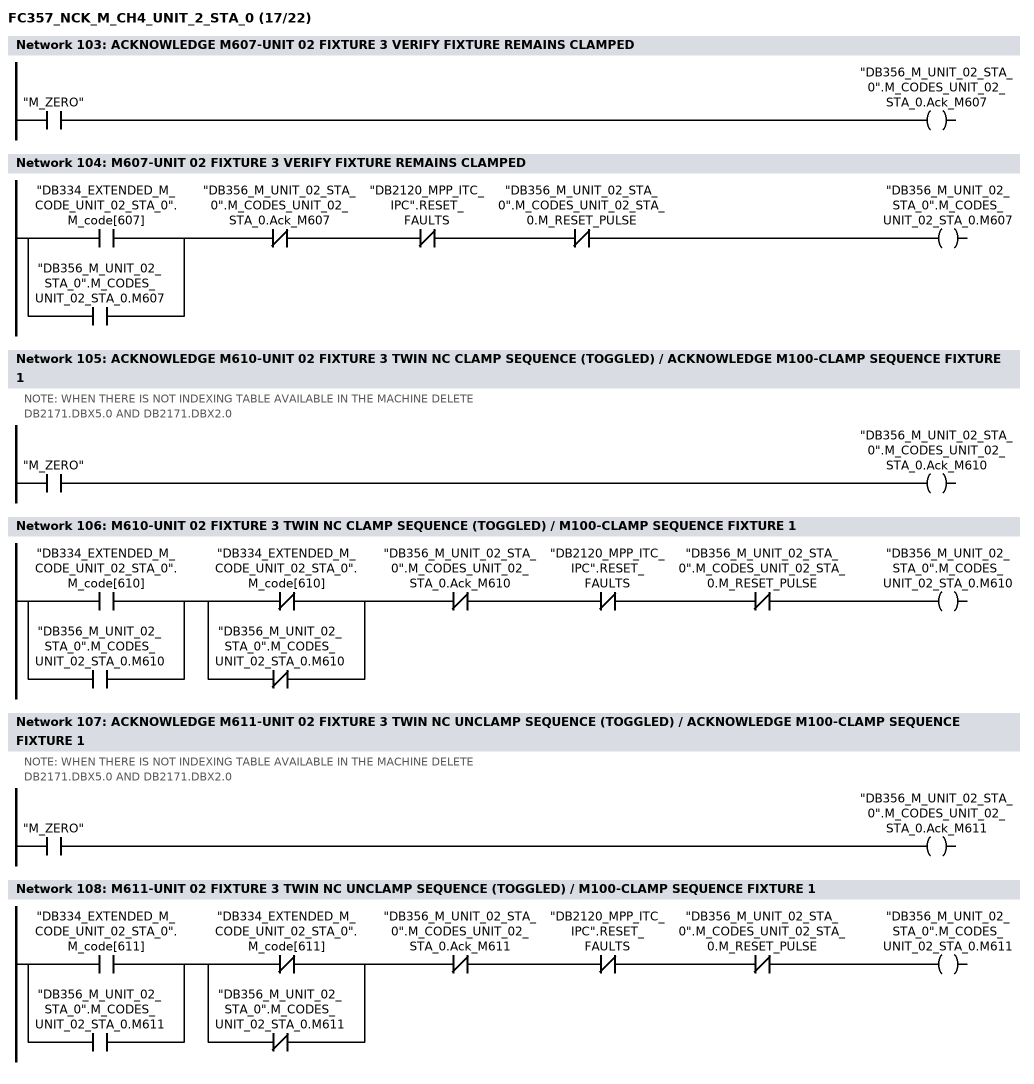
   RUNG wire#powerrail
      Contact( "M_ZERO" )
      Coil( "DB356_M_UNIT_02_STA_0".M_CODES_UNIT_02_STA_0.Ack_M607 )
   END_RUNG
   // the same network as SCL:
   "DB356_M_UNIT_02_STA_0".M_CODES_UNIT_02_STA_0.Ack_M607 := "M_ZERO";
END_REGION

REGION Network 104: M607-UNIT 02 FIXTURE 3 VERIFY FIXTURE REMAINS CLAMPED
   RUNG wire#powerrail
      Contact( "DB334_EXTENDED_M_CODE_UNIT_02_STA_0".M_code[607] )
      wire#w1
      I_Contact( "DB356_M_UNIT_02_STA_0".M_CODES_UNIT_02_STA_0.Ack_M607 )
      I_Contact( "DB2120_MPP_ITC_IPC".RESET_FAULTS )
      I_Contact( "DB356_M_UNIT_02_STA_0".M_CODES_UNIT_02_STA_0.M_RESET_PULSE )
      Coil( "DB356_M_UNIT_02_STA_0".M_CODES_UNIT_02_STA_0.M607 )
   END_RUNG
   RUNG wire#powerrail
      Contact( "DB356_M_UNIT_02_STA_0".M_CODES_UNIT_02_STA_0.M607 )
   END_RUNG wire#w1
   // the same network as SCL:
   "DB356_M_UNIT_02_STA_0".M_CODES_UNIT_02_STA_0.M607 := ("DB334_EXTENDED_M_CODE_UNIT_02_STA_0".M_code[607] OR "DB356_M_UNIT_02_STA_0".M_CODES_UNIT_02_STA_0.M607) AND NOT "DB356_M_UNIT_02_STA_0".M_CODES_UNIT_02_STA_0.Ack_M607 AND NOT "DB2120_MPP_ITC_IPC".RESET_FAULTS AND NOT "DB356_M_UNIT_02_STA_0".M_CODES_UNIT_02_STA_0.M_RESET_PULSE;
END_REGION

REGION Network 105: ACKNOWLEDGE M610-UNIT 02 FIXTURE 3 TWIN NC CLAMP SEQUENCE (TOGGLED) / ACKNOWLEDGE M100-CLAMP SEQUENCE FIXTURE 1
   // NOTE: WHEN THERE IS NOT INDEXING TABLE AVAILABLE IN THE MACHINE DELETE 
   // DB2171.DBX5.0 AND DB2171.DBX2.0
   RUNG wire#powerrail
      Contact( "M_ZERO" )
      Coil( "DB356_M_UNIT_02_STA_0".M_CODES_UNIT_02_STA_0.Ack_M610 )
   END_RUNG
   // the same network as SCL:
   "DB356_M_UNIT_02_STA_0".M_CODES_UNIT_02_STA_0.Ack_M610 := "M_ZERO";
END_REGION

REGION Network 106: M610-UNIT 02 FIXTURE 3 TWIN NC CLAMP SEQUENCE (TOGGLED) / M100-CLAMP SEQUENCE FIXTURE 1
   RUNG wire#powerrail
      Contact( "DB334_EXTENDED_M_CODE_UNIT_02_STA_0".M_code[610] )
      wire#w1
      I_Contact( "DB334_EXTENDED_M_CODE_UNIT_02_STA_0".M_code[610] )
      wire#w2
      I_Contact( "DB356_M_UNIT_02_STA_0".M_CODES_UNIT_02_STA_0.Ack_M610 )
      I_Contact( "DB2120_MPP_ITC_IPC".RESET_FAULTS )
      I_Contact( "DB356_M_UNIT_02_STA_0".M_CODES_UNIT_02_STA_0.M_RESET_PULSE )
      Coil( "DB356_M_UNIT_02_STA_0".M_CODES_UNIT_02_STA_0.M610 )
   END_RUNG
   RUNG wire#powerrail
      Contact( "DB356_M_UNIT_02_STA_0".M_CODES_UNIT_02_STA_0.M610 )
   END_RUNG wire#w1
   RUNG wire#w1
      I_Contact( "DB356_M_UNIT_02_STA_0".M_CODES_UNIT_02_STA_0.M610 )
   END_RUNG wire#w2
   // the same network as SCL:
   "DB356_M_UNIT_02_STA_0".M_CODES_UNIT_02_STA_0.M610 := ("DB334_EXTENDED_M_CODE_UNIT_02_STA_0".M_code[610] OR "DB356_M_UNIT_02_STA_0".M_CODES_UNIT_02_STA_0.M610) AND (NOT "DB334_EXTENDED_M_CODE_UNIT_02_STA_0".M_code[610] OR NOT "DB356_M_UNIT_02_STA_0".M_CODES_UNIT_02_STA_0.M610) AND NOT "DB356_M_UNIT_02_STA_0".M_CODES_UNIT_02_STA_0.Ack_M610 AND NOT "DB2120_MPP_ITC_IPC".RESET_FAULTS AND NOT "DB356_M_UNIT_02_STA_0".M_CODES_UNIT_02_STA_0.M_RESET_PULSE;
END_REGION

REGION Network 107: ACKNOWLEDGE M611-UNIT 02 FIXTURE 3 TWIN NC UNCLAMP SEQUENCE (TOGGLED) / ACKNOWLEDGE M100-CLAMP SEQUENCE FIXTURE 1
   // NOTE: WHEN THERE IS NOT INDEXING TABLE AVAILABLE IN THE MACHINE DELETE 
   // DB2171.DBX5.0 AND DB2171.DBX2.0
   RUNG wire#powerrail
      Contact( "M_ZERO" )
      Coil( "DB356_M_UNIT_02_STA_0".M_CODES_UNIT_02_STA_0.Ack_M611 )
   END_RUNG
   // the same network as SCL:
   "DB356_M_UNIT_02_STA_0".M_CODES_UNIT_02_STA_0.Ack_M611 := "M_ZERO";
END_REGION

